   CASE IP_Arr_OP90JB[Input_Page_num] OF
	500: Lamp4:=I90_BOWL1_RDYI500_3 ;
	501: Lamp4:=I90_CONV1_TRK1_CHO_MOD1I501_3 ;
	502: Lamp4:=I90_HPR2_SOL_DOOR_SW_FBI502_3 ;
	503: Lamp4:=I90_VBF1_CONV2_TRK2_OVERFLWI503_3;
	504: Lamp4:=I90_VBF2_CONV_TRK_OVERFLW_2I504_3 ;
	505: Lamp4:=I90_SPARE_I505_3 ;
   ELSE
       Visibility_4:=FALSE;	
   END_CASE
   
   
    Visibility_5:=TRUE;
   
   CASE IP_Arr_OP90JB[Input_Page_num] OF
	500: Lamp5:=I90_BOWL1_LOW_LVLI500_4 ;
	501: Lamp5:=I90_CONV1_TRK1_CHO_MOD2I501_4 ;
	502: Lamp5:=I90_BOWL2_RDYI502_4 ;
	503: Lamp5:=I90_CONV2_TRK1_CHO_MOD1I503_4;
	504: Lamp5:=I90_SPARE_I504_4 ;
	505: Lamp5:=I90_SPARE_I505_4 ;
   ELSE
       Visibility_5:=FALSE;	
   END_CASE
   
   
    Visibility_6:=TRUE;
   
   CASE IP_Arr_OP90JB[Input_Page_num] OF
	500: Lamp6:=I90_BOWL1_OFF_ONI500_5 ;
	501: Lamp6:=I90_CONV1_TRK2_CHO_MOD1I501_5 ;
	502: Lamp6:=I90_BOWL2_LOW_LVLI502_5 ;
	503: Lamp6:=I90_CONV2_TRK1_CHO_MOD2I503_5;
	504: Lamp6:=I90_SPARE_I504_5 ;
	505: Lamp6:=I90_SPARE_I505_5 ;
   ELSE
       Visibility_6:=FALSE;	
   END_CASE
   
   
    Visibility_7:=TRUE;
   
   CASE IP_Arr_OP90JB[Input_Page_num] OF
	500: Lamp7:=I90_HPR1_OFF_ONI500_6 ;
	501: Lamp7:=I90_CONV1_TRK2_CHO_MOD2I501_6 ;
	502: Lamp7:=I90_BOWL2_OFF_ONI502_6 ;
	503: Lamp7:=I90_CONV2_TRK2_CHO_MOD1I503_6;
	504: Lamp7:=I90_SPARE_I504_6 ;
	505: Lamp7:=I90_SPARE_I505_6 ;
   ELSE
       Visibility_7:=FALSE;	
   END_CASE
   
   
    Visibility_8:=TRUE;
   
   CASE IP_Arr_OP90JB[Input_Page_num] OF
	500: Lamp8:=I90_CONV1_REVI500_7 ;
	501: Lamp8:=I90_CONV1_TRK3_CHO_MOD1I501_7 ;
	502: Lamp8:=I90_HPR2_OFF_ONI502_7 ;
	503: Lamp8:=I90_CONV2_TRK2_CHO_MOD2I503_7;
	504: Lamp8:=I90_SPARE_I504_7 ;
	505: Lamp8:=I90_SPARE_I505_7 ;
   ELSE
       Visibility_8:=FALSE;	
   END_CASE
	
    CASE OP_Arr_OP90[Output_Page_num] OF
    500: OLine1:=" O90_HPR1_ENABLE(Q500.0)  ";
    501: OLine1:=" O90_HPR2_ENABLE(Q501.0)  ";
    502: OLine1:=" O90_SPARE_Q502_0(Q502.0) ";
    503: OLine1:=" O90_SPARE_Q503_0(Q503.0) ";
    else
     OLine1:=" ";
    end_case 
    
    CASE OP_Arr_OP90[Output_Page_num] OF
    500: OLine2:="O90_BOWL1_ENABLE(Q500.1)";
    501: OLine2:="O90_BOWL2_ENABLE(Q501.1)";
    502: OLine2:="O90_SPARE_Q502_1(Q502.1)";
    503: OLine2:="O90_SPARE_Q503_1(Q503.1)";
    else
     OLine2:=" ";
    end_case 
    
    CASE OP_Arr_OP90[Output_Page_num] OF
    500: OLine3:="O90_HPR1_TWR_LMP_RED(Q500.2)";
    501: OLine3:="O90_HPR2_TWR_LMP_RED(Q501.2)";
    502: OLine3:="O90_SPARE_Q502_2(Q502.2)    ";
    503: OLine3:="O90_SPARE_Q503_2(Q503.2)    ";
    else
     OLine3:=" ";
    end_case 
    
    CASE OP_Arr_OP90[Output_Page_num] OF
    500: OLine4:="O90_HPR1_TWR_LMP_GREEN(Q500.3)";
    501: OLine4:="O90_HPR2_TWR_LMP_GREEN(Q501.3)";
    502: OLine4:="O90_SPARE_Q502_3(Q502.3)      ";
    503: OLine4:="O90_SPARE_Q503_3(Q503.3)      ";
    else
     OLine4:=" ";
    end_case 
    
    CASE OP_Arr_OP90[Output_Page_num] OF
    500: OLine5:="O90_BOWL1_AIR_PURGE1(Q500.4)";
    501: OLine5:="O90_BOWL2_AIR_PURGE1(Q501.4)";
    502: OLine5:="O90_SPARE_Q502_4(Q502.4)    ";
    503: OLine5:="O90_SPARE_Q503_4(Q503.4)    ";
    else
     OLine5:=" ";
    end_case 
    
    CASE OP_Arr_OP90[Output_Page_num] OF
    500: OLine6:="O90_BOWL1_AIR_PURGE2(Q500.5)";
    501: OLine6:="O90_BOWL2_AIR_PURGE2(Q501.5)";
    502: OLine6:="O90_SPARE_Q502_5(Q502.5)    ";
    503: OLine6:="O90_SPARE_Q503_5(Q503.5)    ";
    else
     OLine6:=" ";
    end_case 
    
    CASE OP_Arr_OP90[Output_Page_num] OF
    500: OLine7:="O90_HPR1_DOOR_OPN(Q500.6)";
    501: OLine7:="O90_HPR2_DOOR_OPN(Q501.6)";
    502: OLine7:="O90_SPARE_Q502_6(Q502.6) ";
    503: OLine7:="O90_SPARE_Q503_6(Q503.6) ";
    else
     OLine7:=" ";
    end_case 
    
    CASE OP_Arr_OP90[Output_Page_num] OF
    500: OLine8:="O90_SPARE_Q500_7(Q500.7)";
    501: OLine8:="O90_SPARE_Q501_7(Q501.7)";
    502: OLine8:="O90_SPARE_Q502_7(Q502.7)";
    503: OLine8:="O90_SPARE_Q503_7(Q503.7)";
    else
     OLine8:=" ";
    END_CASE 
    Out_Visibility_1:=TRUE;
    CASE OP_Arr_OP90[Output_Page_num] OF
	500:  Out_Lamp1:=O90_HPR1_ENABLEQ500_0;
	501:  Out_Lamp1:=O90_HPR2_ENABLEQ501_0;
	502:  Out_Lamp1:=O90_SPARE_Q502_0;
	503:  Out_Lamp1:=O90_SPARE_Q503_0;
    ELSE
       Out_Visibility_1:=FALSE;	
    END_CASE
   
    Out_Visibility_2:=TRUE;
   
    CASE OP_Arr_OP90[Output_Page_num] OF
	500:  Out_Lamp2:=O90_BOWL1_ENABLEQ500_1;
	501:  Out_Lamp2:=O90_BOWL2_ENABLEQ501_1;
	502:  Out_Lamp2:=O90_SPARE_Q502_1;
	503:  Out_Lamp2:=O90_SPARE_Q503_1;
    ELSE
       Out_Visibility_2:=FALSE;	
    END_CASE 
   
    Out_Visibility_3:=TRUE;
	
    CASE OP_Arr_OP90[Output_Page_num] OF
	500:  Out_Lamp3:=O90_HPR1_TWR_LMP_REDQ500_2; 
	501:  Out_Lamp3:=O90_HPR2_TWR_LMP_REDQ501_2; 
	502:  Out_Lamp3:=O90_SPARE_Q502_2; 
	503:  Out_Lamp3:=O90_SPARE_Q503_2; 
    ELSE
       Out_Visibility_3:=FALSE;
    END_CASE 
   
    Out_Visibility_4:=TRUE;
   
    CASE OP_Arr_OP90[Output_Page_num] OF
	500:  Out_Lamp4:=O90_HPR1_TWR_LMP_GREENQ500_3; 
	501:  Out_Lamp4:=O90_HPR2_TWR_LMP_GREENQ501_3; 
	502:  Out_Lamp4:=O90_SPARE_Q502_3; 
	503:  Out_Lamp4:=O90_SPARE_Q503_3;  
    ELSE
       Out_Visibility_4:=FALSE;
    END_CASE 
   
    Out_Visibility_5:=TRUE;
	
    CASE OP_Arr_OP90[Output_Page_num] OF
	500:  Out_Lamp5:=O90_BOWL1_AIR_PURGE1Q500_4; 
	501:  Out_Lamp5:=O90_BOWL2_AIR_PURGE1Q501_4; 
	502:  Out_Lamp5:=O90_SPARE_Q502_4; 
	503:  Out_Lamp5:=O90_SPARE_Q503_4; 
   ELSE
       Out_Visibility_5:=FALSE;
   END_CASE 
   
    Out_Visibility_6:=TRUE;
	
   CASE OP_Arr_OP90[Output_Page_num] OF
	500:  Out_Lamp6:=O90_BOWL1_AIR_PURGE2Q500_5; 
	501:  Out_Lamp6:=O90_BOWL2_AIR_PURGE2Q501_5; 
	502:  Out_Lamp6:=O90_SPARE_Q502_5; 
	503:  Out_Lamp6:=O90_SPARE_Q503_5; 
   ELSE           
       Out_Visibility_6:=FALSE;
   END_CASE 
    
	Out_Visibility_7:=TRUE;
	
   CASE OP_Arr_OP90[Output_Page_num] OF
	500:  Out_Lamp7:=O90_HPR1_DOOR_OPNQ500_6; 
	501:  Out_Lamp7:=O90_HPR2_DOOR_OPNQ501_6; 
	502:  Out_Lamp7:=O90_SPARE_Q502_6; 
	503:  Out_Lamp7:=O90_SPARE_Q503_6;  
   ELSE 
       Out_Visibility_7:=FALSE;
   END_CASE 
   
    Out_Visibility_8:=TRUE;
   
   CASE OP_Arr_OP90[Output_Page_num] OF
	500:  Out_Lamp8:=O90_SPARE_Q500_7;  
	501:  Out_Lamp8:=O90_SPARE_Q501_7;  
	502:  Out_Lamp8:=O90_SPARE_Q502_7;  
	503:  Out_Lamp8:=O90_SPARE_Q503_7;   
   ELSE
       Out_Visibility_8:=FALSE;	
   END_CASE
 7:	CASE IP_Arr_OP120_JB[Input_Page_num] OF
    600: Line1:="I120_SPARE_600_0(I600.0)        ";
    601: Line1:="I120_CONV_FWD(I601.0)           ";
    602: Line1:="I120_CONV_TRK3_CHO_MOD2(I602.0) ";
    603: Line1:="I120_SPARE_I603_0(I603.0)       ";
    else
     Line1:=" ";
    end_case 
     
    CASE IP_Arr_OP120_JB[Input_Page_num] OF
    600: Line2:="I120_HPR_LOW_LVL_FB(I600.1)       ";
    601: Line2:="I120_VBF_CONV_TRK1_OVERFLW(I601.1)";
    602: Line2:="I120_VBF_CONV_TRK_OVERFLW2(I602.1)   ";
    603: Line2:="I120_SPARE_I603_1(I603.1)         ";
    else
     Line2:=" ";
    end_case 
     
    CASE IP_Arr_OP120_JB[Input_Page_num] OF
    600: Line3:="I120_HPR_SOL_DOOR_SW_FB(I600.2)   ";
    601: Line3:="I120_VBF_CONV_TRK2_OVERFLW(I601.2)";
    602: Line3:="I120_SPARE_I602_2(I602.2)         ";
    603: Line3:="I120_SPARE_I603_2(I603.2)         ";
    else
     Line3:=" ";
    end_case 
     
    CASE IP_Arr_OP120_JB[Input_Page_num] OF
    600: Line4:="I120_BOWL_RDY(I600.3)          ";
    601: Line4:="I120_CONV_TRK1_CHO_MOD1(I601.3)";
    602: Line4:="I120_SPARE_I602_3(I602.3)      ";
    603: Line4:="I120_SPARE_I603_3(I603.3)      ";
    else
     Line4:=" ";
    end_case 
     
    CASE IP_Arr_OP120_JB[Input_Page_num] OF
    600: Line5:="I120_BOWL_LOW_LVL(I600.4)      ";
    601: Line5:="I120_CONV_TRK1_CHO_MOD2(I601.4)";
    602: Line5:="I120_SPARE_I602_4(I602.4)      ";
    603: Line5:="I120_SPARE_I603_4(I603.4)      ";
    else
     Line5:=" ";
    end_case 
     
    CASE IP_Arr_OP120_JB[Input_Page_num] OF
    600: Line6:="I120_BOWL_OFF_ON(I600.5)       ";
    601: Line6:="I120_CONV_TRK2_CHO_MOD1(I601.5)";
    602: Line6:="I120_SPARE_I602_5(I602.5)      ";
    603: Line6:="I120_SPARE_I603_5(I603.5)      ";
    else
     Line6:=" ";
    end_case 
     
    CASE IP_Arr_OP120_JB[Input_Page_num] OF
    600: Line7:="I120_HPR_OFF_ON(I600.6)        ";
    601: Line7:="I120_CONV_TRK2_CHO_MOD2(I601.6)";
    602: Line7:="I120_SPARE_I602_6(I602.6)      ";
    603: Line7:="I120_SPARE_I603_6(I603.6)      ";
    else
     Line7:=" ";
    end_case 
     
    CASE IP_Arr_OP120_JB[Input_Page_num] OF
    600: Line8:="I120_CONV_REV(I600.7)           ";
    601: Line8:="I120_CONV_TRK3_CHO_MOD1(I601.7) ";
    602: Line8:="I120_SPARE_I602_7(I602.7)       ";
    603: Line8:="I120_SPARE_I603_7(I603.7)       ";
    else
     Line8:=" ";
    END_CASE 
	Visibility_1:=TRUE;
   
   CASE IP_Arr_OP120_JB[Input_Page_num] OF
	600: Lamp1:=I120_SPARE_600_0I600_0 ;
	601: Lamp1:=I120_CONV_FWDI601_0 ;
	602: Lamp1:=I120_CONV_TRK3_CHO_MOD2I602_0 ;
	603: Lamp1:=I120_SPARE_I603_0;
   ELSE
       Visibility_1:=FALSE;	
   END_CASE
   
   
   Visibility_2:=TRUE;
   
   CASE IP_Arr_OP120_JB[Input_Page_num] OF
	600: Lamp2:=I120_HPR_LOW_LVL_FBI600_1 ;
	601: Lamp2:=I120_VBF_CONV_TRK1_OVERFLW_I601_1 ;
	602: Lamp2:=I120_VBF_CONV_TRK_OVERFLW2_I602_1 ;
	603: Lamp2:=I120_SPARE_I603_1;
   ELSE
       Visibility_2:=FALSE;	
   END_CASE
   
   
    Visibility_3:=TRUE;
   
   CASE IP_Arr_OP120_JB[Input_Page_num] OF
	600: Lamp3:=I120_HPR_SOL_DOOR_SW_FBI600_2 ;
	601: Lamp3:=I120_VBF_CONV_TRK2_OVERFLWI601_2 ;
	602: Lamp3:=I120_SPARE_I602_2 ;
	603: Lamp3:=I120_SPARE_I603_2;
   ELSE
       Visibility_3:=FALSE;	
   END_CASE

    Visibility_4:=TRUE;
   
   CASE IP_Arr_OP120_JB[Input_Page_num] OF
	600: Lamp4:=I120_BOWL_RDYI600_3 ;
	601: Lamp4:=I120_CONV_TRK1_CHO_MOD1I601_3 ;
	602: Lamp4:=I120_SPARE_I602_3 ;
	603: Lamp4:=I120_SPARE_I603_3;
   ELSE
       Visibility_4:=FALSE;	
   END_CASE
   
   
    Visibility_5:=TRUE;
   
   CASE IP_Arr_OP120_JB[Input_Page_num] OF
	600: Lamp5:=I120_BOWL_LOW_LVLI600_4 ;
	601: Lamp5:=I120_CONV_TRK1_CHO_MOD2I601_4 ;
	602: Lamp5:=I120_SPARE_I602_4 ;
	603: Lamp5:=I120_SPARE_I603_4;
   ELSE
       Visibility_5:=FALSE;	
   END_CASE
   
   
    Visibility_6:=TRUE;
   
   CASE IP_Arr_OP120_JB[Input_Page_num] OF
	600: Lamp6:=I120_BOWL_OFF_ONI600_5 ;
	601: Lamp6:=I120_CONV_TRK2_CHO_MOD1I601_5 ;
	602: Lamp6:=I120_SPARE_I602_5 ;
	603: Lamp6:=I120_SPARE_I603_5;
   ELSE
       Visibility_6:=FALSE;	
   END_CASE
   
   
    Visibility_7:=TRUE;
   
   CASE IP_Arr_OP120_JB[Input_Page_num] OF
	600: Lamp7:=I120_HPR_OFF_ONI600_6 ;
	601: Lamp7:=I120_CONV_TRK2_CHO_MOD2I601_6 ;
	602: Lamp7:=I120_SPARE_I602_6 ;
	603: Lamp7:=I120_SPARE_I603_6;
   ELSE
       Visibility_7:=FALSE;	
   END_CASE
   
   
    Visibility_8:=TRUE;
   
   CASE IP_Arr_OP120_JB[Input_Page_num] OF
	600: Lamp8:=I120_CONV_REVI600_7 ;
	601: Lamp8:=I120_CONV_TRK3_CHO_MOD1I601_7 ;
	602: Lamp8:=I120_SPARE_I602_7 ;
	603: Lamp8:=I120_SPARE_I603_7;
   ELSE
       Visibility_8:=FALSE;	
   END_CASE
    
    CASE OP_Arr_OP120[Output_Page_num] OF
    600: OLine1:="O120_HPR_ENABLE(Q600.0)   ";
    601: OLine1:="O120_SPARE_Q601_0(Q601.0) ";
    602: OLine1:="O120_SPARE_Q602_0(Q602.0) ";
    603: OLine1:="O120_SPARE_Q603_0(Q603.0) ";
    else
     OLine1:=" ";
    end_case 
    
    CASE OP_Arr_OP120[Output_Page_num] OF
    600: OLine2:="O120_BOWL_ENABLE(Q600.1) ";
    601: OLine2:="O120_SPARE_Q601_1(Q601.1)";
    602: OLine2:="O120_SPARE_Q602_1(Q602.1)";
    603: OLine2:="O120_SPARE_Q603_1(Q603.1)";
    else
     OLine2:=" ";
    end_case 
    
    CASE OP_Arr_OP120[Output_Page_num] OF
    600: OLine3:="O120_HPR_TWR_LMP_RED(Q600.2)";
    601: OLine3:="O120_SPARE_Q601_2(Q601.2)   ";
    602: OLine3:="O120_SPARE_Q602_2(Q602.2)   ";
    603: OLine3:="O120_SPARE_Q603_2(Q603.2)   ";
    else
     OLine3:=" ";
    end_case 
    
    CASE OP_Arr_OP120[Output_Page_num] OF
    600: OLine4:="O120_HPR_TWR_LMP_GREEN(Q600.3)";
    601: OLine4:="O120_SPARE_Q601.3(Q601.3)     ";
    602: OLine4:="O120_SPARE_Q602.3(Q602.3)     ";
    603: OLine4:="O120_SPARE_Q603.3(Q603.3)     ";
    else
     OLine4:=" ";
    end_case 
    
    CASE OP_Arr_OP120[Output_Page_num] OF
    600: OLine5:="O120_BOWL_AIR_PURGE1(Q600.4)";
    601: OLine5:="O120_SPARE_Q601_4(Q601.4)   ";
    602: OLine5:="O120_SPARE_Q602_4(Q602.4)   ";
    603: OLine5:="O120_SPARE_Q603_4(Q603.4)   ";
    else
     OLine5:=" ";
    end_case 
    
    CASE OP_Arr_OP120[Output_Page_num] OF
    600: OLine6:="O120_BOWL_AIR_PURGE2(Q600.5)";
    601: OLine6:="O120_SPARE_Q601_5(Q601.5)   ";
    602: OLine6:="O120_SPARE_Q602_5(Q602.5)   ";
    603: OLine6:="O120_SPARE_Q603_5(Q603.5)   ";
    else
     OLine6:=" ";
    end_case 
    
    CASE OP_Arr_OP120[Output_Page_num] OF
    600: OLine7:="O120_HPR_DOOR_OPN(Q600.6)";
    601: OLine7:="O120_SPARE_Q601_6(Q601.6)";
    602: OLine7:="O120_SPARE_Q602_6(Q602.6)";
    603: OLine7:="O120_SPARE_Q603_6(Q603.6)";
    else
     OLine7:=" ";
    end_case 
    
    CASE OP_Arr_OP120[Output_Page_num] OF
    600: OLine8:="O120_SPARE_Q600_7(Q600.7)";
    601: OLine8:="O120_SPARE_Q601_7(Q601.7)";
    602: OLine8:="O120_SPARE_Q602_7(Q602.7)";
    603: OLine8:="O120_SPARE_Q603_7(Q603.7)";
    else
     OLine8:=" ";
    END_CASE 
	   Out_Visibility_1:=TRUE;
   
   CASE OP_Arr_OP120[Output_Page_num] OF
	600:  Out_Lamp1:=O120_HPR_ENABLEQ600_0;
	601:  Out_Lamp1:=O120_SPARE_Q601_0;
	602:  Out_Lamp1:=O120_SPARE_Q602_0;
	603:  Out_Lamp1:=O120_SPARE_Q603_0;
   ELSE
       Out_Visibility_1:=FALSE;	
   END_CASE
   
    Out_Visibility_2:=TRUE;
   
   CASE OP_Arr_OP120[Output_Page_num] OF
	600:  Out_Lamp2:=O120_BOWL_ENABLEQ600_1;
	601:  Out_Lamp2:=O120_SPARE_Q601_1;
	602:  Out_Lamp2:=O120_SPARE_Q602_1;
	603:  Out_Lamp2:=O120_SPARE_Q603_1;
   ELSE
       Out_Visibility_2:=FALSE;	
   END_CASE 
   
    Out_Visibility_3:=TRUE;
	
   CASE OP_Arr_OP10A[Output_Page_num] OF
	600:  Out_Lamp3:=O120_HPR_TWR_LMP_REDQ600_2; 
	601:  Out_Lamp3:=O120_SPARE_Q601_2; 
	602:  Out_Lamp3:=O120_SPARE_Q602_2; 
	603:  Out_Lamp3:=O120_SPARE_Q603_2; 
   ELSE
       Out_Visibility_3:=FALSE;
   END_CASE 
   
    Out_Visibility_4:=TRUE;
   
   CASE OP_Arr_OP120[Output_Page_num] OF
	700:  Out_Lamp4:=O120_HPR_TWR_LMP_GREENQ600_3; 
	701:  Out_Lamp4:=O120_SPARE_Q601_3; 
	702:  Out_Lamp4:=O120_SPARE_Q602_3; 
	703:  Out_Lamp4:=O120_SPARE_Q603_3; 
   ELSE
       Out_Visibility_4:=FALSE;
   END_CASE 
   
    Out_Visibility_5:=TRUE;
	
    CASE OP_Arr_OP120[Output_Page_num] OF
	600:  Out_Lamp5:=O120_BOWL_AIR_PURGE1Q600_4; 
	601:  Out_Lamp5:=O120_SPARE_Q601_4; 
	602:  Out_Lamp5:=O120_SPARE_Q602_4; 
	603:  Out_Lamp5:=O120_SPARE_Q603_4; 
   ELSE
       Out_Visibility_5:=FALSE;
   END_CASE 
   
    Out_Visibility_6:=TRUE;
	
   CASE OP_Arr_OP120[Output_Page_num] OF
	600:  Out_Lamp6:=O120_BOWL_AIR_PURGE2Q600_5; 
	601:  Out_Lamp6:=O120_SPARE_Q601_5; 
	602:  Out_Lamp6:=O120_SPARE_Q602_5; 
	603:  Out_Lamp6:=O120_SPARE_Q603_5; 
   ELSE           
       Out_Visibility_6:=FALSE;
   END_CASE 
    
	Out_Visibility_7:=TRUE;
	
   CASE OP_Arr_OP120[Output_Page_num] OF
	600:  Out_Lamp7:=O120_HPR_DOOR_OPNQ600_6; 
	601:  Out_Lamp7:=O120_SPARE_Q601_6; 
	602:  Out_Lamp7:=O120_SPARE_Q602_6; 
	603:  Out_Lamp7:=O120_SPARE_Q603_6; 
   ELSE 
       Out_Visibility_7:=FALSE;
   END_CASE 
   
    Out_Visibility_8:=TRUE;
   
   CASE OP_Arr_OP120[Output_Page_num] OF
	600:  Out_Lamp8:=O120_SPARE_Q600_7;  
	601:  Out_Lamp8:=O120_SPARE_Q601_7;  
	602:  Out_Lamp8:=O120_SPARE_Q602_7;  
	603:  Out_Lamp8:=O120_SPARE_Q603_7;  
   ELSE
       Out_Visibility_8:=FALSE;	
   END_CASE
	
 8: CASE Safety_IP[Input_Page_num] OF
    400: Line1:="IS90_DOORSW_SET1_CH1(IS400.0)";
    401: Line1:="IS90_DOORSW_SET5_CH1(IS401.0)";
    402: Line1:="IS90_ESTOP_CONT_EDM(IS402.0) ";
    700: Line1:="IS160_ESTOP_CONT_EDM(IS700.0)";
    else
     Line1:=" ";
    END_CASE 
    
    CASE Safety_IP[Input_Page_num] OF
    400: Line2:="IS90_DOORSW_SET2_CH1(IS400.1)";
    401: Line2:="IS90_DOORSW_SET6_CH1(IS401.1)";
    402: Line2:="IS90_DOOR_CONT_EDM(IS402.1)  ";
    700: Line2:="IS160_DOOR_CONT_EDM(IS700.1) ";
    else
     Line2:=" ";
    end_case 
    
    
    CASE Safety_IP[Input_Page_num] OF
    400: Line3:="IS90_DOORSW_SET3_CH1(IS400.2)";
    401: Line3:="IS90_LHS_ESTOP_CH1(IS401.2)  ";
    402: Line3:="IS90_RESET_IS402_2(IS402.2)  ";
    700: Line3:="IS160_SPARE_IS700_2(IS700.2) ";
    else
     Line3:=" ";
    end_case 
    
    
    CASE Safety_IP[Input_Page_num] OF
    400: Line4:="IS90_DOORSW_SET4_CH1(IS400.3)";
    401: Line4:="IS90_RHS_ESTOP_CH1(IS401.3)  ";
    402: Line4:="IS90_SPARE_IS402_3(IS402.3)  ";
    700: Line4:="IS160_SPARE_IS700_3(IS700.3) ";
    else
     Line4:=" ";
    end_case 
    
    CASE Safety_IP[Input_Page_num] OF
    400: Line5:="IS90_DOORSW_SET1_CH2(IS400.4)";
    401: Line5:="IS90_DOORSW_SET5_CH2(IS401.4)";
    402: Line5:="IS90_SPARE_IS402_4(IS402.4)  ";
    700: Line5:="IS160_SPARE_IS700_4(IS700.4) ";
    else
     Line5:=" ";
    end_case 
    
    CASE Safety_IP[Input_Page_num] OF
    400: Line6:="IS90_DOORSW_SET2_CH2(IS400.5)";
    401: Line6:="IS90_DOORSW_SET6_CH2(IS401.5)";
    402: Line6:="IS90_SPARE_IS402_5(IS402.5)  ";
    700: Line6:="IS160_SPARE_IS700_5(IS700.5) ";
    else
     Line6:=" ";
    end_case 
    
    CASE Safety_IP[Input_Page_num] OF
    400: Line7:="IS90_DOORSW_SET3_CH2(IS400.6)";
    401: Line7:="IS90_LHS_ESTOP_CH2(IS401.6)  ";
    402: Line7:="IS90_SPARE_IS402_6(IS402.6)  ";
    700: Line7:="IS160_SPARE_IS700_6(IS700.6) ";
    else
     Line7:=" ";
    end_case 
    
    CASE Safety_IP[Input_Page_num] OF
    400: Line8:="IS90_DOORSW_SET4_CH2(IS400.7)";
    401: Line8:="IS90_RHS_ESTOP_CH2(IS401.7)  ";
    402: Line8:="IS90_SPARE_IS402_7(IS402.7)  ";
    700: Line8:="IS160_SPARE_IS700_7(IS700.7) ";
    else
     Line8:=" ";
    END_CASE 
	   Visibility_1:=TRUE;
   
   CASE Safety_IP[Input_Page_num] OF
	400: Lamp1:=IS90_DOORSW_SET1_CH1_IS400_0 ;
	401: Lamp1:=IS90_DOORSW_SET5_CH1_IS401_0 ;
	402: Lamp1:=IS90_ESTOP_CONT_EDM_IS402_0 ;
	700: Lamp1:=IS160_ESTOP_CONT_EDM_IS700_0;
   ELSE
       Visibility_1:=FALSE;	
   END_CASE
   
   
   Visibility_2:=TRUE;
   
   CASE Safety_IP[Input_Page_num]OF
	400: Lamp2:=IS90_DOORSW_SET2_CH1_IS400_1 ;
	401: Lamp2:=IS90_DOORSW_SET6_CH1_IS401_1 ;
	402: Lamp2:=IS90_DOOR_CONT_EDM_IS402_1 ;
	700: Lamp2:=IS160_DOOR_CONT_EDM_IS700_1;
   ELSE
       Visibility_2:=FALSE;	
   END_CASE
   
   
    Visibility_3:=TRUE;
   
   CASE Safety_IP[Input_Page_num] OF
	400: Lamp3:=IS90_DOORSW_SET3_CH1_IS400_2 ;
	401: Lamp3:=IS90_LHS_ESTOP_CH1_IS401_2 ;
	402: Lamp3:=IS90_RESET_IS402_2 ;
	700: Lamp3:=IS160_SPARE_IS700_2;
   ELSE
       Visibility_3:=FALSE;	
   END_CASE
   
   
    Visibility_4:=TRUE;
   
   CASE Safety_IP[Input_Page_num] OF
	400: Lamp4:=IS90_DOORSW_SET4_CH1_IS400_3 ;
	401: Lamp4:=IS90_RHS_ESTOP_CH1_IS401_3 ;
	402: Lamp4:=IS90_SPARE_IS402_3 ;
	700: Lamp4:=IS160_SPARE_IS700_3;
   ELSE
       Visibility_4:=FALSE;	
   END_CASE
   
   
    Visibility_5:=TRUE;
   
   CASE Safety_IP[Input_Page_num] OF
	400: Lamp5:=IS90_DOORSW_SET1_CH2_IS400_4 ;
	401: Lamp5:=IS90_DOORSW_SET5_CH2_IS401_4 ;
	402: Lamp5:=IS90_SPARE_IS402_4 ;
	700: Lamp5:=IS160_SPARE_IS700_4;
   ELSE
       Visibility_5:=FALSE;	
   END_CASE
   
   
    Visibility_6:=TRUE;
   
   CASE Safety_IP[Input_Page_num] OF
	400: Lamp6:=IS90_DOORSW_SET2_CH2_IS400_5 ;
	401: Lamp6:=IS90_DOORSW_SET6_CH2_IS401_5 ;
	402: Lamp6:=IS90_SPARE_IS402_5 ;
	700: Lamp6:=IS160_SPARE_IS700_5;
   ELSE
       Visibility_6:=FALSE;	
   END_CASE
   
   
    Visibility_7:=TRUE;
   
   CASE Safety_IP[Input_Page_num] OF
	400: Lamp7:=IS90_DOORSW_SET3_CH2_IS400_6 ;
	401: Lamp7:=IS90_LHS_ESTOP_CH2_IS401_6 ;
	402: Lamp7:=IS90_SPARE_IS402_6 ;
	700: Lamp7:=IS160_SPARE_IS700_6;
   ELSE
       Visibility_7:=FALSE;	
   END_CASE
   
   
    Visibility_8:=TRUE;
   
   CASE Safety_IP[Input_Page_num] OF
	400: Lamp8:=IS90_DOORSW_SET4_CH2_IS400_7 ;
	401: Lamp8:=IS90_RHS_ESTOP_CH2_IS401_7 ;
	402: Lamp8:=IS90_SPARE_IS402_7 ;
	700: Lamp8:=IS160_SPARE_IS700_7;
   ELSE
       Visibility_8:=FALSE;	
   END_CASE

	CASE Safety_OP[Output_Page_num] OF
    400: OLine1:="OS90_ESTOP_CH1(QS400.0) ";
    700: OLine1:="OS160_ESTOP_CH1(QS700.0)";
    else
     OLine1:=" ";
    end_case 
    
    CASE Safety_OP[Output_Page_num] OF
    400: OLine2:="OS90_ESTOP_CH2(QS400.1) ";
    700: OLine2:="OS160_ESTOP_CH2(QS700.1)";
    else
     OLine2:=" ";
    end_case 
    
    CASE Safety_OP[Output_Page_num] OF
    400: OLine3:="OS90_DOORCH1(QS400.2)  ";
    700: OLine3:="OS160_DOORCH1(QS700.2) ";
    else
     OLine3:=" ";
    end_case 
    
    CASE Safety_OP[Output_Page_num] OF
    400: OLine4:="OS90_DOORCH2(QS400.3) ";
    700: OLine4:="OS160_DOORCH2(QS700.3)";
    else
     OLine4:=" ";
    END_CASE
	
	   Out_Visibility_1:=TRUE;
   
   CASE Safety_OP[Output_Page_num] OF
	400:  Out_Lamp1:=OS90_ESTOP_CH1_QS400_0;
	700:  Out_Lamp1:=OS160_ESTOP_CH1_QS700_0;
   ELSE
       Out_Visibility_1:=FALSE;	
   END_CASE
   
    Out_Visibility_2:=TRUE;
   
   CASE Safety_OP[Output_Page_num] OF
	400:  Out_Lamp2:=OS90_ESTOP_CH2_QS400_1;
	700:  Out_Lamp2:=OS160_ESTOP_CH2_QS700_1;
   ELSE
       Out_Visibility_2:=FALSE;	
   END_CASE 
   
    Out_Visibility_3:=TRUE;
	
   CASE Safety_OP[Output_Page_num] OF
	400:  Out_Lamp3:=OS90_DOORCH1_QS400_2; 
	700:  Out_Lamp3:=OS160_DOORCH1_QS700_2; 
   ELSE
       Out_Visibility_3:=FALSE;
   END_CASE 
   
    Out_Visibility_4:=TRUE;
   
    CASE Safety_OP[Output_Page_num] OF
	400:  Out_Lamp4:=OS90_DOORCH2_QS400_3; 
	700:  Out_Lamp4:=OS160_DOORCH2_QS700_3; 
    ELSE
	   Out_Visibility_4:=FALSE;
    END_CASE 
	   
    
    Out_Visibility_5:=FALSE; 
    Out_Visibility_6:=FALSE;
    Out_Visibility_7:=FALSE;
    Out_Visibility_8:=FALSE;
   
END_CASE	 

IF panel_num = 1 THEN
i:= IP_Arr_OP10P[Input_Page_num];
j:= OP_Arr_OP10P[Output_Page_num];	
 IF Input_Page_num >= 24 THEN
	Input_Page_num:=0;
 END_IF
 IF Output_Page_num >= 22 THEN
	Output_Page_num:=0;
 END_IF	
END_IF

IF panel_num = 2 THEN
i:= IP_Arr_OP90P[Input_Page_num];
j:= OP_Arr_OP90P[Output_Page_num];	
 IF Input_Page_num >= 12 THEN
	Input_Page_num:=0;
 END_IF
 IF Output_Page_num >= 12 THEN
	Output_Page_num:=0;
 END_IF	
END_IF

IF panel_num = 3 THEN
i:= IP_Arr_OP160P[Input_Page_num];
j:= OP_Arr_OP160P[Output_Page_num];	
 IF Input_Page_num >= 24 THEN
	Input_Page_num:=0;
 END_IF
 IF Output_Page_num >= 18 THEN
	Output_Page_num:=0;
 END_IF	
END_IF

IF panel_num = 4 THEN
i:= IP_Arr_OP10A[Input_Page_num];
j:= OP_Arr_OP10A[Output_Page_num];	
 IF Input_Page_num >= 4 THEN
	Input_Page_num:=0;
 END_IF
 IF Output_Page_num >= 4 THEN
	Output_Page_num:=0;
 END_IF	
END_IF

IF panel_num = 5 THEN
i:= IP_Arr_OP10B[Input_Page_num];
j:= OP_Arr_OP10B_JB[Output_Page_num];	
 IF Input_Page_num >= 4 THEN
	Input_Page_num:=0;
 END_IF
 IF Output_Page_num >= 4 THEN
	Output_Page_num:=0;
 END_IF	
END_IF

IF panel_num = 6 THEN
i:= IP_Arr_OP90JB[Input_Page_num];
j:= OP_Arr_OP90[Output_Page_num];	
 IF Input_Page_num >= 6 THEN
	Input_Page_num:=0;
 END_IF
 IF Output_Page_num >= 4 THEN
	Output_Page_num:=0;
 END_IF	
END_IF

IF panel_num = 7 THEN
i:= IP_Arr_OP120_JB[Input_Page_num];
j:= OP_Arr_OP120[Output_Page_num];	
 IF Input_Page_num >= 4 THEN
	Input_Page_num:=0;
 END_IF
 IF Output_Page_num >= 4 THEN
	Output_Page_num:=0;
 END_IF	
END_IF

IF panel_num = 8 THEN
 OLine5:=" ";
 OLine6:=" ";
 OLine7:=" ";
 OLine8:=" ";	
 i:= Safety_IP[Input_Page_num];
 j:= Safety_OP[Output_Page_num];	
  IF Input_Page_num >= 4 THEN
 	Input_Page_num:=0;
  END_IF
  IF Output_Page_num >= 2 THEN
 	Output_Page_num:=0;
  END_IF	
END_IF

END_PROGRAM

// ---- POUs/IO_mapping_OP10MP/IO_OP10_PANEL.TcPOU
PROGRAM IO_OP10_PANEL
VAR
	OP10_MP_16DI_MODULE_1 AT %I* : WORD;
	OP10_MP_16DI_MODULE_2 AT %I* : WORD;
	OP10_MP_16DI_MODULE_3 AT %I* : WORD;
	OP10_MP_16DI_MODULE_4 AT %I* : WORD;
	OP10_MP_16DI_MODULE_5 AT %I* : WORD;
	OP10_MP_16DI_MODULE_6 AT %I* : WORD;
	
	OP10_MP_16DO_MODULE_1 AT %Q* : WORD;
	OP10_MP_16DO_MODULE_2 AT %Q* : WORD;
	OP10_MP_16DO_MODULE_3 AT %Q* : WORD;
	OP10_MP_16DO_MODULE_4 AT %Q* : WORD;
	OP10_MP_16DO_MODULE_5 AT %Q* : WORD;
	
	WORD_AS_BIT_0: WORD_AS_BIT;
	WORD_AS_BIT_1: WORD_AS_BIT;
	WORD_AS_BIT_2: WORD_AS_BIT;
	WORD_AS_BIT_3: WORD_AS_BIT;
	WORD_AS_BIT_4: WORD_AS_BIT;
	WORD_AS_BIT_5: WORD_AS_BIT;

	BIT_AS_WORD_0: BIT_AS_WORD;
	BIT_AS_WORD_1: BIT_AS_WORD;
	BIT_AS_WORD_2: BIT_AS_WORD;
	BIT_AS_WORD_3: BIT_AS_WORD;
	BIT_AS_WORD_4: BIT_AS_WORD;
	OP10_MP_Spare_byte: WORD;
END_VAR

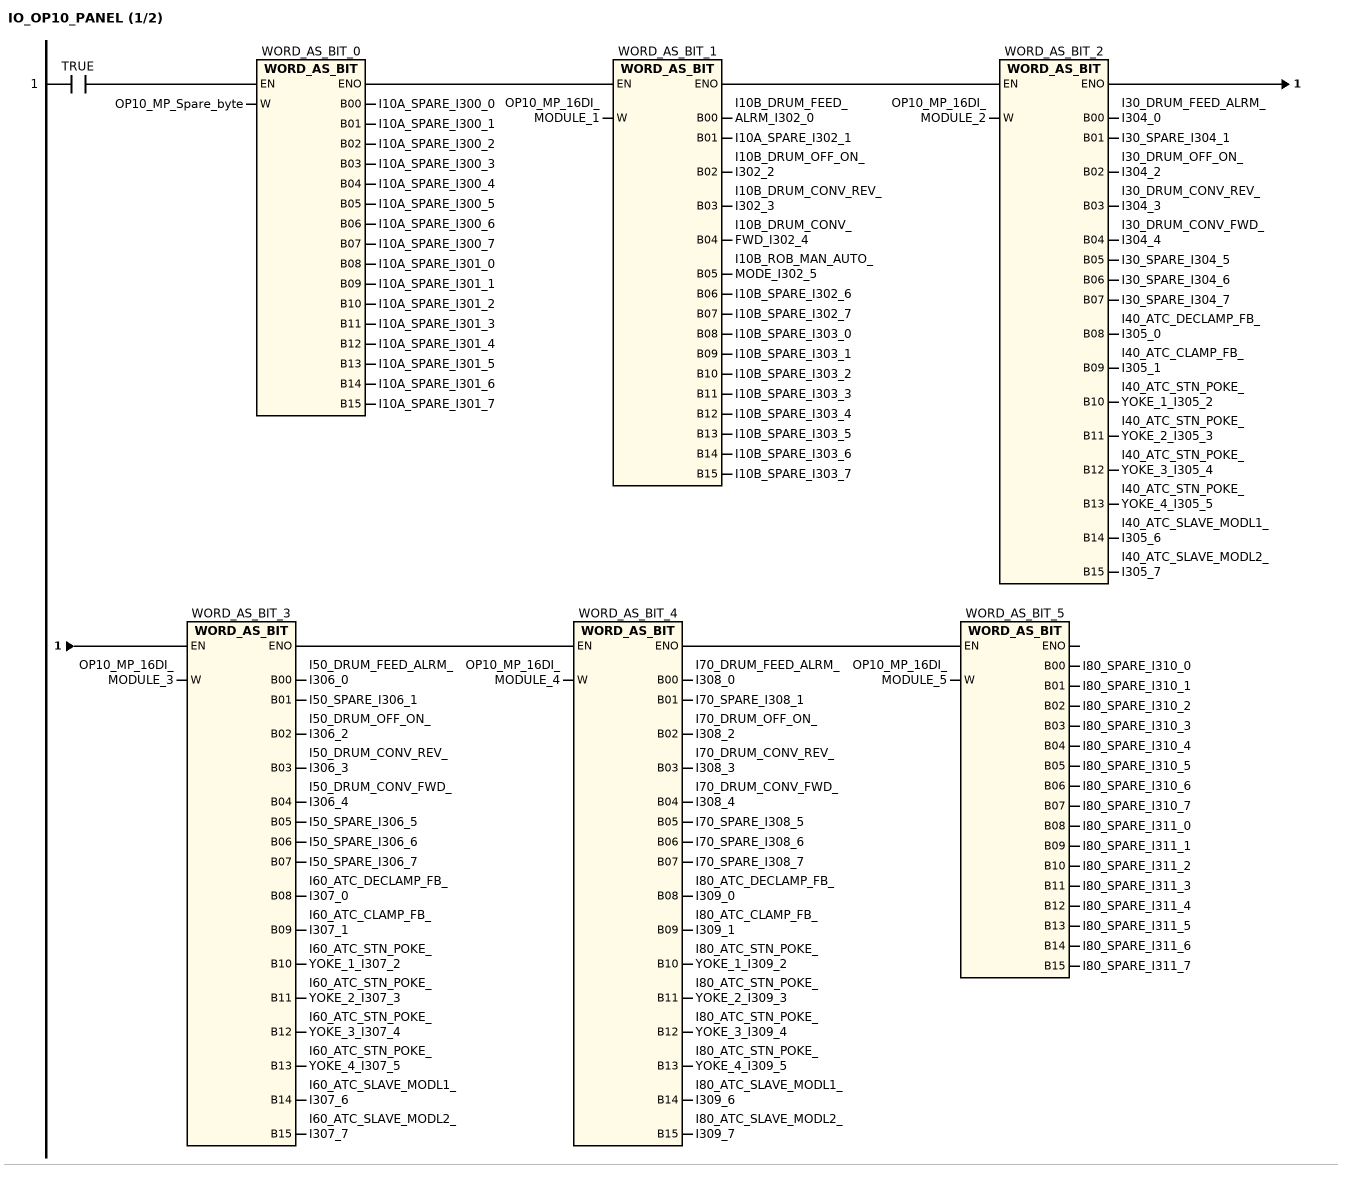
// NETWORK 1
WORD_AS_BIT_0(
    W := OP10_MP_Spare_byte,
    B00 => I10A_SPARE_I300_0,
    B01 => I10A_SPARE_I300_1,
    B02 => I10A_SPARE_I300_2,
    B03 => I10A_SPARE_I300_3,
    B04 => I10A_SPARE_I300_4,
    B05 => I10A_SPARE_I300_5,
    B06 => I10A_SPARE_I300_6,
    B07 => I10A_SPARE_I300_7,
    B08 => I10A_SPARE_I301_0,
    B09 => I10A_SPARE_I301_1,
    B10 => I10A_SPARE_I301_2,
    B11 => I10A_SPARE_I301_3,
    B12 => I10A_SPARE_I301_4,
    B13 => I10A_SPARE_I301_5,
    B14 => I10A_SPARE_I301_6,
    B15 => I10A_SPARE_I301_7); // WORD_AS_BIT
WORD_AS_BIT_1(
    W := OP10_MP_16DI_MODULE_1,
    B00 => I10B_DRUM_FEED_ALRM_I302_0,
    B01 => I10A_SPARE_I302_1,
    B02 => I10B_DRUM_OFF_ON_I302_2,
    B03 => I10B_DRUM_CONV_REV_I302_3,
    B04 => I10B_DRUM_CONV_FWD_I302_4,
    B05 => I10B_ROB_MAN_AUTO_MODE_I302_5,
    B06 => I10B_SPARE_I302_6,
    B07 => I10B_SPARE_I302_7,
    B08 => I10B_SPARE_I303_0,
    B09 => I10B_SPARE_I303_1,
    B10 => I10B_SPARE_I303_2,
    B11 => I10B_SPARE_I303_3,
    B12 => I10B_SPARE_I303_4,
    B13 => I10B_SPARE_I303_5,
    B14 => I10B_SPARE_I303_6,
    B15 => I10B_SPARE_I303_7); // WORD_AS_BIT
WORD_AS_BIT_2(
    W := OP10_MP_16DI_MODULE_2,
    B00 => I30_DRUM_FEED_ALRM_I304_0,
    B01 => I30_SPARE_I304_1,
    B02 => I30_DRUM_OFF_ON_I304_2,
    B03 => I30_DRUM_CONV_REV_I304_3,
    B04 => I30_DRUM_CONV_FWD_I304_4,
    B05 => I30_SPARE_I304_5,
    B06 => I30_SPARE_I304_6,
    B07 => I30_SPARE_I304_7,
    B08 => I40_ATC_DECLAMP_FB_I305_0,
    B09 => I40_ATC_CLAMP_FB_I305_1,
    B10 => I40_ATC_STN_POKE_YOKE_1_I305_2,
    B11 => I40_ATC_STN_POKE_YOKE_2_I305_3,
    B12 => I40_ATC_STN_POKE_YOKE_3_I305_4,
    B13 => I40_ATC_STN_POKE_YOKE_4_I305_5,
    B14 => I40_ATC_SLAVE_MODL1_I305_6,
    B15 => I40_ATC_SLAVE_MODL2_I305_7); // WORD_AS_BIT
WORD_AS_BIT_3(
    W := OP10_MP_16DI_MODULE_3,
    B00 => I50_DRUM_FEED_ALRM_I306_0,
    B01 => I50_SPARE_I306_1,
    B02 => I50_DRUM_OFF_ON_I306_2,
    B03 => I50_DRUM_CONV_REV_I306_3,
    B04 => I50_DRUM_CONV_FWD_I306_4,
    B05 => I50_SPARE_I306_5,
    B06 => I50_SPARE_I306_6,
    B07 => I50_SPARE_I306_7,
    B08 => I60_ATC_DECLAMP_FB_I307_0,
    B09 => I60_ATC_CLAMP_FB_I307_1,
    B10 => I60_ATC_STN_POKE_YOKE_1_I307_2,
    B11 => I60_ATC_STN_POKE_YOKE_2_I307_3,
    B12 => I60_ATC_STN_POKE_YOKE_3_I307_4,
    B13 => I60_ATC_STN_POKE_YOKE_4_I307_5,
    B14 => I60_ATC_SLAVE_MODL1_I307_6,
    B15 => I60_ATC_SLAVE_MODL2_I307_7); // WORD_AS_BIT
WORD_AS_BIT_4(
    W := OP10_MP_16DI_MODULE_4,
    B00 => I70_DRUM_FEED_ALRM_I308_0,
    B01 => I70_SPARE_I308_1,
    B02 => I70_DRUM_OFF_ON_I308_2,
    B03 => I70_DRUM_CONV_REV_I308_3,
    B04 => I70_DRUM_CONV_FWD_I308_4,
    B05 => I70_SPARE_I308_5,
    B06 => I70_SPARE_I308_6,
    B07 => I70_SPARE_I308_7,
    B08 => I80_ATC_DECLAMP_FB_I309_0,
    B09 => I80_ATC_CLAMP_FB_I309_1,
    B10 => I80_ATC_STN_POKE_YOKE_1_I309_2,
    B11 => I80_ATC_STN_POKE_YOKE_2_I309_3,
    B12 => I80_ATC_STN_POKE_YOKE_3_I309_4,
    B13 => I80_ATC_STN_POKE_YOKE_4_I309_5,
    B14 => I80_ATC_SLAVE_MODL1_I309_6,
    B15 => I80_ATC_SLAVE_MODL2_I309_7); // WORD_AS_BIT
WORD_AS_BIT_5(
    W := OP10_MP_16DI_MODULE_5,
    B00 => I80_SPARE_I310_0,
    B01 => I80_SPARE_I310_1,
    B02 => I80_SPARE_I310_2,
    B03 => I80_SPARE_I310_3,
    B04 => I80_SPARE_I310_4,
    B05 => I80_SPARE_I310_5,
    B06 => I80_SPARE_I310_6,
    B07 => I80_SPARE_I310_7,
    B08 => I80_SPARE_I311_0,
    B09 => I80_SPARE_I311_1,
    B10 => I80_SPARE_I311_2,
    B11 => I80_SPARE_I311_3,
    B12 => I80_SPARE_I311_4,
    B13 => I80_SPARE_I311_5,
    B14 => I80_SPARE_I311_6,
    B15 => I80_SPARE_I311_7); // WORD_AS_BIT

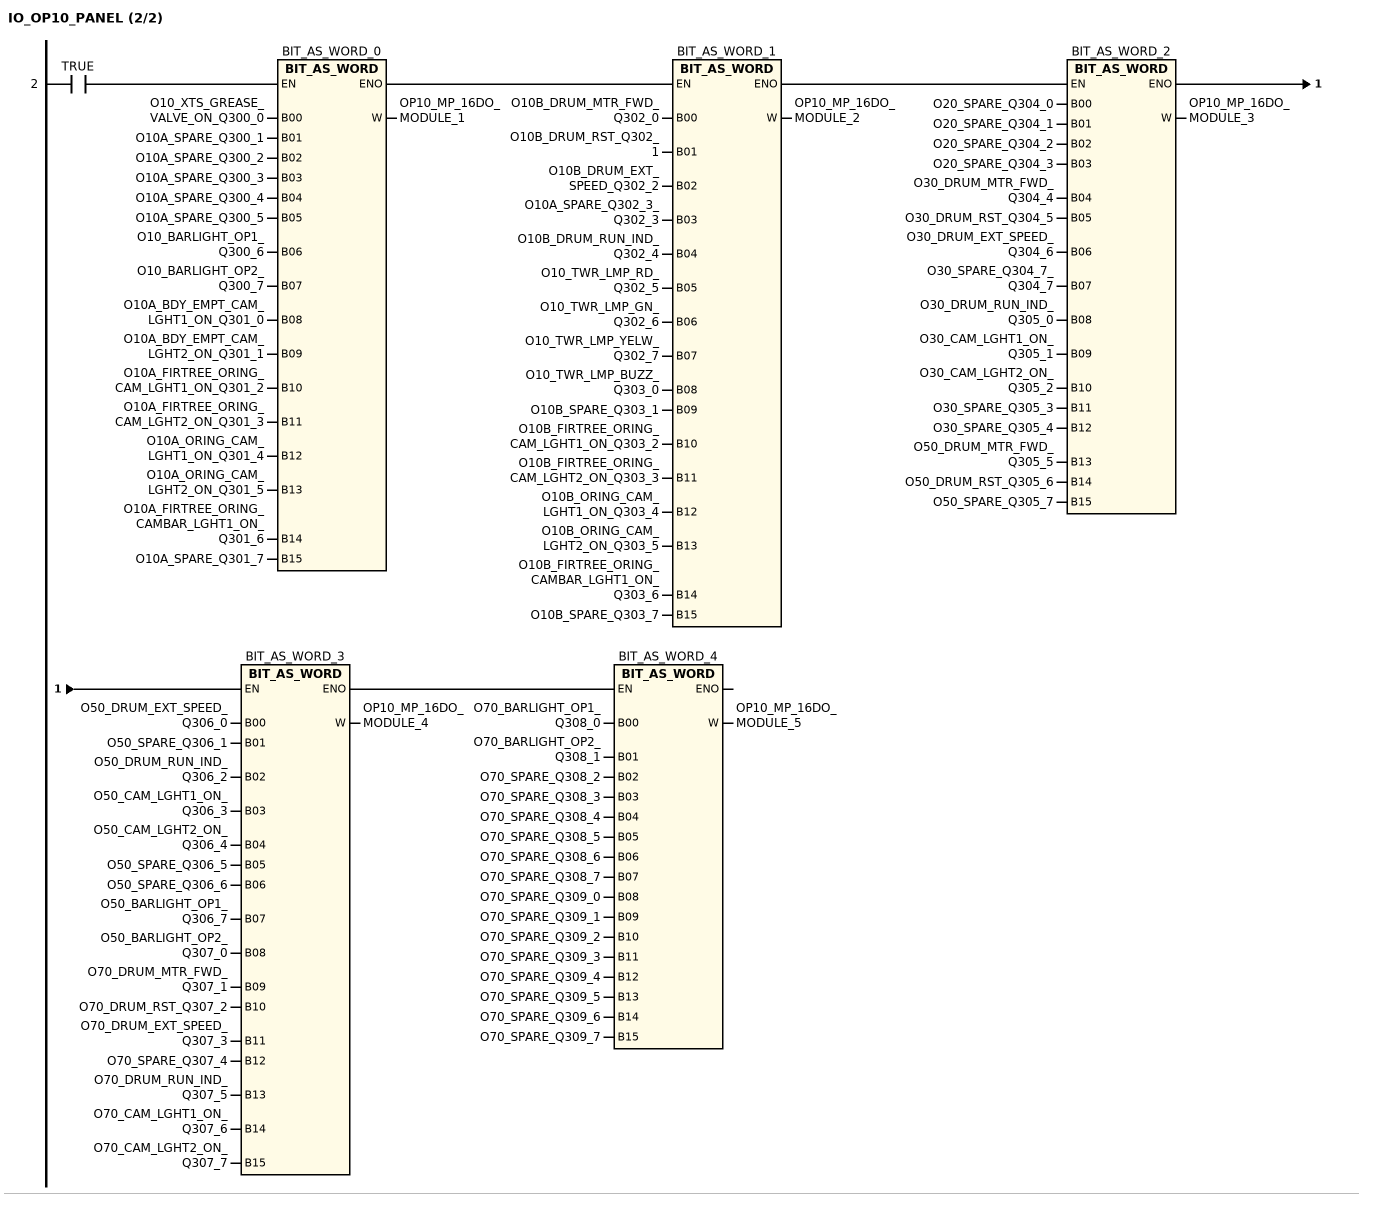
// NETWORK 2
BIT_AS_WORD_0(
    B00 := O10_XTS_GREASE_VALVE_ON_Q300_0,
    B01 := O10A_SPARE_Q300_1,
    B02 := O10A_SPARE_Q300_2,
    B03 := O10A_SPARE_Q300_3,
    B04 := O10A_SPARE_Q300_4,
    B05 := O10A_SPARE_Q300_5,
    B06 := O10_BARLIGHT_OP1_Q300_6,
    B07 := O10_BARLIGHT_OP2_Q300_7,
    B08 := O10A_BDY_EMPT_CAM_LGHT1_ON_Q301_0,
    B09 := O10A_BDY_EMPT_CAM_LGHT2_ON_Q301_1,
    B10 := O10A_FIRTREE_ORING_CAM_LGHT1_ON_Q301_2,
    B11 := O10A_FIRTREE_ORING_CAM_LGHT2_ON_Q301_3,
    B12 := O10A_ORING_CAM_LGHT1_ON_Q301_4,
    B13 := O10A_ORING_CAM_LGHT2_ON_Q301_5,
    B14 := O10A_FIRTREE_ORING_CAMBAR_LGHT1_ON_Q301_6,
    B15 := O10A_SPARE_Q301_7,
    W => OP10_MP_16DO_MODULE_1); // BIT_AS_WORD
BIT_AS_WORD_1(
    B00 := O10B_DRUM_MTR_FWD_Q302_0,
    B01 := O10B_DRUM_RST_Q302_1,
    B02 := O10B_DRUM_EXT_SPEED_Q302_2,
    B03 := O10A_SPARE_Q302_3_Q302_3,
    B04 := O10B_DRUM_RUN_IND_Q302_4,
    B05 := O10_TWR_LMP_RD_Q302_5,
    B06 := O10_TWR_LMP_GN_Q302_6,
    B07 := O10_TWR_LMP_YELW_Q302_7,
    B08 := O10_TWR_LMP_BUZZ_Q303_0,
    B09 := O10B_SPARE_Q303_1,
    B10 := O10B_FIRTREE_ORING_CAM_LGHT1_ON_Q303_2,
    B11 := O10B_FIRTREE_ORING_CAM_LGHT2_ON_Q303_3,
    B12 := O10B_ORING_CAM_LGHT1_ON_Q303_4,
    B13 := O10B_ORING_CAM_LGHT2_ON_Q303_5,
    B14 := O10B_FIRTREE_ORING_CAMBAR_LGHT1_ON_Q303_6,
    B15 := O10B_SPARE_Q303_7,
    W => OP10_MP_16DO_MODULE_2); // BIT_AS_WORD
BIT_AS_WORD_2(
    B00 := O20_SPARE_Q304_0,
    B01 := O20_SPARE_Q304_1,
    B02 := O20_SPARE_Q304_2,
    B03 := O20_SPARE_Q304_3,
    B04 := O30_DRUM_MTR_FWD_Q304_4,
    B05 := O30_DRUM_RST_Q304_5,
    B06 := O30_DRUM_EXT_SPEED_Q304_6,
    B07 := O30_SPARE_Q304_7_Q304_7,
    B08 := O30_DRUM_RUN_IND_Q305_0,
    B09 := O30_CAM_LGHT1_ON_Q305_1,
    B10 := O30_CAM_LGHT2_ON_Q305_2,
    B11 := O30_SPARE_Q305_3,
    B12 := O30_SPARE_Q305_4,
    B13 := O50_DRUM_MTR_FWD_Q305_5,
    B14 := O50_DRUM_RST_Q305_6,
    B15 := O50_SPARE_Q305_7,
    W => OP10_MP_16DO_MODULE_3); // BIT_AS_WORD
BIT_AS_WORD_3(
    B00 := O50_DRUM_EXT_SPEED_Q306_0,
    B01 := O50_SPARE_Q306_1,
    B02 := O50_DRUM_RUN_IND_Q306_2,
    B03 := O50_CAM_LGHT1_ON_Q306_3,
    B04 := O50_CAM_LGHT2_ON_Q306_4,
    B05 := O50_SPARE_Q306_5,
    B06 := O50_SPARE_Q306_6,
    B07 := O50_BARLIGHT_OP1_Q306_7,
    B08 := O50_BARLIGHT_OP2_Q307_0,
    B09 := O70_DRUM_MTR_FWD_Q307_1,
    B10 := O70_DRUM_RST_Q307_2,
    B11 := O70_DRUM_EXT_SPEED_Q307_3,
    B12 := O70_SPARE_Q307_4,
    B13 := O70_DRUM_RUN_IND_Q307_5,
    B14 := O70_CAM_LGHT1_ON_Q307_6,
    B15 := O70_CAM_LGHT2_ON_Q307_7,
    W => OP10_MP_16DO_MODULE_4); // BIT_AS_WORD
BIT_AS_WORD_4(
    B00 := O70_BARLIGHT_OP1_Q308_0,
    B01 := O70_BARLIGHT_OP2_Q308_1,
    B02 := O70_SPARE_Q308_2,
    B03 := O70_SPARE_Q308_3,
    B04 := O70_SPARE_Q308_4,
    B05 := O70_SPARE_Q308_5,
    B06 := O70_SPARE_Q308_6,
    B07 := O70_SPARE_Q308_7,
    B08 := O70_SPARE_Q309_0,
    B09 := O70_SPARE_Q309_1,
    B10 := O70_SPARE_Q309_2,
    B11 := O70_SPARE_Q309_3,
    B12 := O70_SPARE_Q309_4,
    B13 := O70_SPARE_Q309_5,
    B14 := O70_SPARE_Q309_6,
    B15 := O70_SPARE_Q309_7,
    W => OP10_MP_16DO_MODULE_5); // BIT_AS_WORD

END_PROGRAM

// ---- POUs/IO_Mapping_OP10JB/IO_OP10A_10B_JB.TcPOU
PROGRAM IO_OP10A_10B_JB
VAR
	//INPUT
	WORD_AS_BIT_0: WORD_AS_BIT;
	WORD_AS_BIT_1: WORD_AS_BIT;
	WORD_AS_BIT_2: WORD_AS_BIT;
	WORD_AS_BIT_3: WORD_AS_BIT;	
	//OUTPUT
	BIT_AS_WORD_0: BIT_AS_WORD;
	BIT_AS_WORD_1: BIT_AS_WORD;
	BIT_AS_WORD_2: BIT_AS_WORD;
	BIT_AS_WORD_3: BIT_AS_WORD;	
	//OP10A JB DI/DO 
	OP10A_BOWL_FEEDER_JB_16DI_MODULE_1 AT %I* : WORD;
	OP10A_BOWL_FEEDER_JB_16DI_MODULE_2 AT %I* : WORD;
	OP10A_BOWL_FEEDER_JB_16DO_MODULE_1 AT %Q* : WORD;
	OP10A_BOWL_FEEDER_JB_16DO_MODULE_2 AT %Q* : WORD;
	//OP10B JB DI/DO 
	OP10B_BOWL_FEEDER_JB_16DI_MODULE_1 AT %I* : WORD;
	OP10B_BOWL_FEEDER_JB_16DI_MODULE_2 AT %I* : WORD;
	OP10B_BOWL_FEEDER_JB_16DO_MODULE_1 AT %Q* : WORD;
	OP10B_BOWL_FEEDER_JB_16DO_MODULE_2 AT %Q* : WORD;
END_VAR

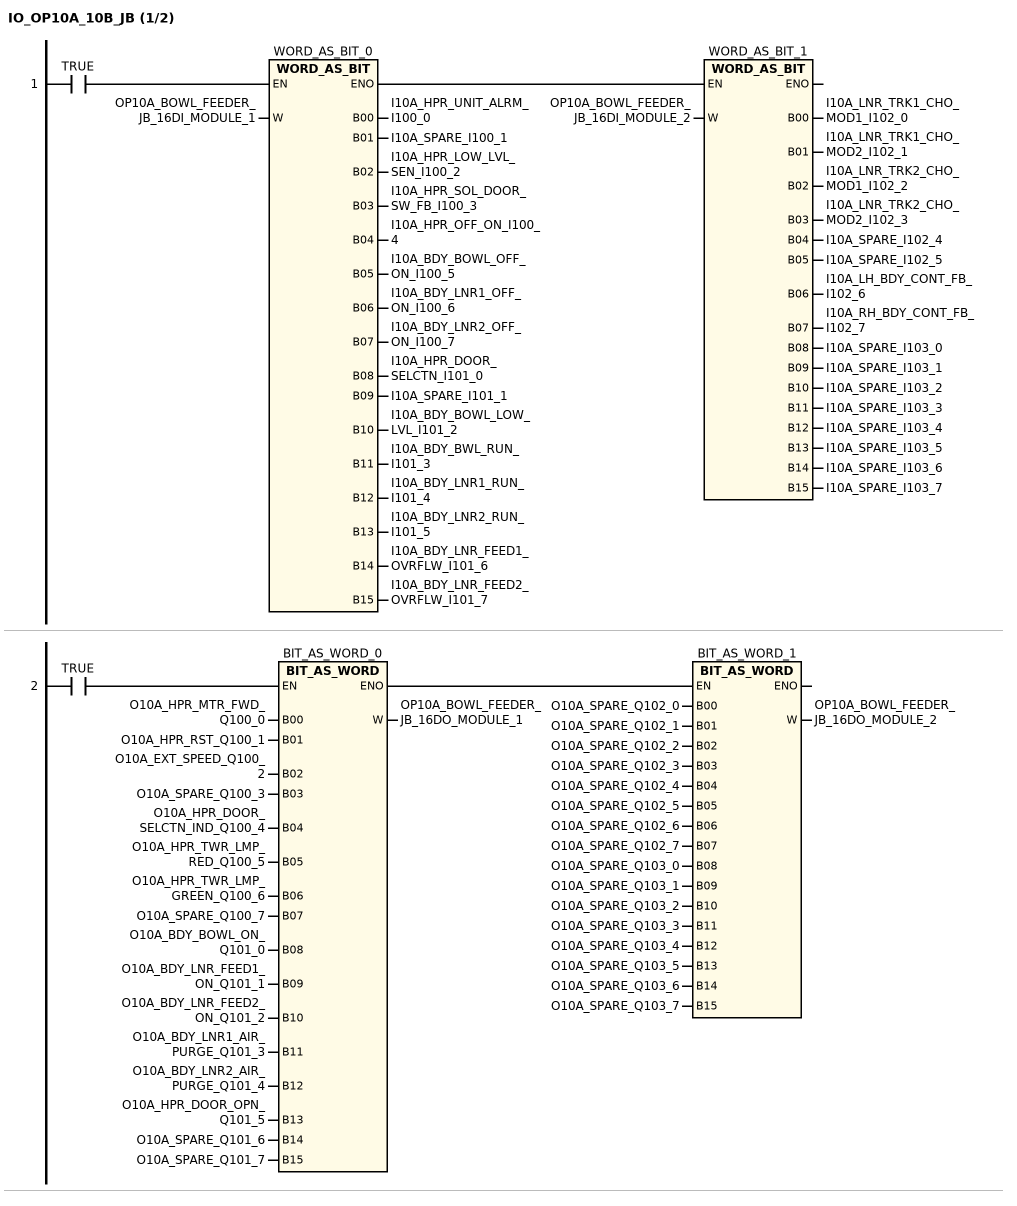
// NETWORK 1
WORD_AS_BIT_0(
    W := OP10A_BOWL_FEEDER_JB_16DI_MODULE_1,
    B00 => I10A_HPR_UNIT_ALRM_I100_0,
    B01 => I10A_SPARE_I100_1,
    B02 => I10A_HPR_LOW_LVL_SEN_I100_2,
    B03 => I10A_HPR_SOL_DOOR_SW_FB_I100_3,
    B04 => I10A_HPR_OFF_ON_I100_4,
    B05 => I10A_BDY_BOWL_OFF_ON_I100_5,
    B06 => I10A_BDY_LNR1_OFF_ON_I100_6,
    B07 => I10A_BDY_LNR2_OFF_ON_I100_7,
    B08 => I10A_HPR_DOOR_SELCTN_I101_0,
    B09 => I10A_SPARE_I101_1,
    B10 => I10A_BDY_BOWL_LOW_LVL_I101_2,
    B11 => I10A_BDY_BWL_RUN_I101_3,
    B12 => I10A_BDY_LNR1_RUN_I101_4,
    B13 => I10A_BDY_LNR2_RUN_I101_5,
    B14 => I10A_BDY_LNR_FEED1_OVRFLW_I101_6,
    B15 => I10A_BDY_LNR_FEED2_OVRFLW_I101_7); // WORD_AS_BIT
WORD_AS_BIT_1(
    W := OP10A_BOWL_FEEDER_JB_16DI_MODULE_2,
    B00 => I10A_LNR_TRK1_CHO_MOD1_I102_0,
    B01 => I10A_LNR_TRK1_CHO_MOD2_I102_1,
    B02 => I10A_LNR_TRK2_CHO_MOD1_I102_2,
    B03 => I10A_LNR_TRK2_CHO_MOD2_I102_3,
    B04 => I10A_SPARE_I102_4,
    B05 => I10A_SPARE_I102_5,
    B06 => I10A_LH_BDY_CONT_FB_I102_6,
    B07 => I10A_RH_BDY_CONT_FB_I102_7,
    B08 => I10A_SPARE_I103_0,
    B09 => I10A_SPARE_I103_1,
    B10 => I10A_SPARE_I103_2,
    B11 => I10A_SPARE_I103_3,
    B12 => I10A_SPARE_I103_4,
    B13 => I10A_SPARE_I103_5,
    B14 => I10A_SPARE_I103_6,
    B15 => I10A_SPARE_I103_7); // WORD_AS_BIT

// NETWORK 2
BIT_AS_WORD_0(
    B00 := O10A_HPR_MTR_FWD_Q100_0,
    B01 := O10A_HPR_RST_Q100_1,
    B02 := O10A_EXT_SPEED_Q100_2,
    B03 := O10A_SPARE_Q100_3,
    B04 := O10A_HPR_DOOR_SELCTN_IND_Q100_4,
    B05 := O10A_HPR_TWR_LMP_RED_Q100_5,
    B06 := O10A_HPR_TWR_LMP_GREEN_Q100_6,
    B07 := O10A_SPARE_Q100_7,
    B08 := O10A_BDY_BOWL_ON_Q101_0,
    B09 := O10A_BDY_LNR_FEED1_ON_Q101_1,
    B10 := O10A_BDY_LNR_FEED2_ON_Q101_2,
    B11 := O10A_BDY_LNR1_AIR_PURGE_Q101_3,
    B12 := O10A_BDY_LNR2_AIR_PURGE_Q101_4,
    B13 := O10A_HPR_DOOR_OPN_Q101_5,
    B14 := O10A_SPARE_Q101_6,
    B15 := O10A_SPARE_Q101_7,
    W => OP10A_BOWL_FEEDER_JB_16DO_MODULE_1); // BIT_AS_WORD
BIT_AS_WORD_1(
    B00 := O10A_SPARE_Q102_0,
    B01 := O10A_SPARE_Q102_1,
    B02 := O10A_SPARE_Q102_2,
    B03 := O10A_SPARE_Q102_3,
    B04 := O10A_SPARE_Q102_4,
    B05 := O10A_SPARE_Q102_5,
    B06 := O10A_SPARE_Q102_6,
    B07 := O10A_SPARE_Q102_7,
    B08 := O10A_SPARE_Q103_0,
    B09 := O10A_SPARE_Q103_1,
    B10 := O10A_SPARE_Q103_2,
    B11 := O10A_SPARE_Q103_3,
    B12 := O10A_SPARE_Q103_4,
    B13 := O10A_SPARE_Q103_5,
    B14 := O10A_SPARE_Q103_6,
    B15 := O10A_SPARE_Q103_7,
    W => OP10A_BOWL_FEEDER_JB_16DO_MODULE_2); // BIT_AS_WORD

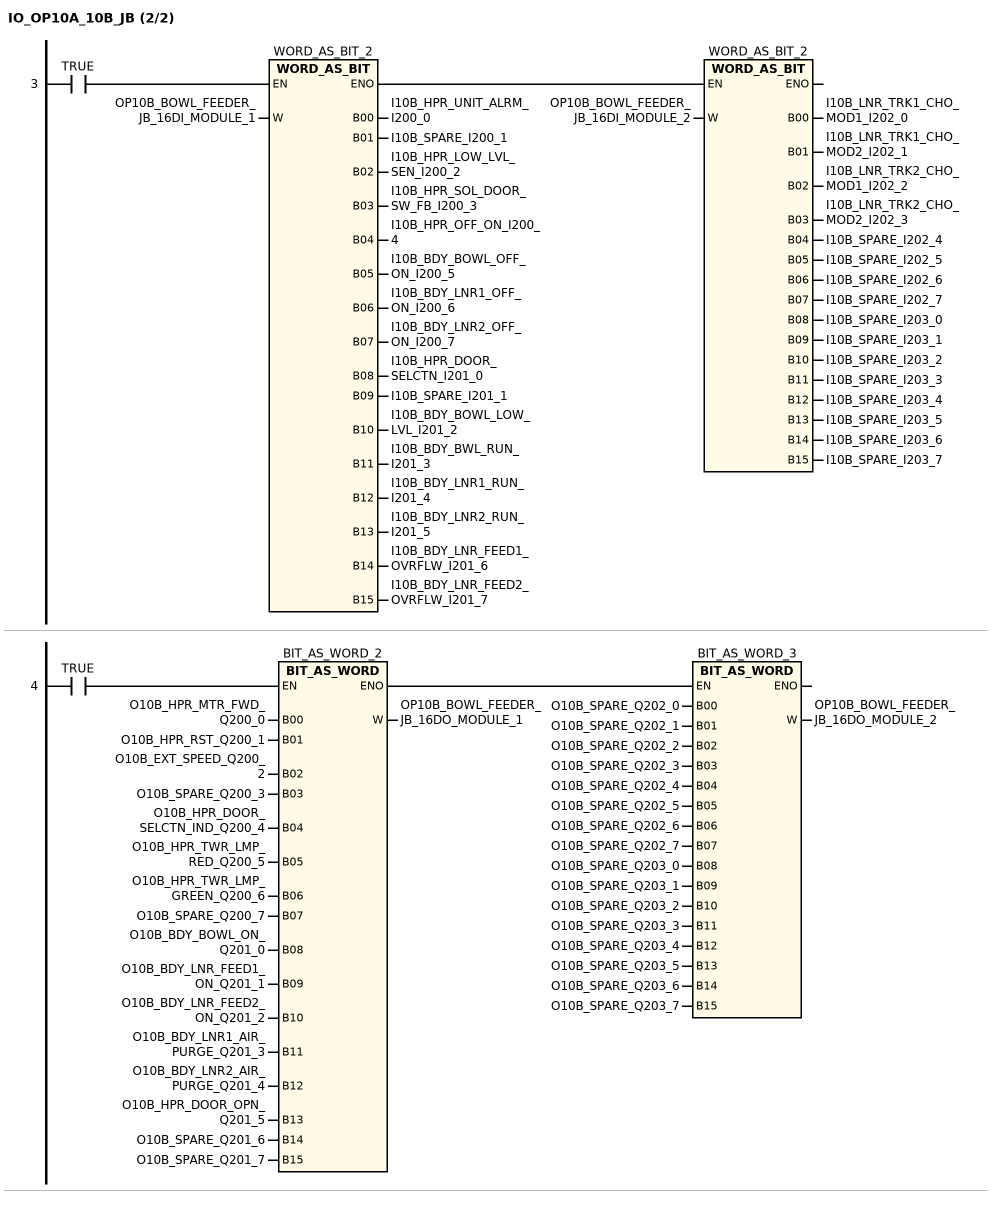
// NETWORK 3
WORD_AS_BIT_2(
    W := OP10B_BOWL_FEEDER_JB_16DI_MODULE_1,
    B00 => I10B_HPR_UNIT_ALRM_I200_0,
    B01 => I10B_SPARE_I200_1,
    B02 => I10B_HPR_LOW_LVL_SEN_I200_2,
    B03 => I10B_HPR_SOL_DOOR_SW_FB_I200_3,
    B04 => I10B_HPR_OFF_ON_I200_4,
    B05 => I10B_BDY_BOWL_OFF_ON_I200_5,
    B06 => I10B_BDY_LNR1_OFF_ON_I200_6,
    B07 => I10B_BDY_LNR2_OFF_ON_I200_7,
    B08 => I10B_HPR_DOOR_SELCTN_I201_0,
    B09 => I10B_SPARE_I201_1,
    B10 => I10B_BDY_BOWL_LOW_LVL_I201_2,
    B11 => I10B_BDY_BWL_RUN_I201_3,
    B12 => I10B_BDY_LNR1_RUN_I201_4,
    B13 => I10B_BDY_LNR2_RUN_I201_5,
    B14 => I10B_BDY_LNR_FEED1_OVRFLW_I201_6,
    B15 => I10B_BDY_LNR_FEED2_OVRFLW_I201_7); // WORD_AS_BIT
WORD_AS_BIT_2(
    W := OP10B_BOWL_FEEDER_JB_16DI_MODULE_2,
    B00 => I10B_LNR_TRK1_CHO_MOD1_I202_0,
    B01 => I10B_LNR_TRK1_CHO_MOD2_I202_1,
    B02 => I10B_LNR_TRK2_CHO_MOD1_I202_2,
    B03 => I10B_LNR_TRK2_CHO_MOD2_I202_3,
    B04 => I10B_SPARE_I202_4,
    B05 => I10B_SPARE_I202_5,
    B06 => I10B_SPARE_I202_6,
    B07 => I10B_SPARE_I202_7,
    B08 => I10B_SPARE_I203_0,
    B09 => I10B_SPARE_I203_1,
    B10 => I10B_SPARE_I203_2,
    B11 => I10B_SPARE_I203_3,
    B12 => I10B_SPARE_I203_4,
    B13 => I10B_SPARE_I203_5,
    B14 => I10B_SPARE_I203_6,
    B15 => I10B_SPARE_I203_7); // WORD_AS_BIT

// NETWORK 4
BIT_AS_WORD_2(
    B00 := O10B_HPR_MTR_FWD_Q200_0,
    B01 := O10B_HPR_RST_Q200_1,
    B02 := O10B_EXT_SPEED_Q200_2,
    B03 := O10B_SPARE_Q200_3,
    B04 := O10B_HPR_DOOR_SELCTN_IND_Q200_4,
    B05 := O10B_HPR_TWR_LMP_RED_Q200_5,
    B06 := O10B_HPR_TWR_LMP_GREEN_Q200_6,
    B07 := O10B_SPARE_Q200_7,
    B08 := O10B_BDY_BOWL_ON_Q201_0,
    B09 := O10B_BDY_LNR_FEED1_ON_Q201_1,
    B10 := O10B_BDY_LNR_FEED2_ON_Q201_2,
    B11 := O10B_BDY_LNR1_AIR_PURGE_Q201_3,
    B12 := O10B_BDY_LNR2_AIR_PURGE_Q201_4,
    B13 := O10B_HPR_DOOR_OPN_Q201_5,
    B14 := O10B_SPARE_Q201_6,
    B15 := O10B_SPARE_Q201_7,
    W => OP10B_BOWL_FEEDER_JB_16DO_MODULE_1); // BIT_AS_WORD
BIT_AS_WORD_3(
    B00 := O10B_SPARE_Q202_0,
    B01 := O10B_SPARE_Q202_1,
    B02 := O10B_SPARE_Q202_2,
    B03 := O10B_SPARE_Q202_3,
    B04 := O10B_SPARE_Q202_4,
    B05 := O10B_SPARE_Q202_5,
    B06 := O10B_SPARE_Q202_6,
    B07 := O10B_SPARE_Q202_7,
    B08 := O10B_SPARE_Q203_0,
    B09 := O10B_SPARE_Q203_1,
    B10 := O10B_SPARE_Q203_2,
    B11 := O10B_SPARE_Q203_3,
    B12 := O10B_SPARE_Q203_4,
    B13 := O10B_SPARE_Q203_5,
    B14 := O10B_SPARE_Q203_6,
    B15 := O10B_SPARE_Q203_7,
    W => OP10B_BOWL_FEEDER_JB_16DO_MODULE_2); // BIT_AS_WORD

END_PROGRAM

// ---- POUs/OP10_Profinet_IO/Master1_IO_Map.TcPOU
PROGRAM Master1_IO_Map
VAR
	BYTE_AS_BIT_0: BYTE_AS_BIT;
	BYTE_AS_BIT_1: BYTE_AS_BIT;
	BYTE_AS_BIT_2: BYTE_AS_BIT;
	BYTE_AS_BIT_3: BYTE_AS_BIT;
	BYTE_AS_BIT_4: BYTE_AS_BIT;
	BYTE_AS_BIT_5: BYTE_AS_BIT;
	BYTE_AS_BIT_6: BYTE_AS_BIT;
	BYTE_AS_BIT_7: BYTE_AS_BIT;
	BYTE_AS_BIT_8: BYTE_AS_BIT;
	BYTE_AS_BIT_9: BYTE_AS_BIT;
	
	BIT_AS_BYTE_0: BIT_AS_BYTE;
	BIT_AS_BYTE_1: BIT_AS_BYTE;
	BIT_AS_BYTE_2: BIT_AS_BYTE;
	BIT_AS_BYTE_3: BIT_AS_BYTE;
	BIT_AS_BYTE_4: BIT_AS_BYTE;
	BIT_AS_BYTE_5: BIT_AS_BYTE;
	BIT_AS_BYTE_6: BIT_AS_BYTE;
	BIT_AS_BYTE_7: BIT_AS_BYTE;
	BIT_AS_BYTE_8: BIT_AS_BYTE;
	BIT_AS_BYTE_9: BIT_AS_BYTE;
	BIT_AS_BYTE_10: BIT_AS_BYTE;
	BIT_AS_BYTE_11: BIT_AS_BYTE;	
	
	OP10_MAS1_PORT1_BYTE1_DI_MODULE_1 AT %I* : BYTE;
	OP10_MAS1_PORT1_BYTE2_DI_MODULE_1 AT %I* : BYTE;
	OP10_MAS1_PORT2_BYTE1_DI_MODULE_2 AT %I* : BYTE;
	OP10_MAS1_PORT2_BYTE2_DI_MODULE_2 AT %I* : BYTE;
	OP10_MAS1_PORT3_BYTE1_DI_MODULE_3 AT %I* : BYTE;
	OP10_MAS1_PORT3_BYTE2_DI_MODULE_3 AT %I* : BYTE;
	OP10_MAS1_PORT4_BYTE1_DI_MODULE_4 AT %I* : BYTE;
	OP10_MAS1_PORT4_BYTE2_DI_MODULE_4 AT %I* : BYTE;
	OP10_MAS1_PORT5_BYTE1_DI_MODULE_5 AT %I* : BYTE;
	OP10_MAS1_PORT5_BYTE2_DI_MODULE_5 AT %I* : BYTE;
	
	OP10_MAS1_PORT6_BYTE1_DO_MODULE_1 AT %Q* : BYTE;
	OP10_MAS1_PORT6_BYTE2_DO_MODULE_1 AT %Q* : BYTE;
    OP10_MAS1_PORT6_BYTE3_DO_MODULE_1 AT %Q* : BYTE;
	OP10_MAS1_PORT6_BYTE4_DO_MODULE_1 AT %Q* : BYTE;
	
	OP10_MAS1_PORT7_BYTE1_DO_MODULE_2 AT %Q* : BYTE;
	OP10_MAS1_PORT7_BYTE2_DO_MODULE_2 AT %Q* : BYTE;
	OP10_MAS1_PORT7_BYTE3_DO_MODULE_2 AT %Q* : BYTE;
	OP10_MAS1_PORT7_BYTE4_DO_MODULE_2 AT %Q* : BYTE;
	
	OP10_MAS1_PORT8_BYTE1_DO_MODULE_3 AT %Q* : BYTE;
	OP10_MAS1_PORT8_BYTE2_DO_MODULE_3 AT %Q* : BYTE;
    OP10_MAS1_PORT8_BYTE3_DO_MODULE_3 AT %Q* : BYTE;
	OP10_MAS1_PORT8_BYTE4_DO_MODULE_3 AT %Q* : BYTE;

END_VAR

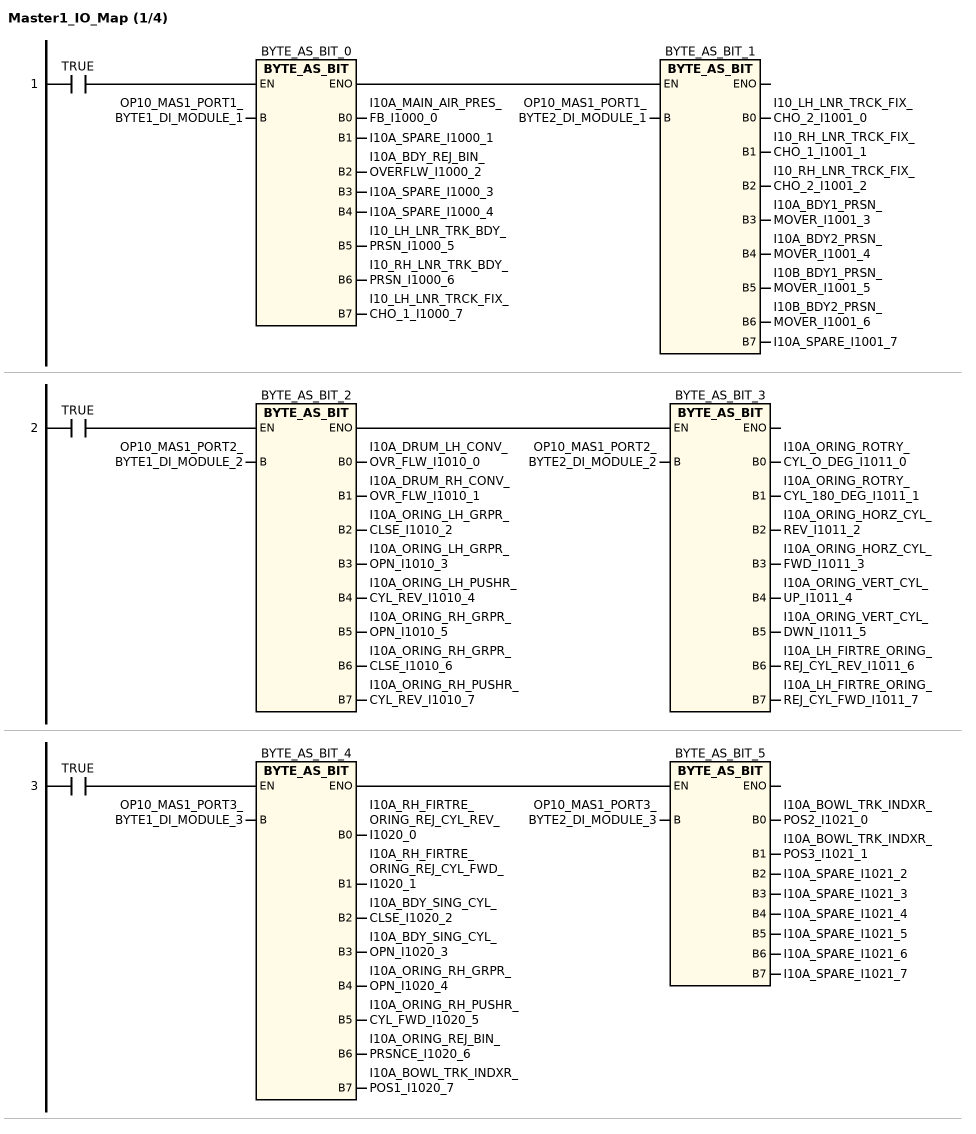
// NETWORK 1
BYTE_AS_BIT_0(
    B := OP10_MAS1_PORT1_BYTE1_DI_MODULE_1,
    B0 => I10A_MAIN_AIR_PRES_FB_I1000_0,
    B1 => I10A_SPARE_I1000_1,
    B2 => I10A_BDY_REJ_BIN_OVERFLW_I1000_2,
    B3 => I10A_SPARE_I1000_3,
    B4 => I10A_SPARE_I1000_4,
    B5 => I10_LH_LNR_TRK_BDY_PRSN_I1000_5,
    B6 => I10_RH_LNR_TRK_BDY_PRSN_I1000_6,
    B7 => I10_LH_LNR_TRCK_FIX_CHO_1_I1000_7); // BYTE_AS_BIT
BYTE_AS_BIT_1(
    B := OP10_MAS1_PORT1_BYTE2_DI_MODULE_1,
    B0 => I10_LH_LNR_TRCK_FIX_CHO_2_I1001_0,
    B1 => I10_RH_LNR_TRCK_FIX_CHO_1_I1001_1,
    B2 => I10_RH_LNR_TRCK_FIX_CHO_2_I1001_2,
    B3 => I10A_BDY1_PRSN_MOVER_I1001_3,
    B4 => I10A_BDY2_PRSN_MOVER_I1001_4,
    B5 => I10B_BDY1_PRSN_MOVER_I1001_5,
    B6 => I10B_BDY2_PRSN_MOVER_I1001_6,
    B7 => I10A_SPARE_I1001_7); // BYTE_AS_BIT

// NETWORK 2
BYTE_AS_BIT_2(
    B := OP10_MAS1_PORT2_BYTE1_DI_MODULE_2,
    B0 => I10A_DRUM_LH_CONV_OVR_FLW_I1010_0,
    B1 => I10A_DRUM_RH_CONV_OVR_FLW_I1010_1,
    B2 => I10A_ORING_LH_GRPR_CLSE_I1010_2,
    B3 => I10A_ORING_LH_GRPR_OPN_I1010_3,
    B4 => I10A_ORING_LH_PUSHR_CYL_REV_I1010_4,
    B5 => I10A_ORING_RH_GRPR_OPN_I1010_5,
    B6 => I10A_ORING_RH_GRPR_CLSE_I1010_6,
    B7 => I10A_ORING_RH_PUSHR_CYL_REV_I1010_7); // BYTE_AS_BIT
BYTE_AS_BIT_3(
    B := OP10_MAS1_PORT2_BYTE2_DI_MODULE_2,
    B0 => I10A_ORING_ROTRY_CYL_O_DEG_I1011_0,
    B1 => I10A_ORING_ROTRY_CYL_180_DEG_I1011_1,
    B2 => I10A_ORING_HORZ_CYL_REV_I1011_2,
    B3 => I10A_ORING_HORZ_CYL_FWD_I1011_3,
    B4 => I10A_ORING_VERT_CYL_UP_I1011_4,
    B5 => I10A_ORING_VERT_CYL_DWN_I1011_5,
    B6 => I10A_LH_FIRTRE_ORING_REJ_CYL_REV_I1011_6,
    B7 => I10A_LH_FIRTRE_ORING_REJ_CYL_FWD_I1011_7); // BYTE_AS_BIT

// NETWORK 3
BYTE_AS_BIT_4(
    B := OP10_MAS1_PORT3_BYTE1_DI_MODULE_3,
    B0 => I10A_RH_FIRTRE_ORING_REJ_CYL_REV_I1020_0,
    B1 => I10A_RH_FIRTRE_ORING_REJ_CYL_FWD_I1020_1,
    B2 => I10A_BDY_SING_CYL_CLSE_I1020_2,
    B3 => I10A_BDY_SING_CYL_OPN_I1020_3,
    B4 => I10A_ORING_RH_GRPR_OPN_I1020_4,
    B5 => I10A_ORING_RH_PUSHR_CYL_FWD_I1020_5,
    B6 => I10A_ORING_REJ_BIN_PRSNCE_I1020_6,
    B7 => I10A_BOWL_TRK_INDXR_POS1_I1020_7); // BYTE_AS_BIT
BYTE_AS_BIT_5(
    B := OP10_MAS1_PORT3_BYTE2_DI_MODULE_3,
    B0 => I10A_BOWL_TRK_INDXR_POS2_I1021_0,
    B1 => I10A_BOWL_TRK_INDXR_POS3_I1021_1,
    B2 => I10A_SPARE_I1021_2,
    B3 => I10A_SPARE_I1021_3,
    B4 => I10A_SPARE_I1021_4,
    B5 => I10A_SPARE_I1021_5,
    B6 => I10A_SPARE_I1021_6,
    B7 => I10A_SPARE_I1021_7); // BYTE_AS_BIT

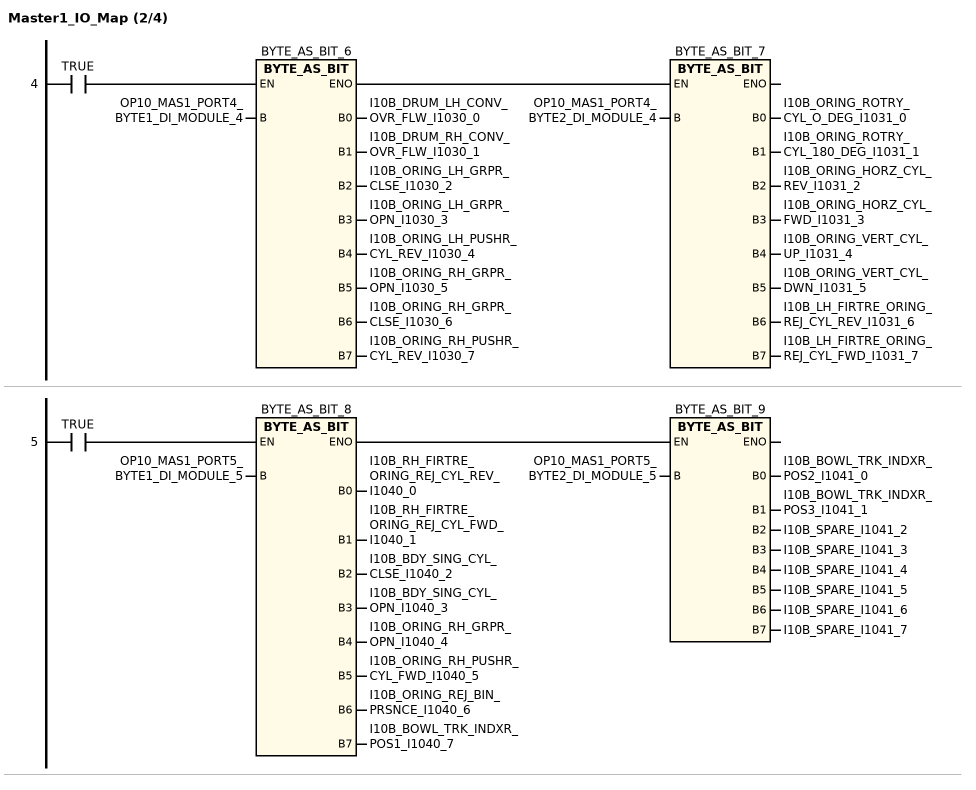
// NETWORK 4
BYTE_AS_BIT_6(
    B := OP10_MAS1_PORT4_BYTE1_DI_MODULE_4,
    B0 => I10B_DRUM_LH_CONV_OVR_FLW_I1030_0,
    B1 => I10B_DRUM_RH_CONV_OVR_FLW_I1030_1,
    B2 => I10B_ORING_LH_GRPR_CLSE_I1030_2,
    B3 => I10B_ORING_LH_GRPR_OPN_I1030_3,
    B4 => I10B_ORING_LH_PUSHR_CYL_REV_I1030_4,
    B5 => I10B_ORING_RH_GRPR_OPN_I1030_5,
    B6 => I10B_ORING_RH_GRPR_CLSE_I1030_6,
    B7 => I10B_ORING_RH_PUSHR_CYL_REV_I1030_7); // BYTE_AS_BIT
BYTE_AS_BIT_7(
    B := OP10_MAS1_PORT4_BYTE2_DI_MODULE_4,
    B0 => I10B_ORING_ROTRY_CYL_O_DEG_I1031_0,
    B1 => I10B_ORING_ROTRY_CYL_180_DEG_I1031_1,
    B2 => I10B_ORING_HORZ_CYL_REV_I1031_2,
    B3 => I10B_ORING_HORZ_CYL_FWD_I1031_3,
    B4 => I10B_ORING_VERT_CYL_UP_I1031_4,
    B5 => I10B_ORING_VERT_CYL_DWN_I1031_5,
    B6 => I10B_LH_FIRTRE_ORING_REJ_CYL_REV_I1031_6,
    B7 => I10B_LH_FIRTRE_ORING_REJ_CYL_FWD_I1031_7); // BYTE_AS_BIT

// NETWORK 5
BYTE_AS_BIT_8(
    B := OP10_MAS1_PORT5_BYTE1_DI_MODULE_5,
    B0 => I10B_RH_FIRTRE_ORING_REJ_CYL_REV_I1040_0,
    B1 => I10B_RH_FIRTRE_ORING_REJ_CYL_FWD_I1040_1,
    B2 => I10B_BDY_SING_CYL_CLSE_I1040_2,
    B3 => I10B_BDY_SING_CYL_OPN_I1040_3,
    B4 => I10B_ORING_RH_GRPR_OPN_I1040_4,
    B5 => I10B_ORING_RH_PUSHR_CYL_FWD_I1040_5,
    B6 => I10B_ORING_REJ_BIN_PRSNCE_I1040_6,
    B7 => I10B_BOWL_TRK_INDXR_POS1_I1040_7); // BYTE_AS_BIT
BYTE_AS_BIT_9(
    B := OP10_MAS1_PORT5_BYTE2_DI_MODULE_5,
    B0 => I10B_BOWL_TRK_INDXR_POS2_I1041_0,
    B1 => I10B_BOWL_TRK_INDXR_POS3_I1041_1,
    B2 => I10B_SPARE_I1041_2,
    B3 => I10B_SPARE_I1041_3,
    B4 => I10B_SPARE_I1041_4,
    B5 => I10B_SPARE_I1041_5,
    B6 => I10B_SPARE_I1041_6,
    B7 => I10B_SPARE_I1041_7); // BYTE_AS_BIT

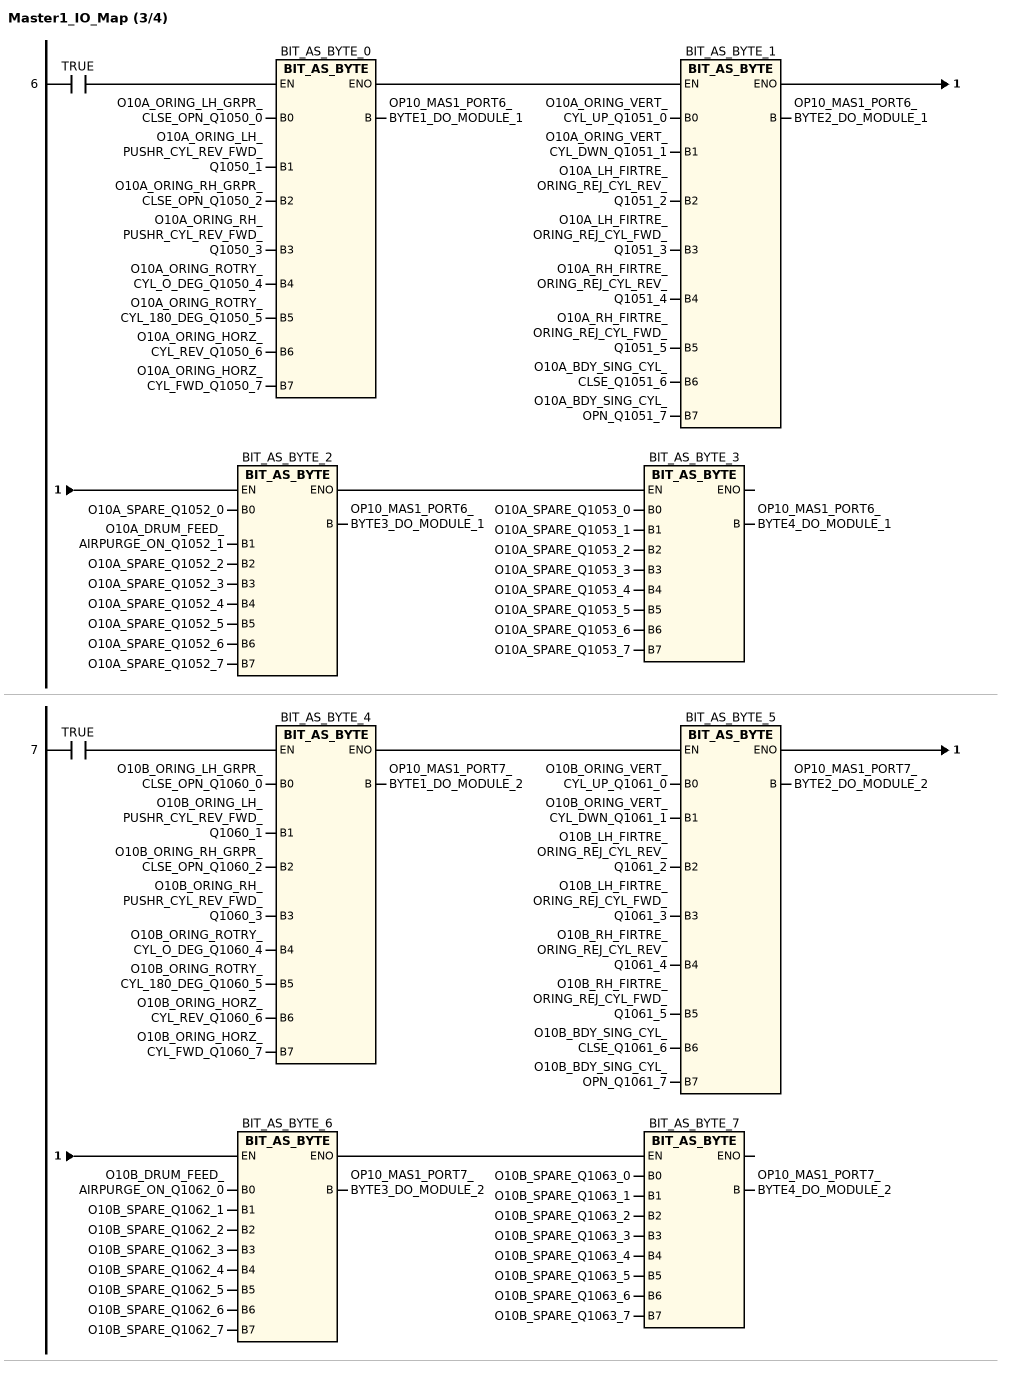
// NETWORK 6
BIT_AS_BYTE_0(
    B0 := O10A_ORING_LH_GRPR_CLSE_OPN_Q1050_0,
    B1 := O10A_ORING_LH_PUSHR_CYL_REV_FWD_Q1050_1,
    B2 := O10A_ORING_RH_GRPR_CLSE_OPN_Q1050_2,
    B3 := O10A_ORING_RH_PUSHR_CYL_REV_FWD_Q1050_3,
    B4 := O10A_ORING_ROTRY_CYL_O_DEG_Q1050_4,
    B5 := O10A_ORING_ROTRY_CYL_180_DEG_Q1050_5,
    B6 := O10A_ORING_HORZ_CYL_REV_Q1050_6,
    B7 := O10A_ORING_HORZ_CYL_FWD_Q1050_7,
    B => OP10_MAS1_PORT6_BYTE1_DO_MODULE_1); // BIT_AS_BYTE
BIT_AS_BYTE_1(
    B0 := O10A_ORING_VERT_CYL_UP_Q1051_0,
    B1 := O10A_ORING_VERT_CYL_DWN_Q1051_1,
    B2 := O10A_LH_FIRTRE_ORING_REJ_CYL_REV_Q1051_2,
    B3 := O10A_LH_FIRTRE_ORING_REJ_CYL_FWD_Q1051_3,
    B4 := O10A_RH_FIRTRE_ORING_REJ_CYL_REV_Q1051_4,
    B5 := O10A_RH_FIRTRE_ORING_REJ_CYL_FWD_Q1051_5,
    B6 := O10A_BDY_SING_CYL_CLSE_Q1051_6,
    B7 := O10A_BDY_SING_CYL_OPN_Q1051_7,
    B => OP10_MAS1_PORT6_BYTE2_DO_MODULE_1); // BIT_AS_BYTE
BIT_AS_BYTE_2(
    B0 := O10A_SPARE_Q1052_0,
    B1 := O10A_DRUM_FEED_AIRPURGE_ON_Q1052_1,
    B2 := O10A_SPARE_Q1052_2,
    B3 := O10A_SPARE_Q1052_3,
    B4 := O10A_SPARE_Q1052_4,
    B5 := O10A_SPARE_Q1052_5,
    B6 := O10A_SPARE_Q1052_6,
    B7 := O10A_SPARE_Q1052_7,
    B => OP10_MAS1_PORT6_BYTE3_DO_MODULE_1); // BIT_AS_BYTE
BIT_AS_BYTE_3(
    B0 := O10A_SPARE_Q1053_0,
    B1 := O10A_SPARE_Q1053_1,
    B2 := O10A_SPARE_Q1053_2,
    B3 := O10A_SPARE_Q1053_3,
    B4 := O10A_SPARE_Q1053_4,
    B5 := O10A_SPARE_Q1053_5,
    B6 := O10A_SPARE_Q1053_6,
    B7 := O10A_SPARE_Q1053_7,
    B => OP10_MAS1_PORT6_BYTE4_DO_MODULE_1); // BIT_AS_BYTE

// NETWORK 7
BIT_AS_BYTE_4(
    B0 := O10B_ORING_LH_GRPR_CLSE_OPN_Q1060_0,
    B1 := O10B_ORING_LH_PUSHR_CYL_REV_FWD_Q1060_1,
    B2 := O10B_ORING_RH_GRPR_CLSE_OPN_Q1060_2,
    B3 := O10B_ORING_RH_PUSHR_CYL_REV_FWD_Q1060_3,
    B4 := O10B_ORING_ROTRY_CYL_O_DEG_Q1060_4,
    B5 := O10B_ORING_ROTRY_CYL_180_DEG_Q1060_5,
    B6 := O10B_ORING_HORZ_CYL_REV_Q1060_6,
    B7 := O10B_ORING_HORZ_CYL_FWD_Q1060_7,
    B => OP10_MAS1_PORT7_BYTE1_DO_MODULE_2); // BIT_AS_BYTE
BIT_AS_BYTE_5(
    B0 := O10B_ORING_VERT_CYL_UP_Q1061_0,
    B1 := O10B_ORING_VERT_CYL_DWN_Q1061_1,
    B2 := O10B_LH_FIRTRE_ORING_REJ_CYL_REV_Q1061_2,
    B3 := O10B_LH_FIRTRE_ORING_REJ_CYL_FWD_Q1061_3,
    B4 := O10B_RH_FIRTRE_ORING_REJ_CYL_REV_Q1061_4,
    B5 := O10B_RH_FIRTRE_ORING_REJ_CYL_FWD_Q1061_5,
    B6 := O10B_BDY_SING_CYL_CLSE_Q1061_6,
    B7 := O10B_BDY_SING_CYL_OPN_Q1061_7,
    B => OP10_MAS1_PORT7_BYTE2_DO_MODULE_2); // BIT_AS_BYTE
BIT_AS_BYTE_6(
    B0 := O10B_DRUM_FEED_AIRPURGE_ON_Q1062_0,
    B1 := O10B_SPARE_Q1062_1,
    B2 := O10B_SPARE_Q1062_2,
    B3 := O10B_SPARE_Q1062_3,
    B4 := O10B_SPARE_Q1062_4,
    B5 := O10B_SPARE_Q1062_5,
    B6 := O10B_SPARE_Q1062_6,
    B7 := O10B_SPARE_Q1062_7,
    B => OP10_MAS1_PORT7_BYTE3_DO_MODULE_2); // BIT_AS_BYTE
BIT_AS_BYTE_7(
    B0 := O10B_SPARE_Q1063_0,
    B1 := O10B_SPARE_Q1063_1,
    B2 := O10B_SPARE_Q1063_2,
    B3 := O10B_SPARE_Q1063_3,
    B4 := O10B_SPARE_Q1063_4,
    B5 := O10B_SPARE_Q1063_5,
    B6 := O10B_SPARE_Q1063_6,
    B7 := O10B_SPARE_Q1063_7,
    B => OP10_MAS1_PORT7_BYTE4_DO_MODULE_2); // BIT_AS_BYTE

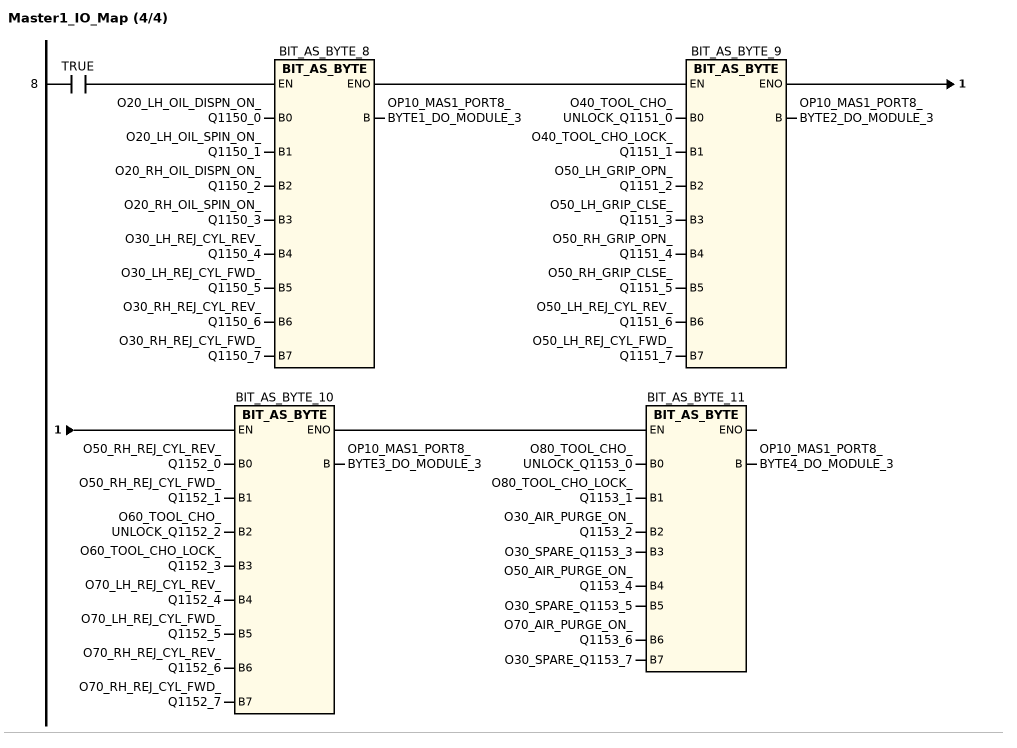
// NETWORK 8
BIT_AS_BYTE_8(
    B0 := O20_LH_OIL_DISPN_ON_Q1150_0,
    B1 := O20_LH_OIL_SPIN_ON_Q1150_1,
    B2 := O20_RH_OIL_DISPN_ON_Q1150_2,
    B3 := O20_RH_OIL_SPIN_ON_Q1150_3,
    B4 := O30_LH_REJ_CYL_REV_Q1150_4,
    B5 := O30_LH_REJ_CYL_FWD_Q1150_5,
    B6 := O30_RH_REJ_CYL_REV_Q1150_6,
    B7 := O30_RH_REJ_CYL_FWD_Q1150_7,
    B => OP10_MAS1_PORT8_BYTE1_DO_MODULE_3); // BIT_AS_BYTE
BIT_AS_BYTE_9(
    B0 := O40_TOOL_CHO_UNLOCK_Q1151_0,
    B1 := O40_TOOL_CHO_LOCK_Q1151_1,
    B2 := O50_LH_GRIP_OPN_Q1151_2,
    B3 := O50_LH_GRIP_CLSE_Q1151_3,
    B4 := O50_RH_GRIP_OPN_Q1151_4,
    B5 := O50_RH_GRIP_CLSE_Q1151_5,
    B6 := O50_LH_REJ_CYL_REV_Q1151_6,
    B7 := O50_LH_REJ_CYL_FWD_Q1151_7,
    B => OP10_MAS1_PORT8_BYTE2_DO_MODULE_3); // BIT_AS_BYTE
BIT_AS_BYTE_10(
    B0 := O50_RH_REJ_CYL_REV_Q1152_0,
    B1 := O50_RH_REJ_CYL_FWD_Q1152_1,
    B2 := O60_TOOL_CHO_UNLOCK_Q1152_2,
    B3 := O60_TOOL_CHO_LOCK_Q1152_3,
    B4 := O70_LH_REJ_CYL_REV_Q1152_4,
    B5 := O70_LH_REJ_CYL_FWD_Q1152_5,
    B6 := O70_RH_REJ_CYL_REV_Q1152_6,
    B7 := O70_RH_REJ_CYL_FWD_Q1152_7,
    B => OP10_MAS1_PORT8_BYTE3_DO_MODULE_3); // BIT_AS_BYTE
BIT_AS_BYTE_11(
    B0 := O80_TOOL_CHO_UNLOCK_Q1153_0,
    B1 := O80_TOOL_CHO_LOCK_Q1153_1,
    B2 := O30_AIR_PURGE_ON_Q1153_2,
    B3 := O30_SPARE_Q1153_3,
    B4 := O50_AIR_PURGE_ON_Q1153_4,
    B5 := O30_SPARE_Q1153_5,
    B6 := O70_AIR_PURGE_ON_Q1153_6,
    B7 := O30_SPARE_Q1153_7,
    B => OP10_MAS1_PORT8_BYTE4_DO_MODULE_3); // BIT_AS_BYTE

END_PROGRAM

// ---- POUs/OP10_Profinet_IO/MASTER2_IO_Map.TcPOU
PROGRAM MASTER2_IO_Map
VAR
	BYTE_AS_BIT_0: BYTE_AS_BIT;
	BYTE_AS_BIT_1: BYTE_AS_BIT;
	BYTE_AS_BIT_2: BYTE_AS_BIT;
	BYTE_AS_BIT_3: BYTE_AS_BIT;

	BIT_AS_BYTE_0: BIT_AS_BYTE;
	BIT_AS_BYTE_1: BIT_AS_BYTE;
	BIT_AS_BYTE_2: BIT_AS_BYTE;
	BIT_AS_BYTE_3: BIT_AS_BYTE;
	
	OP10_MAS2_PORT1_BYTE1_DI_MODULE_1 AT %I* : BYTE;
	OP10_MAS2_PORT1_BYTE2_DI_MODULE_1 AT %I* : BYTE;
	OP10_MAS2_PORT2_BYTE1_DI_MODULE_2 AT %I* : BYTE;
	OP10_MAS2_PORT2_BYTE2_DI_MODULE_2 AT %I* : BYTE;	

	
END_VAR

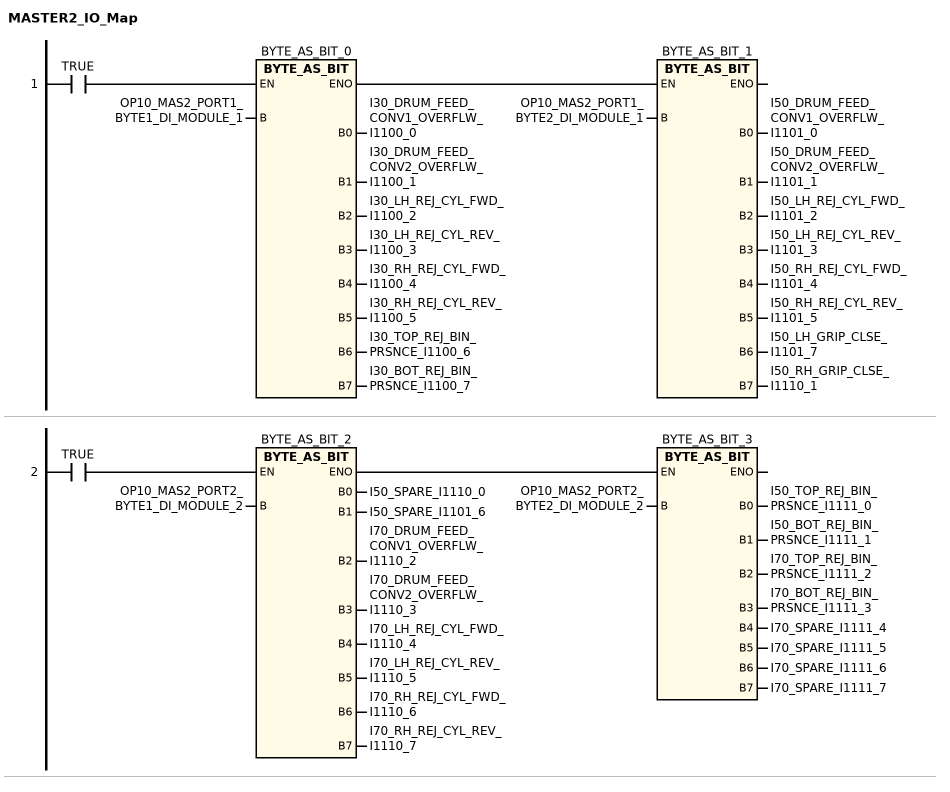
// NETWORK 1
BYTE_AS_BIT_0(
    B := OP10_MAS2_PORT1_BYTE1_DI_MODULE_1,
    B0 => I30_DRUM_FEED_CONV1_OVERFLW_I1100_0,
    B1 => I30_DRUM_FEED_CONV2_OVERFLW_I1100_1,
    B2 => I30_LH_REJ_CYL_FWD_I1100_2,
    B3 => I30_LH_REJ_CYL_REV_I1100_3,
    B4 => I30_RH_REJ_CYL_FWD_I1100_4,
    B5 => I30_RH_REJ_CYL_REV_I1100_5,
    B6 => I30_TOP_REJ_BIN_PRSNCE_I1100_6,
    B7 => I30_BOT_REJ_BIN_PRSNCE_I1100_7); // BYTE_AS_BIT
BYTE_AS_BIT_1(
    B := OP10_MAS2_PORT1_BYTE2_DI_MODULE_1,
    B0 => I50_DRUM_FEED_CONV1_OVERFLW_I1101_0,
    B1 => I50_DRUM_FEED_CONV2_OVERFLW_I1101_1,
    B2 => I50_LH_REJ_CYL_FWD_I1101_2,
    B3 => I50_LH_REJ_CYL_REV_I1101_3,
    B4 => I50_RH_REJ_CYL_FWD_I1101_4,
    B5 => I50_RH_REJ_CYL_REV_I1101_5,
    B6 => I50_LH_GRIP_CLSE_I1101_7,
    B7 => I50_RH_GRIP_CLSE_I1110_1); // BYTE_AS_BIT

// NETWORK 2
BYTE_AS_BIT_2(
    B := OP10_MAS2_PORT2_BYTE1_DI_MODULE_2,
    B0 => I50_SPARE_I1110_0,
    B1 => I50_SPARE_I1101_6,
    B2 => I70_DRUM_FEED_CONV1_OVERFLW_I1110_2,
    B3 => I70_DRUM_FEED_CONV2_OVERFLW_I1110_3,
    B4 => I70_LH_REJ_CYL_FWD_I1110_4,
    B5 => I70_LH_REJ_CYL_REV_I1110_5,
    B6 => I70_RH_REJ_CYL_FWD_I1110_6,
    B7 => I70_RH_REJ_CYL_REV_I1110_7); // BYTE_AS_BIT
BYTE_AS_BIT_3(
    B := OP10_MAS2_PORT2_BYTE2_DI_MODULE_2,
    B0 => I50_TOP_REJ_BIN_PRSNCE_I1111_0,
    B1 => I50_BOT_REJ_BIN_PRSNCE_I1111_1,
    B2 => I70_TOP_REJ_BIN_PRSNCE_I1111_2,
    B3 => I70_BOT_REJ_BIN_PRSNCE_I1111_3,
    B4 => I70_SPARE_I1111_4,
    B5 => I70_SPARE_I1111_5,
    B6 => I70_SPARE_I1111_6,
    B7 => I70_SPARE_I1111_7); // BYTE_AS_BIT

END_PROGRAM

// ---- POUs/IO/OP90_MP_IO.TcPOU
PROGRAM OP90_MP_IO
VAR
	OP90_MP_DI_MODULE_1 AT %I* : WORD;
	OP90_MP_DI_MODULE_2 AT %I* : WORD;
	OP90_MP_DI_MODULE_3 AT %I* : WORD;
	
	OP90_MP_DO_MODULE_1 AT %Q* : WORD;
	OP90_MP_DO_MODULE_2 AT %Q* : WORD;
	
	WORD_AS_BIT_0: WORD_AS_BIT;
	WORD_AS_BIT_1: WORD_AS_BIT;
	WORD_AS_BIT_2: WORD_AS_BIT;
	
	BIT_AS_WORD_0: BIT_AS_WORD;
	BIT_AS_WORD_1: BIT_AS_WORD;
END_VAR

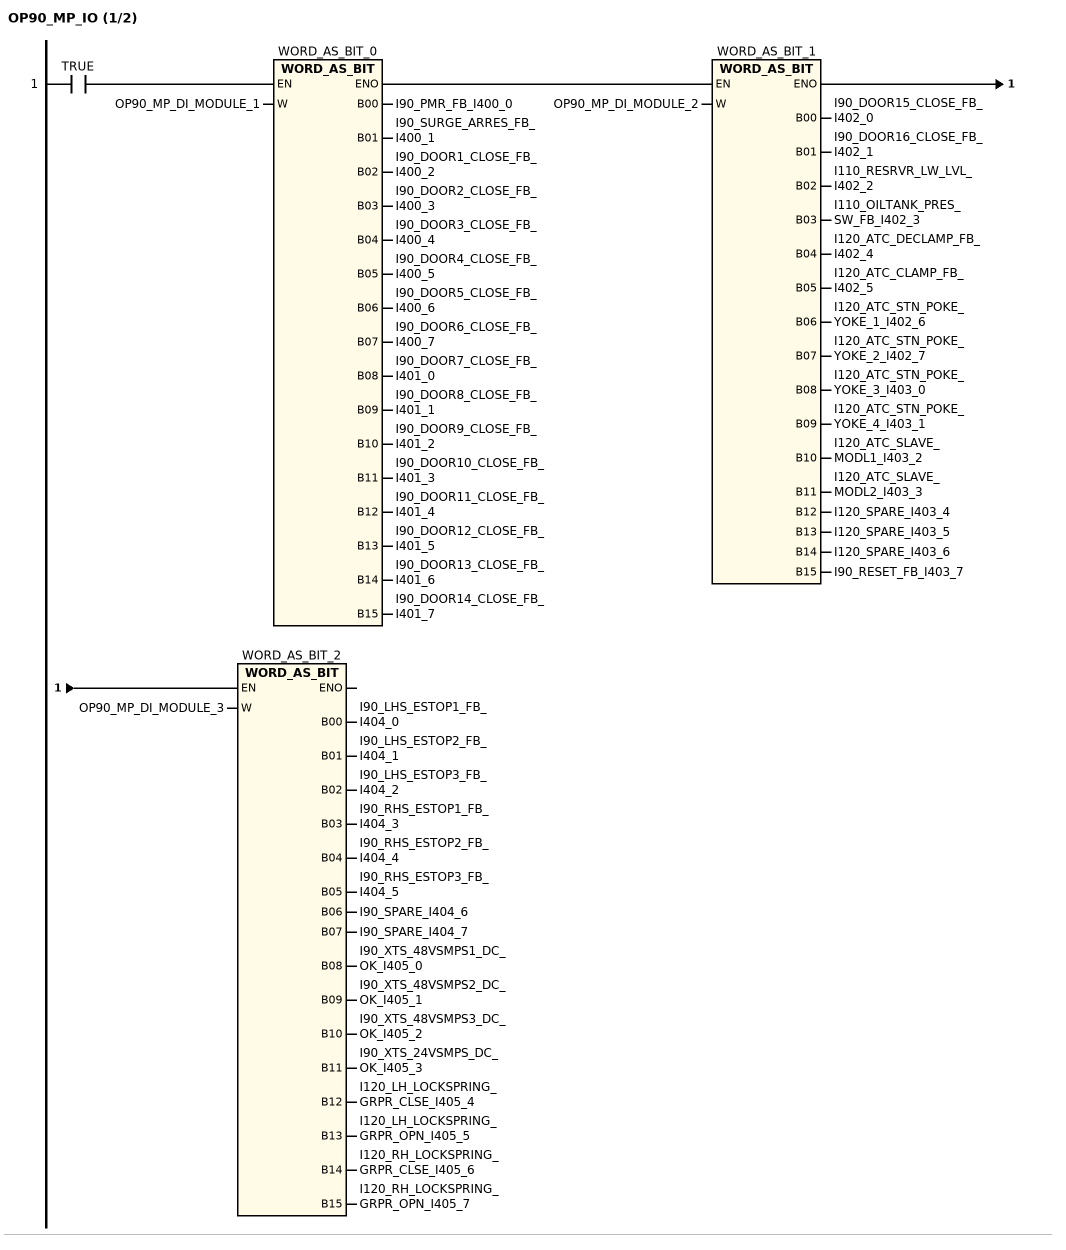
// NETWORK 1
WORD_AS_BIT_0(
    W := OP90_MP_DI_MODULE_1,
    B00 => I90_PMR_FB_I400_0,
    B01 => I90_SURGE_ARRES_FB_I400_1,
    B02 => I90_DOOR1_CLOSE_FB_I400_2,
    B03 => I90_DOOR2_CLOSE_FB_I400_3,
    B04 => I90_DOOR3_CLOSE_FB_I400_4,
    B05 => I90_DOOR4_CLOSE_FB_I400_5,
    B06 => I90_DOOR5_CLOSE_FB_I400_6,
    B07 => I90_DOOR6_CLOSE_FB_I400_7,
    B08 => I90_DOOR7_CLOSE_FB_I401_0,
    B09 => I90_DOOR8_CLOSE_FB_I401_1,
    B10 => I90_DOOR9_CLOSE_FB_I401_2,
    B11 => I90_DOOR10_CLOSE_FB_I401_3,
    B12 => I90_DOOR11_CLOSE_FB_I401_4,
    B13 => I90_DOOR12_CLOSE_FB_I401_5,
    B14 => I90_DOOR13_CLOSE_FB_I401_6,
    B15 => I90_DOOR14_CLOSE_FB_I401_7); // WORD_AS_BIT
WORD_AS_BIT_1(
    W := OP90_MP_DI_MODULE_2,
    B00 => I90_DOOR15_CLOSE_FB_I402_0,
    B01 => I90_DOOR16_CLOSE_FB_I402_1,
    B02 => I110_RESRVR_LW_LVL_I402_2,
    B03 => I110_OILTANK_PRES_SW_FB_I402_3,
    B04 => I120_ATC_DECLAMP_FB_I402_4,
    B05 => I120_ATC_CLAMP_FB_I402_5,
    B06 => I120_ATC_STN_POKE_YOKE_1_I402_6,
    B07 => I120_ATC_STN_POKE_YOKE_2_I402_7,
    B08 => I120_ATC_STN_POKE_YOKE_3_I403_0,
    B09 => I120_ATC_STN_POKE_YOKE_4_I403_1,
    B10 => I120_ATC_SLAVE_MODL1_I403_2,
    B11 => I120_ATC_SLAVE_MODL2_I403_3,
    B12 => I120_SPARE_I403_4,
    B13 => I120_SPARE_I403_5,
    B14 => I120_SPARE_I403_6,
    B15 => I90_RESET_FB_I403_7); // WORD_AS_BIT
WORD_AS_BIT_2(
    W := OP90_MP_DI_MODULE_3,
    B00 => I90_LHS_ESTOP1_FB_I404_0,
    B01 => I90_LHS_ESTOP2_FB_I404_1,
    B02 => I90_LHS_ESTOP3_FB_I404_2,
    B03 => I90_RHS_ESTOP1_FB_I404_3,
    B04 => I90_RHS_ESTOP2_FB_I404_4,
    B05 => I90_RHS_ESTOP3_FB_I404_5,
    B06 => I90_SPARE_I404_6,
    B07 => I90_SPARE_I404_7,
    B08 => I90_XTS_48VSMPS1_DC_OK_I405_0,
    B09 => I90_XTS_48VSMPS2_DC_OK_I405_1,
    B10 => I90_XTS_48VSMPS3_DC_OK_I405_2,
    B11 => I90_XTS_24VSMPS_DC_OK_I405_3,
    B12 => I120_LH_LOCKSPRING_GRPR_CLSE_I405_4,
    B13 => I120_LH_LOCKSPRING_GRPR_OPN_I405_5,
    B14 => I120_RH_LOCKSPRING_GRPR_CLSE_I405_6,
    B15 => I120_RH_LOCKSPRING_GRPR_OPN_I405_7); // WORD_AS_BIT

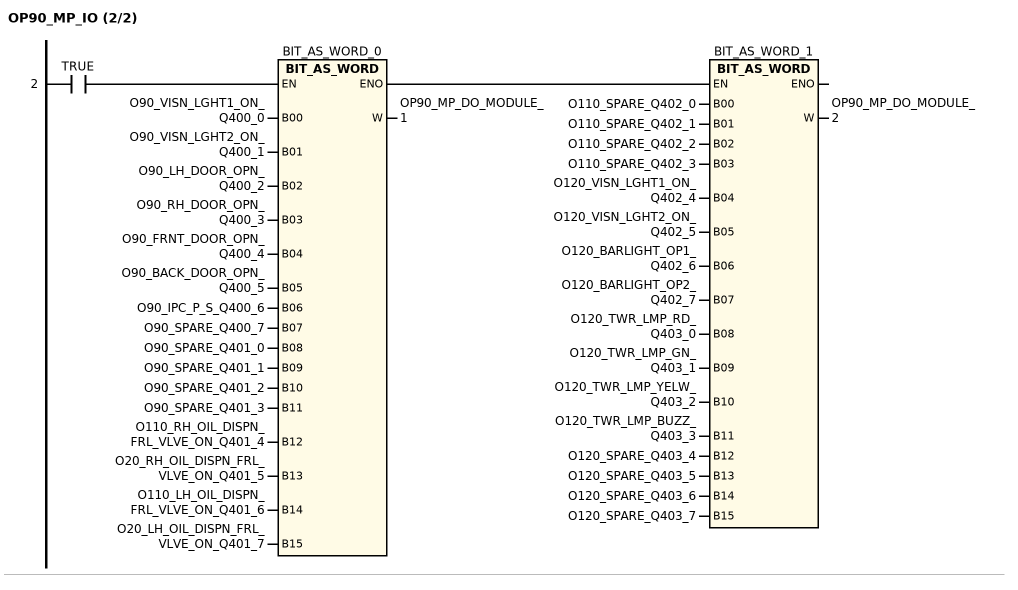
// NETWORK 2
BIT_AS_WORD_0(
    B00 := O90_VISN_LGHT1_ON_Q400_0,
    B01 := O90_VISN_LGHT2_ON_Q400_1,
    B02 := O90_LH_DOOR_OPN_Q400_2,
    B03 := O90_RH_DOOR_OPN_Q400_3,
    B04 := O90_FRNT_DOOR_OPN_Q400_4,
    B05 := O90_BACK_DOOR_OPN_Q400_5,
    B06 := O90_IPC_P_S_Q400_6,
    B07 := O90_SPARE_Q400_7,
    B08 := O90_SPARE_Q401_0,
    B09 := O90_SPARE_Q401_1,
    B10 := O90_SPARE_Q401_2,
    B11 := O90_SPARE_Q401_3,
    B12 := O110_RH_OIL_DISPN_FRL_VLVE_ON_Q401_4,
    B13 := O20_RH_OIL_DISPN_FRL_VLVE_ON_Q401_5,
    B14 := O110_LH_OIL_DISPN_FRL_VLVE_ON_Q401_6,
    B15 := O20_LH_OIL_DISPN_FRL_VLVE_ON_Q401_7,
    W => OP90_MP_DO_MODULE_1); // BIT_AS_WORD
BIT_AS_WORD_1(
    B00 := O110_SPARE_Q402_0,
    B01 := O110_SPARE_Q402_1,
    B02 := O110_SPARE_Q402_2,
    B03 := O110_SPARE_Q402_3,
    B04 := O120_VISN_LGHT1_ON_Q402_4,
    B05 := O120_VISN_LGHT2_ON_Q402_5,
    B06 := O120_BARLIGHT_OP1_Q402_6,
    B07 := O120_BARLIGHT_OP2_Q402_7,
    B08 := O120_TWR_LMP_RD_Q403_0,
    B09 := O120_TWR_LMP_GN_Q403_1,
    B10 := O120_TWR_LMP_YELW_Q403_2,
    B11 := O120_TWR_LMP_BUZZ_Q403_3,
    B12 := O120_SPARE_Q403_4,
    B13 := O120_SPARE_Q403_5,
    B14 := O120_SPARE_Q403_6,
    B15 := O120_SPARE_Q403_7,
    W => OP90_MP_DO_MODULE_2); // BIT_AS_WORD

END_PROGRAM

// ---- POUs/IO/OP90_MASTER3_IO.TcPOU
PROGRAM OP90_MASTER3_IO
VAR
    OP90_MAS3_PORT1_BYTE1_DI_MODULE_1 AT %I* : BYTE;
	OP90_MAS3_PORT1_BYTE2_DI_MODULE_1 AT %I* : BYTE;
	OP90_MAS3_PORT2_BYTE1_DI_MODULE_2 AT %I* : BYTE;
	OP90_MAS3_PORT2_BYTE2_DI_MODULE_2 AT %I* : BYTE;
	OP90_MAS3_PORT3_BYTE1_DI_MODULE_3 AT %I* : BYTE;
	OP90_MAS3_PORT3_BYTE2_DI_MODULE_3 AT %I* : BYTE;
	
	OP90_MAS3_PORT5_BYTE1_DO_MODULE_1 AT %Q* : BYTE;
	OP90_MAS3_PORT5_BYTE2_DO_MODULE_1 AT %Q* : BYTE;
	OP90_MAS3_PORT5_BYTE3_DO_MODULE_1 AT %Q* : BYTE;
	OP90_MAS3_PORT6_BYTE1_DO_MODULE_2 AT %Q* : BYTE;
	OP90_MAS3_PORT6_BYTE2_DO_MODULE_2 AT %Q* : BYTE;
	OP90_MAS3_PORT7_BYTE1_DO_MODULE_3 AT %Q* : BYTE; 
	OP90_MAS3_PORT7_BYTE2_DO_MODULE_3 AT %Q* : BYTE;
	OP90_MAS3_PORT7_BYTE3_DO_MODULE_3 AT %Q* : BYTE;
	
	

	BYTE_AS_BIT_0: BYTE_AS_BIT;
	BYTE_AS_BIT_1: BYTE_AS_BIT;
	BYTE_AS_BIT_2: BYTE_AS_BIT;
	BYTE_AS_BIT_3: BYTE_AS_BIT;
	BYTE_AS_BIT_4: BYTE_AS_BIT;
	BYTE_AS_BIT_5: BYTE_AS_BIT;
	
	
	
	BIT_AS_BYTE_0: BIT_AS_BYTE;
	BIT_AS_BYTE_1: BIT_AS_BYTE;
	BIT_AS_BYTE_2: BIT_AS_BYTE;
	BIT_AS_BYTE_3: BIT_AS_BYTE;
	BIT_AS_BYTE_4: BIT_AS_BYTE;
	BIT_AS_BYTE_5: BIT_AS_BYTE;
	BIT_AS_BYTE_6: BIT_AS_BYTE;
	BIT_AS_BYTE_7: BIT_AS_BYTE;
		
END_VAR

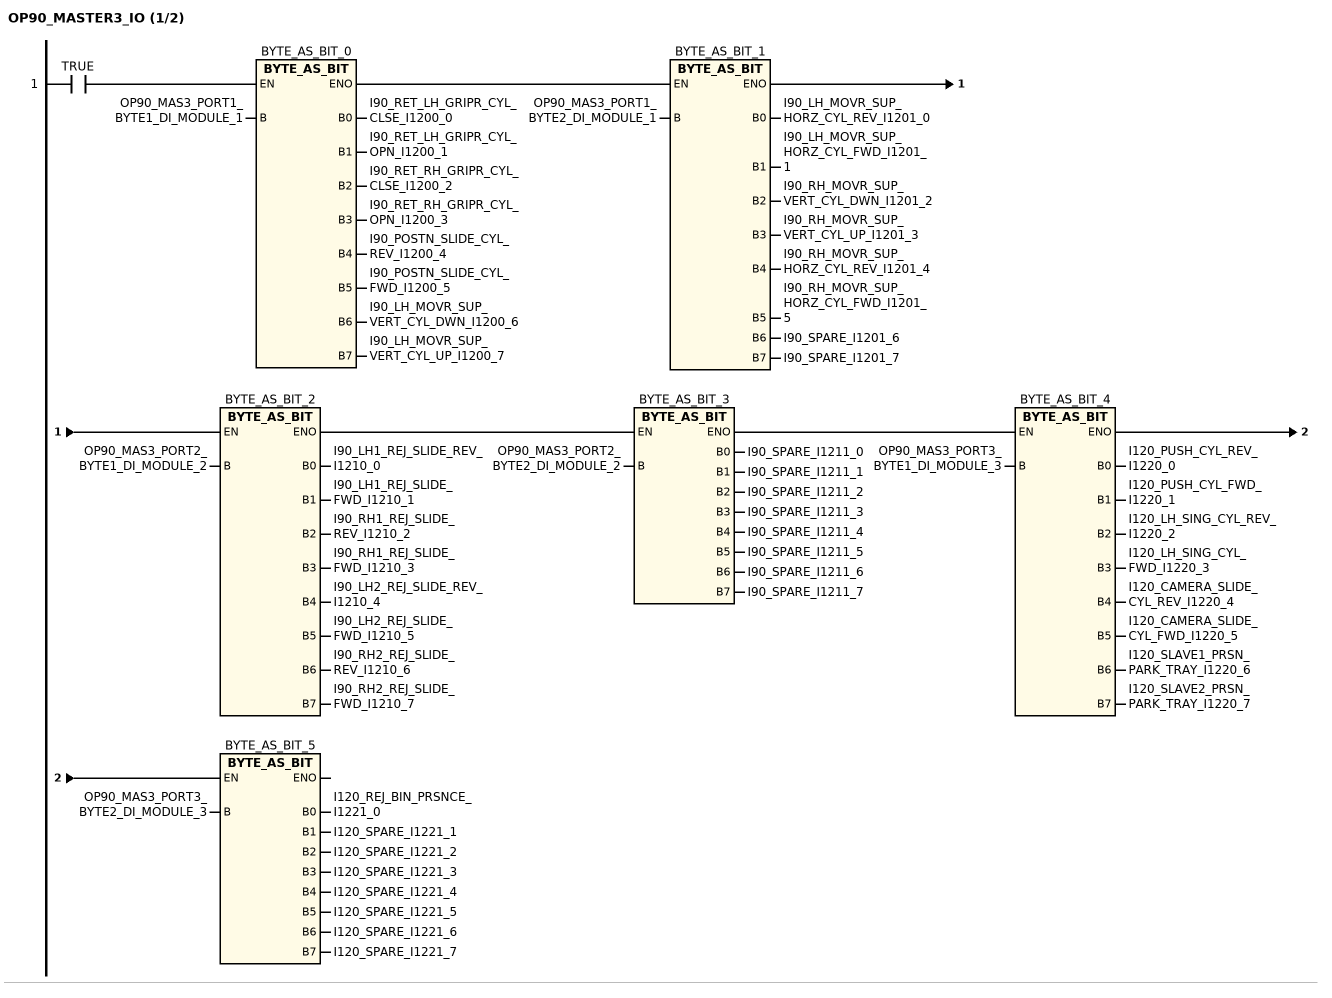
// NETWORK 1
BYTE_AS_BIT_0(
    B := OP90_MAS3_PORT1_BYTE1_DI_MODULE_1,
    B0 => I90_RET_LH_GRIPR_CYL_CLSE_I1200_0,
    B1 => I90_RET_LH_GRIPR_CYL_OPN_I1200_1,
    B2 => I90_RET_RH_GRIPR_CYL_CLSE_I1200_2,
    B3 => I90_RET_RH_GRIPR_CYL_OPN_I1200_3,
    B4 => I90_POSTN_SLIDE_CYL_REV_I1200_4,
    B5 => I90_POSTN_SLIDE_CYL_FWD_I1200_5,
    B6 => I90_LH_MOVR_SUP_VERT_CYL_DWN_I1200_6,
    B7 => I90_LH_MOVR_SUP_VERT_CYL_UP_I1200_7); // BYTE_AS_BIT
BYTE_AS_BIT_1(
    B := OP90_MAS3_PORT1_BYTE2_DI_MODULE_1,
    B0 => I90_LH_MOVR_SUP_HORZ_CYL_REV_I1201_0,
    B1 => I90_LH_MOVR_SUP_HORZ_CYL_FWD_I1201_1,
    B2 => I90_RH_MOVR_SUP_VERT_CYL_DWN_I1201_2,
    B3 => I90_RH_MOVR_SUP_VERT_CYL_UP_I1201_3,
    B4 => I90_RH_MOVR_SUP_HORZ_CYL_REV_I1201_4,
    B5 => I90_RH_MOVR_SUP_HORZ_CYL_FWD_I1201_5,
    B6 => I90_SPARE_I1201_6,
    B7 => I90_SPARE_I1201_7); // BYTE_AS_BIT
BYTE_AS_BIT_2(
    B := OP90_MAS3_PORT2_BYTE1_DI_MODULE_2,
    B0 => I90_LH1_REJ_SLIDE_REV_I1210_0,
    B1 => I90_LH1_REJ_SLIDE_FWD_I1210_1,
    B2 => I90_RH1_REJ_SLIDE_REV_I1210_2,
    B3 => I90_RH1_REJ_SLIDE_FWD_I1210_3,
    B4 => I90_LH2_REJ_SLIDE_REV_I1210_4,
    B5 => I90_LH2_REJ_SLIDE_FWD_I1210_5,
    B6 => I90_RH2_REJ_SLIDE_REV_I1210_6,
    B7 => I90_RH2_REJ_SLIDE_FWD_I1210_7); // BYTE_AS_BIT
BYTE_AS_BIT_3(
    B := OP90_MAS3_PORT2_BYTE2_DI_MODULE_2,
    B0 => I90_SPARE_I1211_0,
    B1 => I90_SPARE_I1211_1,
    B2 => I90_SPARE_I1211_2,
    B3 => I90_SPARE_I1211_3,
    B4 => I90_SPARE_I1211_4,
    B5 => I90_SPARE_I1211_5,
    B6 => I90_SPARE_I1211_6,
    B7 => I90_SPARE_I1211_7); // BYTE_AS_BIT
BYTE_AS_BIT_4(
    B := OP90_MAS3_PORT3_BYTE1_DI_MODULE_3,
    B0 => I120_PUSH_CYL_REV_I1220_0,
    B1 => I120_PUSH_CYL_FWD_I1220_1,
    B2 => I120_LH_SING_CYL_REV_I1220_2,
    B3 => I120_LH_SING_CYL_FWD_I1220_3,
    B4 => I120_CAMERA_SLIDE_CYL_REV_I1220_4,
    B5 => I120_CAMERA_SLIDE_CYL_FWD_I1220_5,
    B6 => I120_SLAVE1_PRSN_PARK_TRAY_I1220_6,
    B7 => I120_SLAVE2_PRSN_PARK_TRAY_I1220_7); // BYTE_AS_BIT
BYTE_AS_BIT_5(
    B := OP90_MAS3_PORT3_BYTE2_DI_MODULE_3,
    B0 => I120_REJ_BIN_PRSNCE_I1221_0,
    B1 => I120_SPARE_I1221_1,
    B2 => I120_SPARE_I1221_2,
    B3 => I120_SPARE_I1221_3,
    B4 => I120_SPARE_I1221_4,
    B5 => I120_SPARE_I1221_5,
    B6 => I120_SPARE_I1221_6,
    B7 => I120_SPARE_I1221_7); // BYTE_AS_BIT

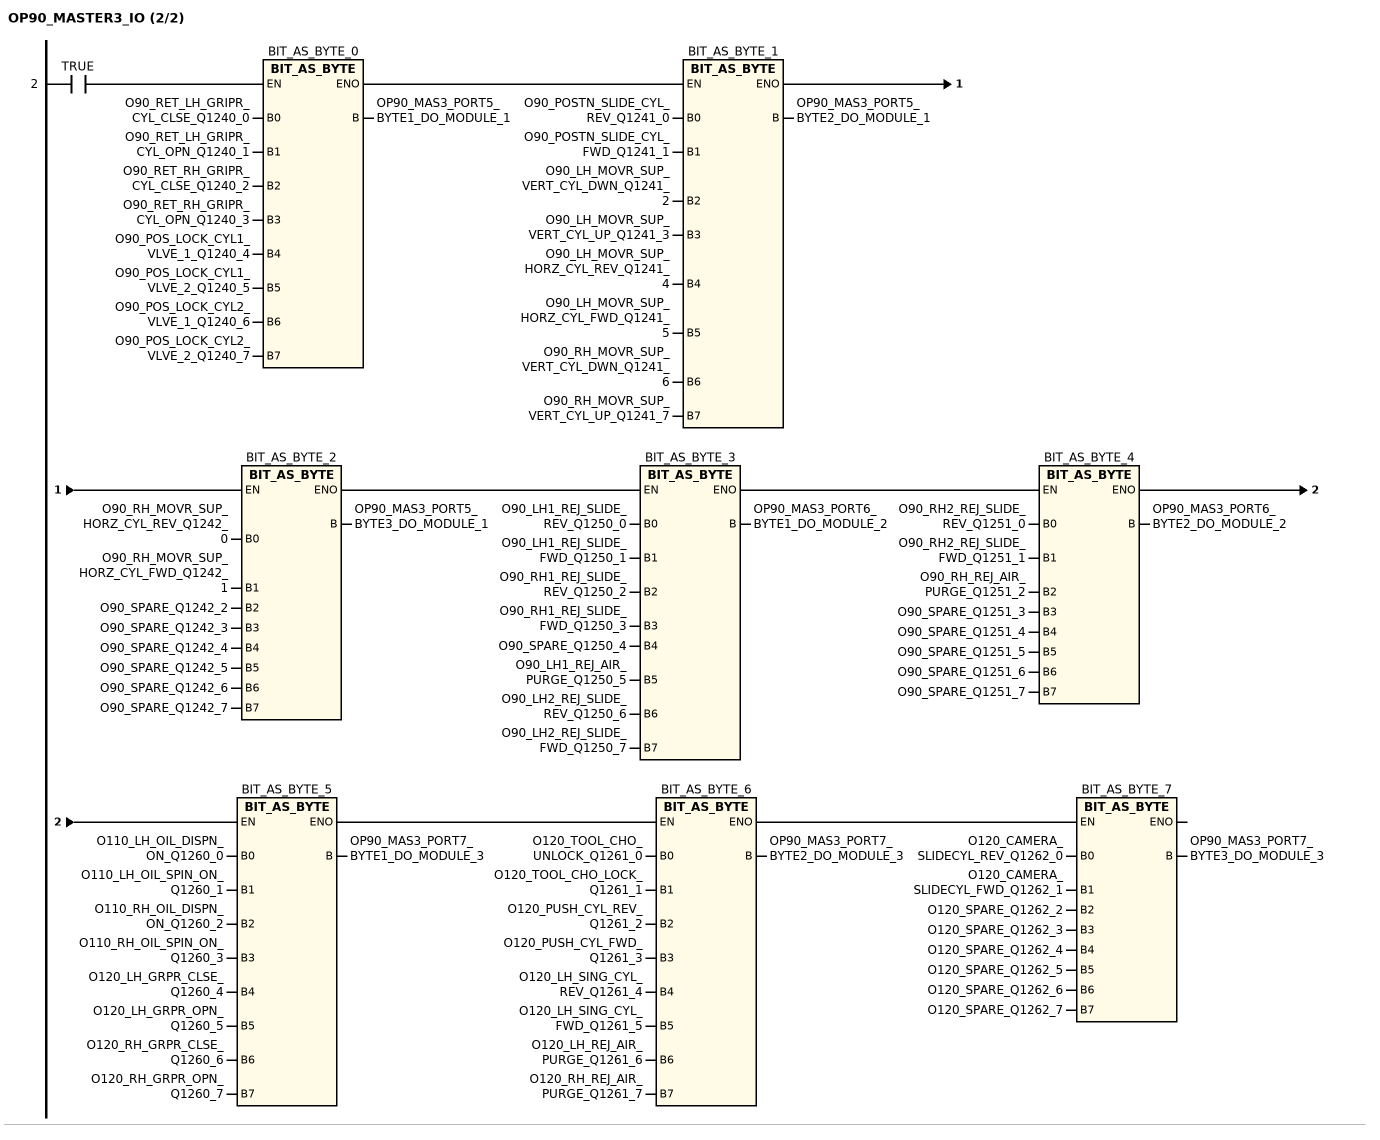
// NETWORK 2
BIT_AS_BYTE_0(
    B0 := O90_RET_LH_GRIPR_CYL_CLSE_Q1240_0,
    B1 := O90_RET_LH_GRIPR_CYL_OPN_Q1240_1,
    B2 := O90_RET_RH_GRIPR_CYL_CLSE_Q1240_2,
    B3 := O90_RET_RH_GRIPR_CYL_OPN_Q1240_3,
    B4 := O90_POS_LOCK_CYL1_VLVE_1_Q1240_4,
    B5 := O90_POS_LOCK_CYL1_VLVE_2_Q1240_5,
    B6 := O90_POS_LOCK_CYL2_VLVE_1_Q1240_6,
    B7 := O90_POS_LOCK_CYL2_VLVE_2_Q1240_7,
    B => OP90_MAS3_PORT5_BYTE1_DO_MODULE_1); // BIT_AS_BYTE
BIT_AS_BYTE_1(
    B0 := O90_POSTN_SLIDE_CYL_REV_Q1241_0,
    B1 := O90_POSTN_SLIDE_CYL_FWD_Q1241_1,
    B2 := O90_LH_MOVR_SUP_VERT_CYL_DWN_Q1241_2,
    B3 := O90_LH_MOVR_SUP_VERT_CYL_UP_Q1241_3,
    B4 := O90_LH_MOVR_SUP_HORZ_CYL_REV_Q1241_4,
    B5 := O90_LH_MOVR_SUP_HORZ_CYL_FWD_Q1241_5,
    B6 := O90_RH_MOVR_SUP_VERT_CYL_DWN_Q1241_6,
    B7 := O90_RH_MOVR_SUP_VERT_CYL_UP_Q1241_7,
    B => OP90_MAS3_PORT5_BYTE2_DO_MODULE_1); // BIT_AS_BYTE
BIT_AS_BYTE_2(
    B0 := O90_RH_MOVR_SUP_HORZ_CYL_REV_Q1242_0,
    B1 := O90_RH_MOVR_SUP_HORZ_CYL_FWD_Q1242_1,
    B2 := O90_SPARE_Q1242_2,
    B3 := O90_SPARE_Q1242_3,
    B4 := O90_SPARE_Q1242_4,
    B5 := O90_SPARE_Q1242_5,
    B6 := O90_SPARE_Q1242_6,
    B7 := O90_SPARE_Q1242_7,
    B => OP90_MAS3_PORT5_BYTE3_DO_MODULE_1); // BIT_AS_BYTE
BIT_AS_BYTE_3(
    B0 := O90_LH1_REJ_SLIDE_REV_Q1250_0,
    B1 := O90_LH1_REJ_SLIDE_FWD_Q1250_1,
    B2 := O90_RH1_REJ_SLIDE_REV_Q1250_2,
    B3 := O90_RH1_REJ_SLIDE_FWD_Q1250_3,
    B4 := O90_SPARE_Q1250_4,
    B5 := O90_LH1_REJ_AIR_PURGE_Q1250_5,
    B6 := O90_LH2_REJ_SLIDE_REV_Q1250_6,
    B7 := O90_LH2_REJ_SLIDE_FWD_Q1250_7,
    B => OP90_MAS3_PORT6_BYTE1_DO_MODULE_2); // BIT_AS_BYTE
BIT_AS_BYTE_4(
    B0 := O90_RH2_REJ_SLIDE_REV_Q1251_0,
    B1 := O90_RH2_REJ_SLIDE_FWD_Q1251_1,
    B2 := O90_RH_REJ_AIR_PURGE_Q1251_2,
    B3 := O90_SPARE_Q1251_3,
    B4 := O90_SPARE_Q1251_4,
    B5 := O90_SPARE_Q1251_5,
    B6 := O90_SPARE_Q1251_6,
    B7 := O90_SPARE_Q1251_7,
    B => OP90_MAS3_PORT6_BYTE2_DO_MODULE_2); // BIT_AS_BYTE
BIT_AS_BYTE_5(
    B0 := O110_LH_OIL_DISPN_ON_Q1260_0,
    B1 := O110_LH_OIL_SPIN_ON_Q1260_1,
    B2 := O110_RH_OIL_DISPN_ON_Q1260_2,
    B3 := O110_RH_OIL_SPIN_ON_Q1260_3,
    B4 := O120_LH_GRPR_CLSE_Q1260_4,
    B5 := O120_LH_GRPR_OPN_Q1260_5,
    B6 := O120_RH_GRPR_CLSE_Q1260_6,
    B7 := O120_RH_GRPR_OPN_Q1260_7,
    B => OP90_MAS3_PORT7_BYTE1_DO_MODULE_3); // BIT_AS_BYTE
BIT_AS_BYTE_6(
    B0 := O120_TOOL_CHO_UNLOCK_Q1261_0,
    B1 := O120_TOOL_CHO_LOCK_Q1261_1,
    B2 := O120_PUSH_CYL_REV_Q1261_2,
    B3 := O120_PUSH_CYL_FWD_Q1261_3,
    B4 := O120_LH_SING_CYL_REV_Q1261_4,
    B5 := O120_LH_SING_CYL_FWD_Q1261_5,
    B6 := O120_LH_REJ_AIR_PURGE_Q1261_6,
    B7 := O120_RH_REJ_AIR_PURGE_Q1261_7,
    B => OP90_MAS3_PORT7_BYTE2_DO_MODULE_3); // BIT_AS_BYTE
BIT_AS_BYTE_7(
    B0 := O120_CAMERA_SLIDECYL_REV_Q1262_0,
    B1 := O120_CAMERA_SLIDECYL_FWD_Q1262_1,
    B2 := O120_SPARE_Q1262_2,
    B3 := O120_SPARE_Q1262_3,
    B4 := O120_SPARE_Q1262_4,
    B5 := O120_SPARE_Q1262_5,
    B6 := O120_SPARE_Q1262_6,
    B7 := O120_SPARE_Q1262_7,
    B => OP90_MAS3_PORT7_BYTE3_DO_MODULE_3); // BIT_AS_BYTE

END_PROGRAM

// ---- POUs/IO/OP90_JB_IO.TcPOU
PROGRAM OP90_JB_IO

VAR
	OP90_JB_DI_MODULE_1 AT %I* : WORD;
	OP90_JB_DI_MODULE_2 AT %I* : WORD;
	OP90_JB_DI_MODULE_3 AT %I* : WORD;
	
	OP90_JB_DO_MODULE_1  AT %Q* : WORD;
	OP90_JB_DO_MODULE_2 AT %Q* : WORD;
	
	WORD_AS_BIT_0: WORD_AS_BIT;
	WORD_AS_BIT_1: WORD_AS_BIT;
	WORD_AS_BIT_2: WORD_AS_BIT;
	
	BIT_AS_WORD_0: BIT_AS_WORD;
	BIT_AS_WORD_1: BIT_AS_WORD;
END_VAR

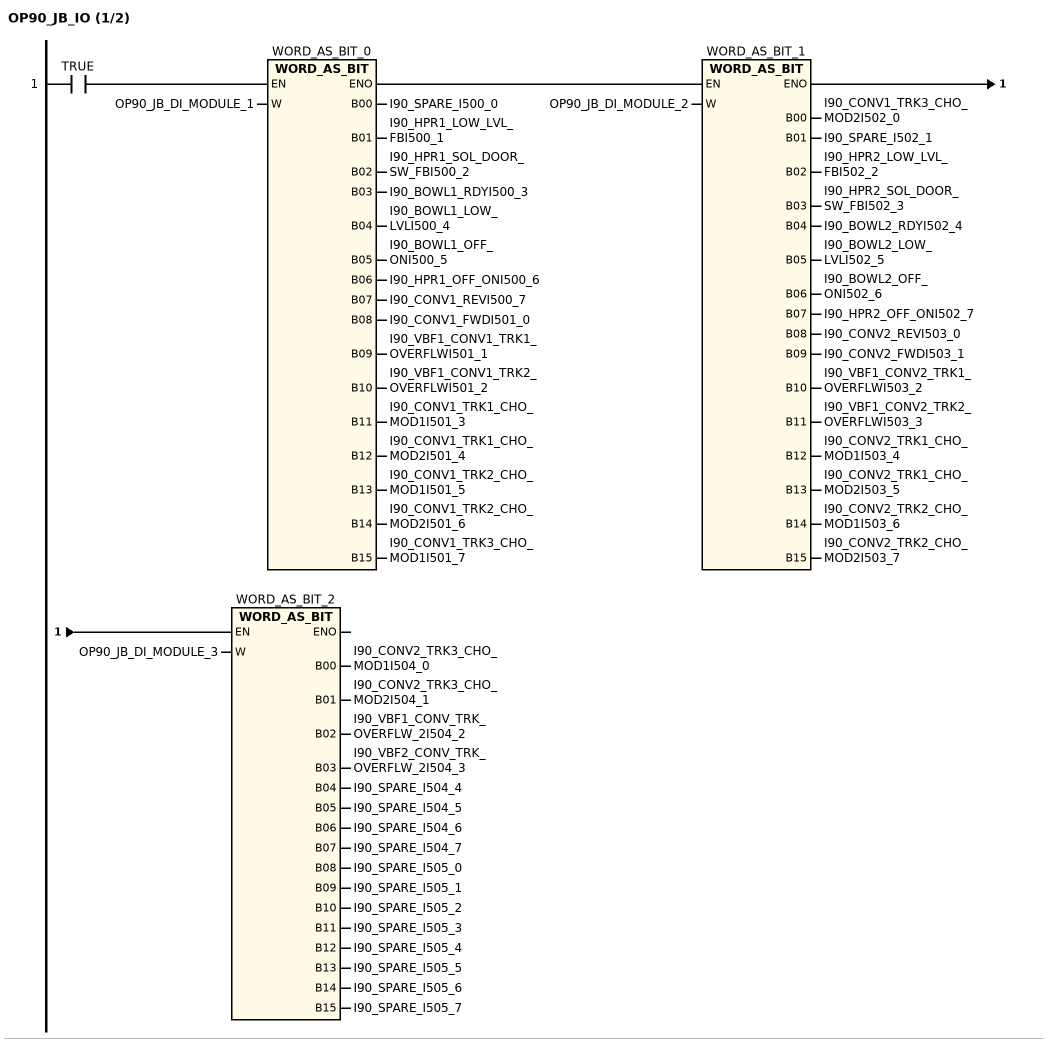
// NETWORK 1
WORD_AS_BIT_0(
    W := OP90_JB_DI_MODULE_1,
    B00 => I90_SPARE_I500_0,
    B01 => I90_HPR1_LOW_LVL_FBI500_1,
    B02 => I90_HPR1_SOL_DOOR_SW_FBI500_2,
    B03 => I90_BOWL1_RDYI500_3,
    B04 => I90_BOWL1_LOW_LVLI500_4,
    B05 => I90_BOWL1_OFF_ONI500_5,
    B06 => I90_HPR1_OFF_ONI500_6,
    B07 => I90_CONV1_REVI500_7,
    B08 => I90_CONV1_FWDI501_0,
    B09 => I90_VBF1_CONV1_TRK1_OVERFLWI501_1,
    B10 => I90_VBF1_CONV1_TRK2_OVERFLWI501_2,
    B11 => I90_CONV1_TRK1_CHO_MOD1I501_3,
    B12 => I90_CONV1_TRK1_CHO_MOD2I501_4,
    B13 => I90_CONV1_TRK2_CHO_MOD1I501_5,
    B14 => I90_CONV1_TRK2_CHO_MOD2I501_6,
    B15 => I90_CONV1_TRK3_CHO_MOD1I501_7); // WORD_AS_BIT
WORD_AS_BIT_1(
    W := OP90_JB_DI_MODULE_2,
    B00 => I90_CONV1_TRK3_CHO_MOD2I502_0,
    B01 => I90_SPARE_I502_1,
    B02 => I90_HPR2_LOW_LVL_FBI502_2,
    B03 => I90_HPR2_SOL_DOOR_SW_FBI502_3,
    B04 => I90_BOWL2_RDYI502_4,
    B05 => I90_BOWL2_LOW_LVLI502_5,
    B06 => I90_BOWL2_OFF_ONI502_6,
    B07 => I90_HPR2_OFF_ONI502_7,
    B08 => I90_CONV2_REVI503_0,
    B09 => I90_CONV2_FWDI503_1,
    B10 => I90_VBF1_CONV2_TRK1_OVERFLWI503_2,
    B11 => I90_VBF1_CONV2_TRK2_OVERFLWI503_3,
    B12 => I90_CONV2_TRK1_CHO_MOD1I503_4,
    B13 => I90_CONV2_TRK1_CHO_MOD2I503_5,
    B14 => I90_CONV2_TRK2_CHO_MOD1I503_6,
    B15 => I90_CONV2_TRK2_CHO_MOD2I503_7); // WORD_AS_BIT
WORD_AS_BIT_2(
    W := OP90_JB_DI_MODULE_3,
    B00 => I90_CONV2_TRK3_CHO_MOD1I504_0,
    B01 => I90_CONV2_TRK3_CHO_MOD2I504_1,
    B02 => I90_VBF1_CONV_TRK_OVERFLW_2I504_2,
    B03 => I90_VBF2_CONV_TRK_OVERFLW_2I504_3,
    B04 => I90_SPARE_I504_4,
    B05 => I90_SPARE_I504_5,
    B06 => I90_SPARE_I504_6,
    B07 => I90_SPARE_I504_7,
    B08 => I90_SPARE_I505_0,
    B09 => I90_SPARE_I505_1,
    B10 => I90_SPARE_I505_2,
    B11 => I90_SPARE_I505_3,
    B12 => I90_SPARE_I505_4,
    B13 => I90_SPARE_I505_5,
    B14 => I90_SPARE_I505_6,
    B15 => I90_SPARE_I505_7); // WORD_AS_BIT

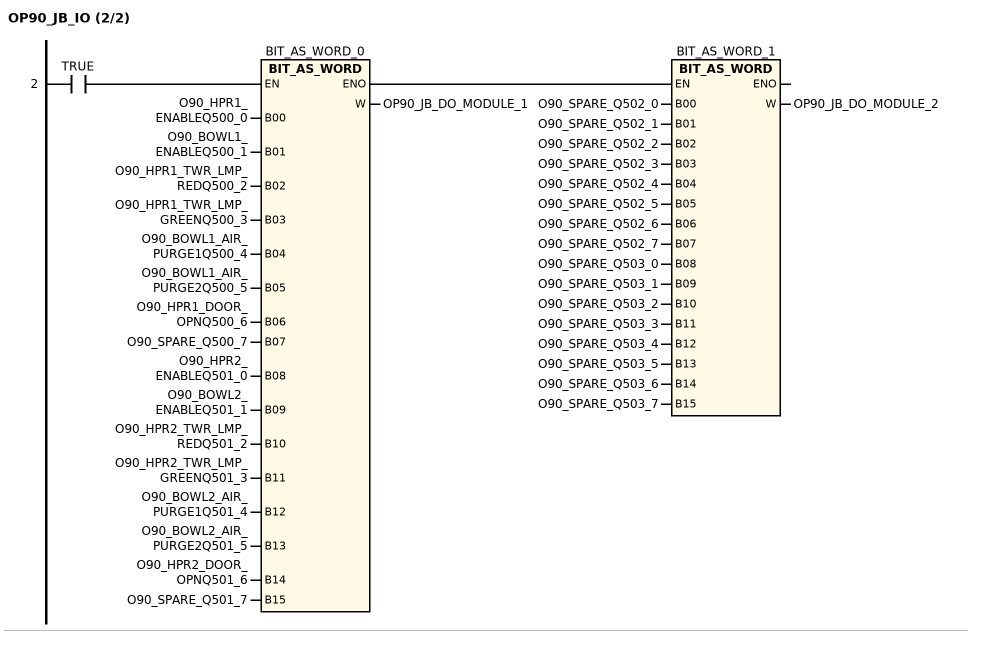
// NETWORK 2
BIT_AS_WORD_0(
    B00 := O90_HPR1_ENABLEQ500_0,
    B01 := O90_BOWL1_ENABLEQ500_1,
    B02 := O90_HPR1_TWR_LMP_REDQ500_2,
    B03 := O90_HPR1_TWR_LMP_GREENQ500_3,
    B04 := O90_BOWL1_AIR_PURGE1Q500_4,
    B05 := O90_BOWL1_AIR_PURGE2Q500_5,
    B06 := O90_HPR1_DOOR_OPNQ500_6,
    B07 := O90_SPARE_Q500_7,
    B08 := O90_HPR2_ENABLEQ501_0,
    B09 := O90_BOWL2_ENABLEQ501_1,
    B10 := O90_HPR2_TWR_LMP_REDQ501_2,
    B11 := O90_HPR2_TWR_LMP_GREENQ501_3,
    B12 := O90_BOWL2_AIR_PURGE1Q501_4,
    B13 := O90_BOWL2_AIR_PURGE2Q501_5,
    B14 := O90_HPR2_DOOR_OPNQ501_6,
    B15 := O90_SPARE_Q501_7,
    W => OP90_JB_DO_MODULE_1); // BIT_AS_WORD
BIT_AS_WORD_1(
    B00 := O90_SPARE_Q502_0,
    B01 := O90_SPARE_Q502_1,
    B02 := O90_SPARE_Q502_2,
    B03 := O90_SPARE_Q502_3,
    B04 := O90_SPARE_Q502_4,
    B05 := O90_SPARE_Q502_5,
    B06 := O90_SPARE_Q502_6,
    B07 := O90_SPARE_Q502_7,
    B08 := O90_SPARE_Q503_0,
    B09 := O90_SPARE_Q503_1,
    B10 := O90_SPARE_Q503_2,
    B11 := O90_SPARE_Q503_3,
    B12 := O90_SPARE_Q503_4,
    B13 := O90_SPARE_Q503_5,
    B14 := O90_SPARE_Q503_6,
    B15 := O90_SPARE_Q503_7,
    W => OP90_JB_DO_MODULE_2); // BIT_AS_WORD

END_PROGRAM

// ---- POUs/IO/OP160_MP_IO.TcPOU
PROGRAM OP160_MP_IO
VAR
	OP160_MP_DI_MODULE_1 AT %I* : WORD;
	OP160_MP_DI_MODULE_2 AT %I* : WORD;
	OP160_MP_DI_MODULE_3 AT %I* : WORD;
	OP160_MP_DI_MODULE_4 AT %I* : WORD;
	OP160_MP_DI_MODULE_5 AT %I* : WORD;
	OP160_MP_DI_MODULE_6 AT %I* : WORD;
	OP160_MP_DI_MODULE_7 AT %I* : WORD;
	OP160_MP_DI_MODULE_8 AT %I* : WORD;
	
	OP160_MP_DO_MODULE_1 AT %Q* : WORD;
	OP160_MP_DO_MODULE_2 AT %Q* : WORD;
	OP160_MP_DO_MODULE_3 AT %Q* : WORD;
	OP160_MP_DO_MODULE_4 AT %Q* : WORD;
	OP160_MP_DO_MODULE_5 AT %Q* : WORD;
	
	
	WORD_AS_BIT_0: WORD_AS_BIT;
	WORD_AS_BIT_1: WORD_AS_BIT;
	WORD_AS_BIT_2: WORD_AS_BIT;
	WORD_AS_BIT_3: WORD_AS_BIT;
	WORD_AS_BIT_4: WORD_AS_BIT;
	WORD_AS_BIT_5: WORD_AS_BIT;
	WORD_AS_BIT_6: WORD_AS_BIT;
	WORD_AS_BIT_7: WORD_AS_BIT;
	
	BIT_AS_WORD_0: BIT_AS_WORD;
	BIT_AS_WORD_1: BIT_AS_WORD;
	BIT_AS_WORD_2: BIT_AS_WORD;
	BIT_AS_WORD_3: BIT_AS_WORD;
	BIT_AS_WORD_4: BIT_AS_WORD;
END_VAR

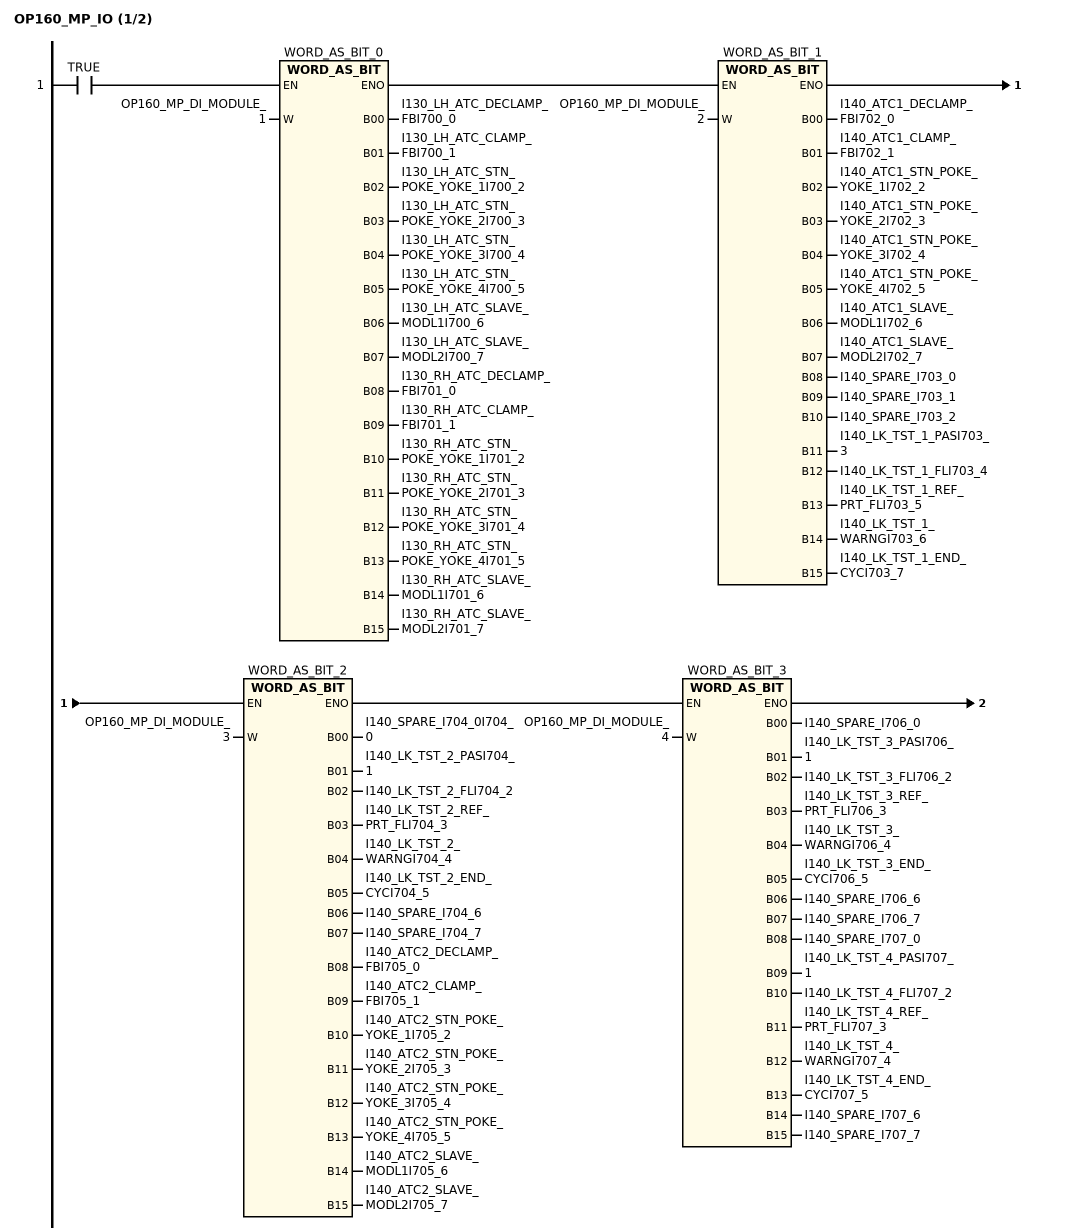
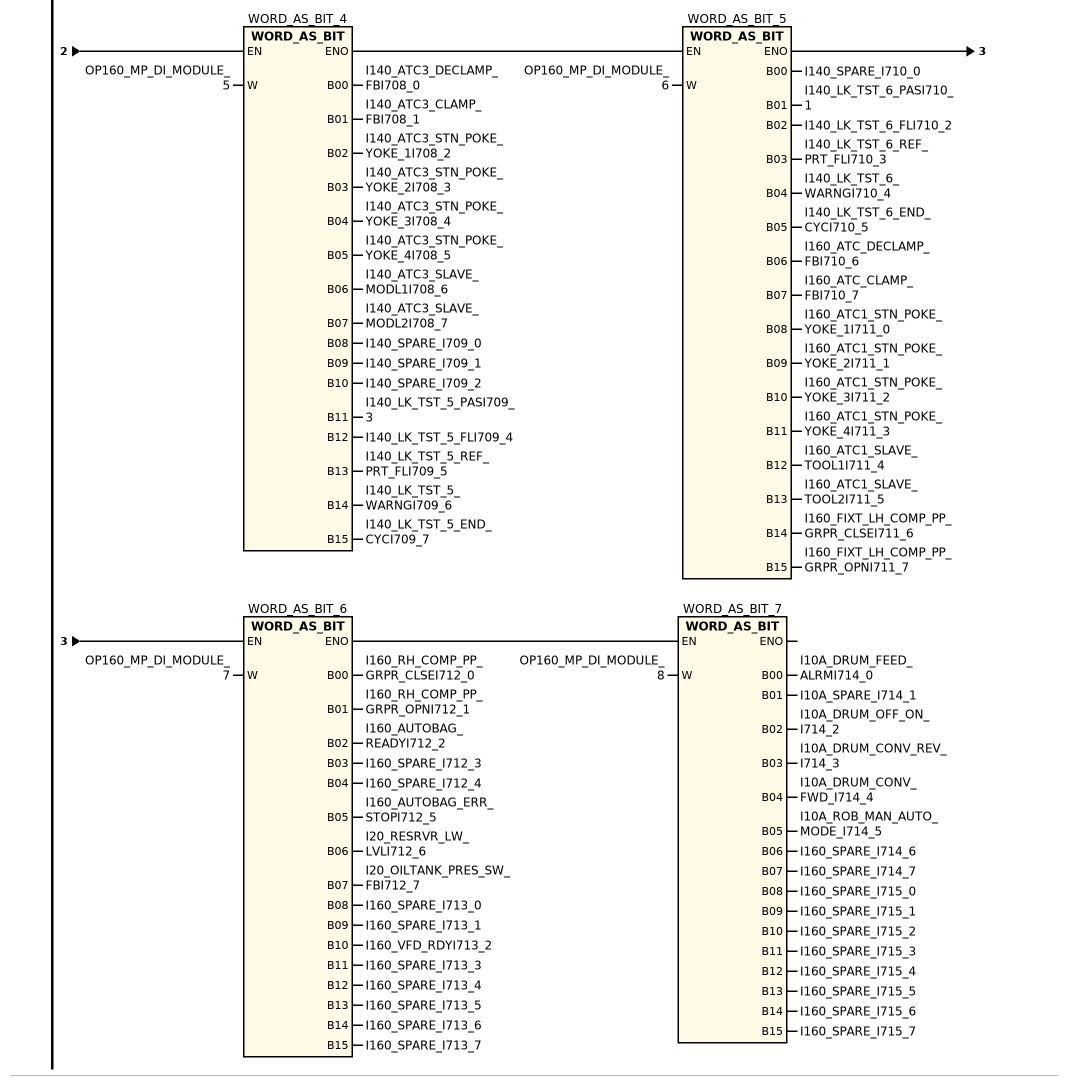
// NETWORK 1
WORD_AS_BIT_0(
    W := OP160_MP_DI_MODULE_1,
    B00 => I130_LH_ATC_DECLAMP_FBI700_0,
    B01 => I130_LH_ATC_CLAMP_FBI700_1,
    B02 => I130_LH_ATC_STN_POKE_YOKE_1I700_2,
    B03 => I130_LH_ATC_STN_POKE_YOKE_2I700_3,
    B04 => I130_LH_ATC_STN_POKE_YOKE_3I700_4,
    B05 => I130_LH_ATC_STN_POKE_YOKE_4I700_5,
    B06 => I130_LH_ATC_SLAVE_MODL1I700_6,
    B07 => I130_LH_ATC_SLAVE_MODL2I700_7,
    B08 => I130_RH_ATC_DECLAMP_FBI701_0,
    B09 => I130_RH_ATC_CLAMP_FBI701_1,
    B10 => I130_RH_ATC_STN_POKE_YOKE_1I701_2,
    B11 => I130_RH_ATC_STN_POKE_YOKE_2I701_3,
    B12 => I130_RH_ATC_STN_POKE_YOKE_3I701_4,
    B13 => I130_RH_ATC_STN_POKE_YOKE_4I701_5,
    B14 => I130_RH_ATC_SLAVE_MODL1I701_6,
    B15 => I130_RH_ATC_SLAVE_MODL2I701_7); // WORD_AS_BIT
WORD_AS_BIT_1(
    W := OP160_MP_DI_MODULE_2,
    B00 => I140_ATC1_DECLAMP_FBI702_0,
    B01 => I140_ATC1_CLAMP_FBI702_1,
    B02 => I140_ATC1_STN_POKE_YOKE_1I702_2,
    B03 => I140_ATC1_STN_POKE_YOKE_2I702_3,
    B04 => I140_ATC1_STN_POKE_YOKE_3I702_4,
    B05 => I140_ATC1_STN_POKE_YOKE_4I702_5,
    B06 => I140_ATC1_SLAVE_MODL1I702_6,
    B07 => I140_ATC1_SLAVE_MODL2I702_7,
    B08 => I140_SPARE_I703_0,
    B09 => I140_SPARE_I703_1,
    B10 => I140_SPARE_I703_2,
    B11 => I140_LK_TST_1_PASI703_3,
    B12 => I140_LK_TST_1_FLI703_4,
    B13 => I140_LK_TST_1_REF_PRT_FLI703_5,
    B14 => I140_LK_TST_1_WARNGI703_6,
    B15 => I140_LK_TST_1_END_CYCI703_7); // WORD_AS_BIT
WORD_AS_BIT_2(
    W := OP160_MP_DI_MODULE_3,
    B00 => I140_SPARE_I704_0I704_0,
    B01 => I140_LK_TST_2_PASI704_1,
    B02 => I140_LK_TST_2_FLI704_2,
    B03 => I140_LK_TST_2_REF_PRT_FLI704_3,
    B04 => I140_LK_TST_2_WARNGI704_4,
    B05 => I140_LK_TST_2_END_CYCI704_5,
    B06 => I140_SPARE_I704_6,
    B07 => I140_SPARE_I704_7,
    B08 => I140_ATC2_DECLAMP_FBI705_0,
    B09 => I140_ATC2_CLAMP_FBI705_1,
    B10 => I140_ATC2_STN_POKE_YOKE_1I705_2,
    B11 => I140_ATC2_STN_POKE_YOKE_2I705_3,
    B12 => I140_ATC2_STN_POKE_YOKE_3I705_4,
    B13 => I140_ATC2_STN_POKE_YOKE_4I705_5,
    B14 => I140_ATC2_SLAVE_MODL1I705_6,
    B15 => I140_ATC2_SLAVE_MODL2I705_7); // WORD_AS_BIT
WORD_AS_BIT_3(
    W := OP160_MP_DI_MODULE_4,
    B00 => I140_SPARE_I706_0,
    B01 => I140_LK_TST_3_PASI706_1,
    B02 => I140_LK_TST_3_FLI706_2,
    B03 => I140_LK_TST_3_REF_PRT_FLI706_3,
    B04 => I140_LK_TST_3_WARNGI706_4,
    B05 => I140_LK_TST_3_END_CYCI706_5,
    B06 => I140_SPARE_I706_6,
    B07 => I140_SPARE_I706_7,
    B08 => I140_SPARE_I707_0,
    B09 => I140_LK_TST_4_PASI707_1,
    B10 => I140_LK_TST_4_FLI707_2,
    B11 => I140_LK_TST_4_REF_PRT_FLI707_3,
    B12 => I140_LK_TST_4_WARNGI707_4,
    B13 => I140_LK_TST_4_END_CYCI707_5,
    B14 => I140_SPARE_I707_6,
    B15 => I140_SPARE_I707_7); // WORD_AS_BIT
WORD_AS_BIT_4(
    W := OP160_MP_DI_MODULE_5,
    B00 => I140_ATC3_DECLAMP_FBI708_0,
    B01 => I140_ATC3_CLAMP_FBI708_1,
    B02 => I140_ATC3_STN_POKE_YOKE_1I708_2,
    B03 => I140_ATC3_STN_POKE_YOKE_2I708_3,
    B04 => I140_ATC3_STN_POKE_YOKE_3I708_4,
    B05 => I140_ATC3_STN_POKE_YOKE_4I708_5,
    B06 => I140_ATC3_SLAVE_MODL1I708_6,
    B07 => I140_ATC3_SLAVE_MODL2I708_7,
    B08 => I140_SPARE_I709_0,
    B09 => I140_SPARE_I709_1,
    B10 => I140_SPARE_I709_2,
    B11 => I140_LK_TST_5_PASI709_3,
    B12 => I140_LK_TST_5_FLI709_4,
    B13 => I140_LK_TST_5_REF_PRT_FLI709_5,
    B14 => I140_LK_TST_5_WARNGI709_6,
    B15 => I140_LK_TST_5_END_CYCI709_7); // WORD_AS_BIT
WORD_AS_BIT_5(
    W := OP160_MP_DI_MODULE_6,
    B00 => I140_SPARE_I710_0,
    B01 => I140_LK_TST_6_PASI710_1,
    B02 => I140_LK_TST_6_FLI710_2,
    B03 => I140_LK_TST_6_REF_PRT_FLI710_3,
    B04 => I140_LK_TST_6_WARNGI710_4,
    B05 => I140_LK_TST_6_END_CYCI710_5,
    B06 => I160_ATC_DECLAMP_FBI710_6,
    B07 => I160_ATC_CLAMP_FBI710_7,
    B08 => I160_ATC1_STN_POKE_YOKE_1I711_0,
    B09 => I160_ATC1_STN_POKE_YOKE_2I711_1,
    B10 => I160_ATC1_STN_POKE_YOKE_3I711_2,
    B11 => I160_ATC1_STN_POKE_YOKE_4I711_3,
    B12 => I160_ATC1_SLAVE_TOOL1I711_4,
    B13 => I160_ATC1_SLAVE_TOOL2I711_5,
    B14 => I160_FIXT_LH_COMP_PP_GRPR_CLSEI711_6,
    B15 => I160_FIXT_LH_COMP_PP_GRPR_OPNI711_7); // WORD_AS_BIT
WORD_AS_BIT_6(
    W := OP160_MP_DI_MODULE_7,
    B00 => I160_RH_COMP_PP_GRPR_CLSEI712_0,
    B01 => I160_RH_COMP_PP_GRPR_OPNI712_1,
    B02 => I160_AUTOBAG_READYI712_2,
    B03 => I160_SPARE_I712_3,
    B04 => I160_SPARE_I712_4,
    B05 => I160_AUTOBAG_ERR_STOPI712_5,
    B06 => I20_RESRVR_LW_LVLI712_6,
    B07 => I20_OILTANK_PRES_SW_FBI712_7,
    B08 => I160_SPARE_I713_0,
    B09 => I160_SPARE_I713_1,
    B10 => I160_VFD_RDYI713_2,
    B11 => I160_SPARE_I713_3,
    B12 => I160_SPARE_I713_4,
    B13 => I160_SPARE_I713_5,
    B14 => I160_SPARE_I713_6,
    B15 => I160_SPARE_I713_7); // WORD_AS_BIT
WORD_AS_BIT_7(
    W := OP160_MP_DI_MODULE_8,
    B00 => I10A_DRUM_FEED_ALRMI714_0,
    B01 => I10A_SPARE_I714_1,
    B02 => I10A_DRUM_OFF_ON_I714_2,
    B03 => I10A_DRUM_CONV_REV_I714_3,
    B04 => I10A_DRUM_CONV_FWD_I714_4,
    B05 => I10A_ROB_MAN_AUTO_MODE_I714_5,
    B06 => I160_SPARE_I714_6,
    B07 => I160_SPARE_I714_7,
    B08 => I160_SPARE_I715_0,
    B09 => I160_SPARE_I715_1,
    B10 => I160_SPARE_I715_2,
    B11 => I160_SPARE_I715_3,
    B12 => I160_SPARE_I715_4,
    B13 => I160_SPARE_I715_5,
    B14 => I160_SPARE_I715_6,
    B15 => I160_SPARE_I715_7); // WORD_AS_BIT

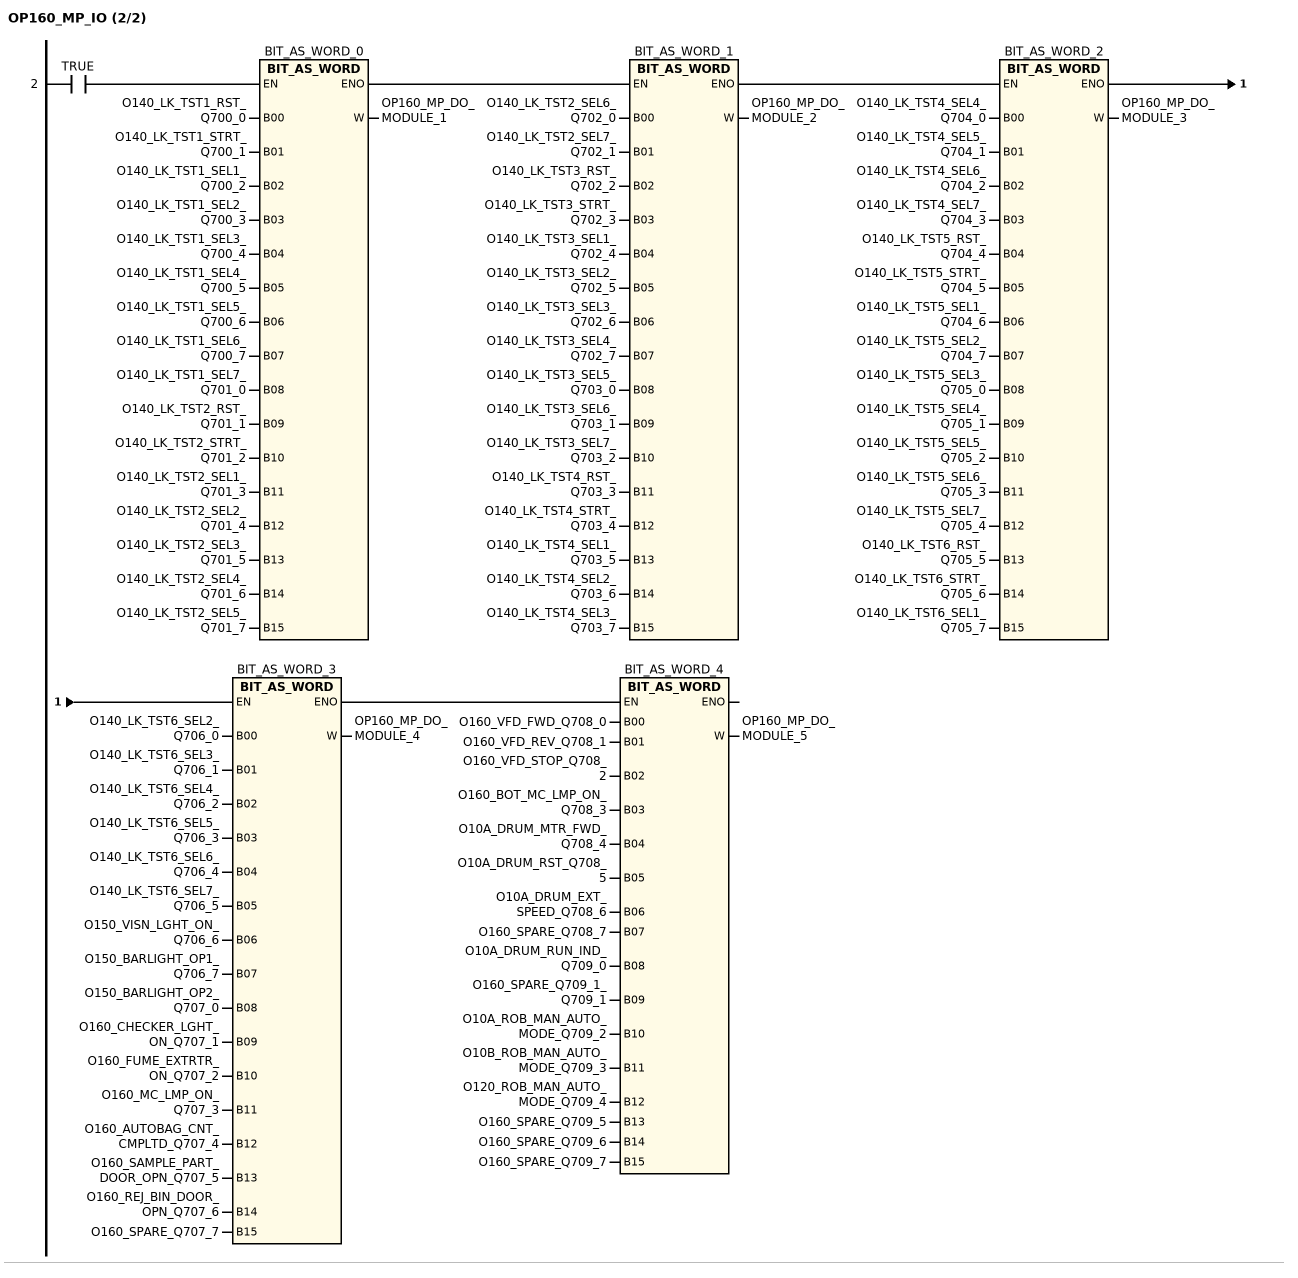
// NETWORK 2
BIT_AS_WORD_0(
    B00 := O140_LK_TST1_RST_Q700_0,
    B01 := O140_LK_TST1_STRT_Q700_1,
    B02 := O140_LK_TST1_SEL1_Q700_2,
    B03 := O140_LK_TST1_SEL2_Q700_3,
    B04 := O140_LK_TST1_SEL3_Q700_4,
    B05 := O140_LK_TST1_SEL4_Q700_5,
    B06 := O140_LK_TST1_SEL5_Q700_6,
    B07 := O140_LK_TST1_SEL6_Q700_7,
    B08 := O140_LK_TST1_SEL7_Q701_0,
    B09 := O140_LK_TST2_RST_Q701_1,
    B10 := O140_LK_TST2_STRT_Q701_2,
    B11 := O140_LK_TST2_SEL1_Q701_3,
    B12 := O140_LK_TST2_SEL2_Q701_4,
    B13 := O140_LK_TST2_SEL3_Q701_5,
    B14 := O140_LK_TST2_SEL4_Q701_6,
    B15 := O140_LK_TST2_SEL5_Q701_7,
    W => OP160_MP_DO_MODULE_1); // BIT_AS_WORD
BIT_AS_WORD_1(
    B00 := O140_LK_TST2_SEL6_Q702_0,
    B01 := O140_LK_TST2_SEL7_Q702_1,
    B02 := O140_LK_TST3_RST_Q702_2,
    B03 := O140_LK_TST3_STRT_Q702_3,
    B04 := O140_LK_TST3_SEL1_Q702_4,
    B05 := O140_LK_TST3_SEL2_Q702_5,
    B06 := O140_LK_TST3_SEL3_Q702_6,
    B07 := O140_LK_TST3_SEL4_Q702_7,
    B08 := O140_LK_TST3_SEL5_Q703_0,
    B09 := O140_LK_TST3_SEL6_Q703_1,
    B10 := O140_LK_TST3_SEL7_Q703_2,
    B11 := O140_LK_TST4_RST_Q703_3,
    B12 := O140_LK_TST4_STRT_Q703_4,
    B13 := O140_LK_TST4_SEL1_Q703_5,
    B14 := O140_LK_TST4_SEL2_Q703_6,
    B15 := O140_LK_TST4_SEL3_Q703_7,
    W => OP160_MP_DO_MODULE_2); // BIT_AS_WORD
BIT_AS_WORD_2(
    B00 := O140_LK_TST4_SEL4_Q704_0,
    B01 := O140_LK_TST4_SEL5_Q704_1,
    B02 := O140_LK_TST4_SEL6_Q704_2,
    B03 := O140_LK_TST4_SEL7_Q704_3,
    B04 := O140_LK_TST5_RST_Q704_4,
    B05 := O140_LK_TST5_STRT_Q704_5,
    B06 := O140_LK_TST5_SEL1_Q704_6,
    B07 := O140_LK_TST5_SEL2_Q704_7,
    B08 := O140_LK_TST5_SEL3_Q705_0,
    B09 := O140_LK_TST5_SEL4_Q705_1,
    B10 := O140_LK_TST5_SEL5_Q705_2,
    B11 := O140_LK_TST5_SEL6_Q705_3,
    B12 := O140_LK_TST5_SEL7_Q705_4,
    B13 := O140_LK_TST6_RST_Q705_5,
    B14 := O140_LK_TST6_STRT_Q705_6,
    B15 := O140_LK_TST6_SEL1_Q705_7,
    W => OP160_MP_DO_MODULE_3); // BIT_AS_WORD
BIT_AS_WORD_3(
    B00 := O140_LK_TST6_SEL2_Q706_0,
    B01 := O140_LK_TST6_SEL3_Q706_1,
    B02 := O140_LK_TST6_SEL4_Q706_2,
    B03 := O140_LK_TST6_SEL5_Q706_3,
    B04 := O140_LK_TST6_SEL6_Q706_4,
    B05 := O140_LK_TST6_SEL7_Q706_5,
    B06 := O150_VISN_LGHT_ON_Q706_6,
    B07 := O150_BARLIGHT_OP1_Q706_7,
    B08 := O150_BARLIGHT_OP2_Q707_0,
    B09 := O160_CHECKER_LGHT_ON_Q707_1,
    B10 := O160_FUME_EXTRTR_ON_Q707_2,
    B11 := O160_MC_LMP_ON_Q707_3,
    B12 := O160_AUTOBAG_CNT_CMPLTD_Q707_4,
    B13 := O160_SAMPLE_PART_DOOR_OPN_Q707_5,
    B14 := O160_REJ_BIN_DOOR_OPN_Q707_6,
    B15 := O160_SPARE_Q707_7,
    W => OP160_MP_DO_MODULE_4); // BIT_AS_WORD
BIT_AS_WORD_4(
    B00 := O160_VFD_FWD_Q708_0,
    B01 := O160_VFD_REV_Q708_1,
    B02 := O160_VFD_STOP_Q708_2,
    B03 := O160_BOT_MC_LMP_ON_Q708_3,
    B04 := O10A_DRUM_MTR_FWD_Q708_4,
    B05 := O10A_DRUM_RST_Q708_5,
    B06 := O10A_DRUM_EXT_SPEED_Q708_6,
    B07 := O160_SPARE_Q708_7,
    B08 := O10A_DRUM_RUN_IND_Q709_0,
    B09 := O160_SPARE_Q709_1_Q709_1,
    B10 := O10A_ROB_MAN_AUTO_MODE_Q709_2,
    B11 := O10B_ROB_MAN_AUTO_MODE_Q709_3,
    B12 := O120_ROB_MAN_AUTO_MODE_Q709_4,
    B13 := O160_SPARE_Q709_5,
    B14 := O160_SPARE_Q709_6,
    B15 := O160_SPARE_Q709_7,
    W => OP160_MP_DO_MODULE_5); // BIT_AS_WORD

END_PROGRAM

// ---- POUs/IO/OP160_MASTER4_IO.TcPOU
PROGRAM OP160_MASTER4_IO
VAR
	OP160_MAS4_PORT1_BYTE1_DI_MODULE_1 AT %I* : BYTE;
	OP160_MAS4_PORT1_BYTE2_DI_MODULE_1 AT %I* : BYTE;
	OP160_MAS4_PORT2_BYTE1_DI_MODULE_2 AT %I* : BYTE;
	OP160_MAS4_PORT2_BYTE2_DI_MODULE_2 AT %I* : BYTE;
	OP160_MAS4_PORT3_BYTE1_DI_MODULE_3 AT %I* : BYTE;
	OP160_MAS4_PORT3_BYTE2_DI_MODULE_3 AT %I* : BYTE;
	OP160_MAS4_PORT4_BYTE1_DI_MODULE_4 AT %I* : BYTE;
	OP160_MAS4_PORT4_BYTE2_DI_MODULE_4 AT %I* : BYTE;
	
	OP160_MAS4_PORT5_BYTE1_DO_MODULE_1 AT %Q* : BYTE;
	OP160_MAS4_PORT5_BYTE2_DO_MODULE_1 AT %Q* : BYTE;
	OP160_MAS4_PORT5_BYTE3_DO_MODULE_1 AT %Q* : BYTE;
	OP160_MAS4_PORT5_BYTE4_DO_MODULE_1 AT %Q* : BYTE;
	OP160_MAS4_PORT6_BYTE1_DO_MODULE_2 AT %Q* : BYTE;
	OP160_MAS4_PORT6_BYTE2_DO_MODULE_2 AT %Q* : BYTE;
	OP160_MAS4_PORT6_BYTE3_DO_MODULE_2 AT %Q* : BYTE;
	OP160_MAS4_PORT6_BYTE4_DO_MODULE_2 AT %Q* : BYTE;
	
	
	

	BYTE_AS_BIT_0: BYTE_AS_BIT;
	BYTE_AS_BIT_1: BYTE_AS_BIT;
	BYTE_AS_BIT_2: BYTE_AS_BIT;
	BYTE_AS_BIT_3: BYTE_AS_BIT;
	BYTE_AS_BIT_4: BYTE_AS_BIT;
	BYTE_AS_BIT_5: BYTE_AS_BIT;
	BYTE_AS_BIT_6: BYTE_AS_BIT;
	BYTE_AS_BIT_7: BYTE_AS_BIT;
	
		
	BIT_AS_BYTE_0: BIT_AS_BYTE;
	BIT_AS_BYTE_1: BIT_AS_BYTE;
	BIT_AS_BYTE_2: BIT_AS_BYTE;
	BIT_AS_BYTE_3: BIT_AS_BYTE;
	BIT_AS_BYTE_4: BIT_AS_BYTE;
	BIT_AS_BYTE_5: BIT_AS_BYTE;
	BIT_AS_BYTE_6: BIT_AS_BYTE;
	BIT_AS_BYTE_7: BIT_AS_BYTE;
END_VAR

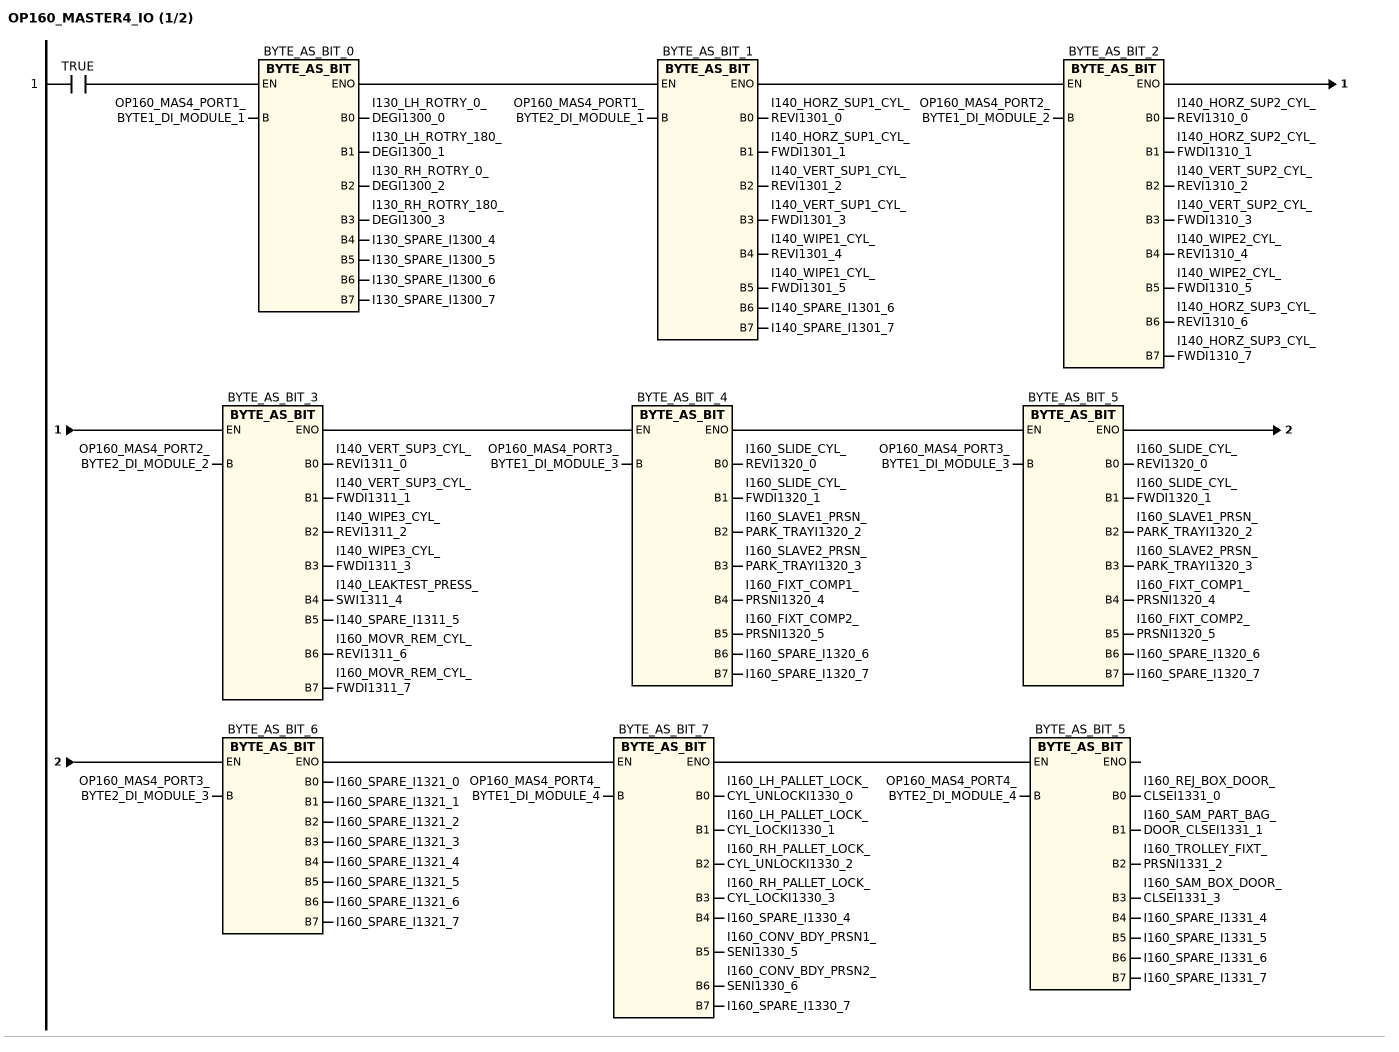
// NETWORK 1
BYTE_AS_BIT_0(
    B := OP160_MAS4_PORT1_BYTE1_DI_MODULE_1,
    B0 => I130_LH_ROTRY_0_DEGI1300_0,
    B1 => I130_LH_ROTRY_180_DEGI1300_1,
    B2 => I130_RH_ROTRY_0_DEGI1300_2,
    B3 => I130_RH_ROTRY_180_DEGI1300_3,
    B4 => I130_SPARE_I1300_4,
    B5 => I130_SPARE_I1300_5,
    B6 => I130_SPARE_I1300_6,
    B7 => I130_SPARE_I1300_7); // BYTE_AS_BIT
BYTE_AS_BIT_1(
    B := OP160_MAS4_PORT1_BYTE2_DI_MODULE_1,
    B0 => I140_HORZ_SUP1_CYL_REVI1301_0,
    B1 => I140_HORZ_SUP1_CYL_FWDI1301_1,
    B2 => I140_VERT_SUP1_CYL_REVI1301_2,
    B3 => I140_VERT_SUP1_CYL_FWDI1301_3,
    B4 => I140_WIPE1_CYL_REVI1301_4,
    B5 => I140_WIPE1_CYL_FWDI1301_5,
    B6 => I140_SPARE_I1301_6,
    B7 => I140_SPARE_I1301_7); // BYTE_AS_BIT
BYTE_AS_BIT_2(
    B := OP160_MAS4_PORT2_BYTE1_DI_MODULE_2,
    B0 => I140_HORZ_SUP2_CYL_REVI1310_0,
    B1 => I140_HORZ_SUP2_CYL_FWDI1310_1,
    B2 => I140_VERT_SUP2_CYL_REVI1310_2,
    B3 => I140_VERT_SUP2_CYL_FWDI1310_3,
    B4 => I140_WIPE2_CYL_REVI1310_4,
    B5 => I140_WIPE2_CYL_FWDI1310_5,
    B6 => I140_HORZ_SUP3_CYL_REVI1310_6,
    B7 => I140_HORZ_SUP3_CYL_FWDI1310_7); // BYTE_AS_BIT
BYTE_AS_BIT_3(
    B := OP160_MAS4_PORT2_BYTE2_DI_MODULE_2,
    B0 => I140_VERT_SUP3_CYL_REVI1311_0,
    B1 => I140_VERT_SUP3_CYL_FWDI1311_1,
    B2 => I140_WIPE3_CYL_REVI1311_2,
    B3 => I140_WIPE3_CYL_FWDI1311_3,
    B4 => I140_LEAKTEST_PRESS_SWI1311_4,
    B5 => I140_SPARE_I1311_5,
    B6 => I160_MOVR_REM_CYL_REVI1311_6,
    B7 => I160_MOVR_REM_CYL_FWDI1311_7); // BYTE_AS_BIT
BYTE_AS_BIT_4(
    B := OP160_MAS4_PORT3_BYTE1_DI_MODULE_3,
    B0 => I160_SLIDE_CYL_REVI1320_0,
    B1 => I160_SLIDE_CYL_FWDI1320_1,
    B2 => I160_SLAVE1_PRSN_PARK_TRAYI1320_2,
    B3 => I160_SLAVE2_PRSN_PARK_TRAYI1320_3,
    B4 => I160_FIXT_COMP1_PRSNI1320_4,
    B5 => I160_FIXT_COMP2_PRSNI1320_5,
    B6 => I160_SPARE_I1320_6,
    B7 => I160_SPARE_I1320_7); // BYTE_AS_BIT
BYTE_AS_BIT_5(
    B := OP160_MAS4_PORT3_BYTE1_DI_MODULE_3,
    B0 => I160_SLIDE_CYL_REVI1320_0,
    B1 => I160_SLIDE_CYL_FWDI1320_1,
    B2 => I160_SLAVE1_PRSN_PARK_TRAYI1320_2,
    B3 => I160_SLAVE2_PRSN_PARK_TRAYI1320_3,
    B4 => I160_FIXT_COMP1_PRSNI1320_4,
    B5 => I160_FIXT_COMP2_PRSNI1320_5,
    B6 => I160_SPARE_I1320_6,
    B7 => I160_SPARE_I1320_7); // BYTE_AS_BIT
BYTE_AS_BIT_6(
    B := OP160_MAS4_PORT3_BYTE2_DI_MODULE_3,
    B0 => I160_SPARE_I1321_0,
    B1 => I160_SPARE_I1321_1,
    B2 => I160_SPARE_I1321_2,
    B3 => I160_SPARE_I1321_3,
    B4 => I160_SPARE_I1321_4,
    B5 => I160_SPARE_I1321_5,
    B6 => I160_SPARE_I1321_6,
    B7 => I160_SPARE_I1321_7); // BYTE_AS_BIT
BYTE_AS_BIT_7(
    B := OP160_MAS4_PORT4_BYTE1_DI_MODULE_4,
    B0 => I160_LH_PALLET_LOCK_CYL_UNLOCKI1330_0,
    B1 => I160_LH_PALLET_LOCK_CYL_LOCKI1330_1,
    B2 => I160_RH_PALLET_LOCK_CYL_UNLOCKI1330_2,
    B3 => I160_RH_PALLET_LOCK_CYL_LOCKI1330_3,
    B4 => I160_SPARE_I1330_4,
    B5 => I160_CONV_BDY_PRSN1_SENI1330_5,
    B6 => I160_CONV_BDY_PRSN2_SENI1330_6,
    B7 => I160_SPARE_I1330_7); // BYTE_AS_BIT
BYTE_AS_BIT_5(
    B := OP160_MAS4_PORT4_BYTE2_DI_MODULE_4,
    B0 => I160_REJ_BOX_DOOR_CLSEI1331_0,
    B1 => I160_SAM_PART_BAG_DOOR_CLSEI1331_1,
    B2 => I160_TROLLEY_FIXT_PRSNI1331_2,
    B3 => I160_SAM_BOX_DOOR_CLSEI1331_3,
    B4 => I160_SPARE_I1331_4,
    B5 => I160_SPARE_I1331_5,
    B6 => I160_SPARE_I1331_6,
    B7 => I160_SPARE_I1331_7); // BYTE_AS_BIT

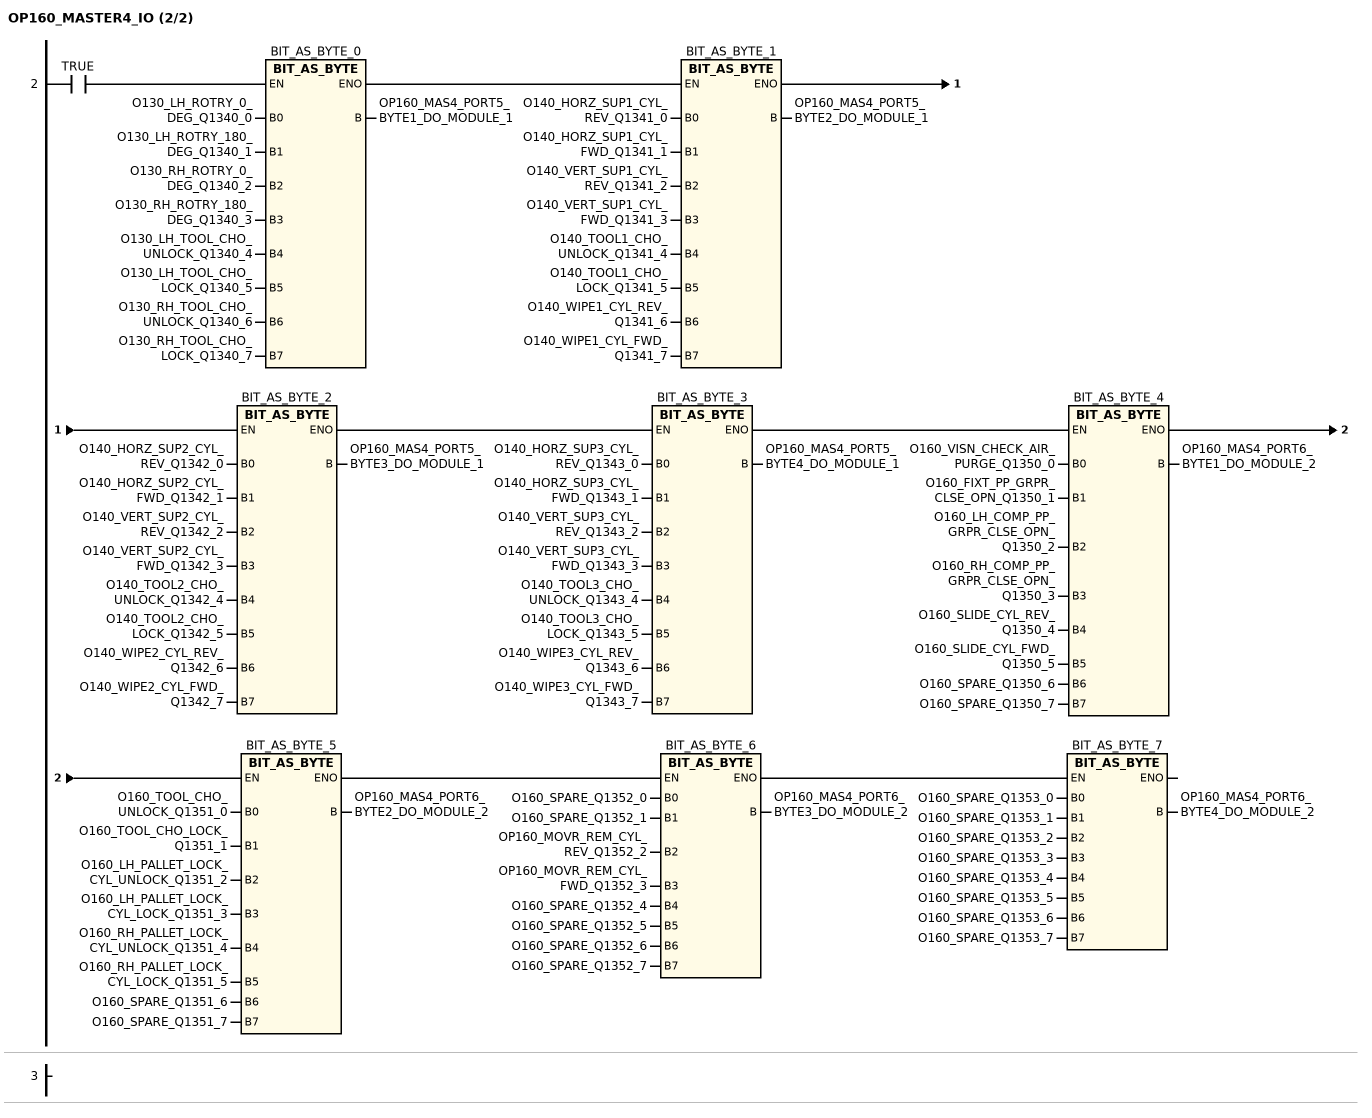
// NETWORK 2
BIT_AS_BYTE_0(
    B0 := O130_LH_ROTRY_0_DEG_Q1340_0,
    B1 := O130_LH_ROTRY_180_DEG_Q1340_1,
    B2 := O130_RH_ROTRY_0_DEG_Q1340_2,
    B3 := O130_RH_ROTRY_180_DEG_Q1340_3,
    B4 := O130_LH_TOOL_CHO_UNLOCK_Q1340_4,
    B5 := O130_LH_TOOL_CHO_LOCK_Q1340_5,
    B6 := O130_RH_TOOL_CHO_UNLOCK_Q1340_6,
    B7 := O130_RH_TOOL_CHO_LOCK_Q1340_7,
    B => OP160_MAS4_PORT5_BYTE1_DO_MODULE_1); // BIT_AS_BYTE
BIT_AS_BYTE_1(
    B0 := O140_HORZ_SUP1_CYL_REV_Q1341_0,
    B1 := O140_HORZ_SUP1_CYL_FWD_Q1341_1,
    B2 := O140_VERT_SUP1_CYL_REV_Q1341_2,
    B3 := O140_VERT_SUP1_CYL_FWD_Q1341_3,
    B4 := O140_TOOL1_CHO_UNLOCK_Q1341_4,
    B5 := O140_TOOL1_CHO_LOCK_Q1341_5,
    B6 := O140_WIPE1_CYL_REV_Q1341_6,
    B7 := O140_WIPE1_CYL_FWD_Q1341_7,
    B => OP160_MAS4_PORT5_BYTE2_DO_MODULE_1); // BIT_AS_BYTE
BIT_AS_BYTE_2(
    B0 := O140_HORZ_SUP2_CYL_REV_Q1342_0,
    B1 := O140_HORZ_SUP2_CYL_FWD_Q1342_1,
    B2 := O140_VERT_SUP2_CYL_REV_Q1342_2,
    B3 := O140_VERT_SUP2_CYL_FWD_Q1342_3,
    B4 := O140_TOOL2_CHO_UNLOCK_Q1342_4,
    B5 := O140_TOOL2_CHO_LOCK_Q1342_5,
    B6 := O140_WIPE2_CYL_REV_Q1342_6,
    B7 := O140_WIPE2_CYL_FWD_Q1342_7,
    B => OP160_MAS4_PORT5_BYTE3_DO_MODULE_1); // BIT_AS_BYTE
BIT_AS_BYTE_3(
    B0 := O140_HORZ_SUP3_CYL_REV_Q1343_0,
    B1 := O140_HORZ_SUP3_CYL_FWD_Q1343_1,
    B2 := O140_VERT_SUP3_CYL_REV_Q1343_2,
    B3 := O140_VERT_SUP3_CYL_FWD_Q1343_3,
    B4 := O140_TOOL3_CHO_UNLOCK_Q1343_4,
    B5 := O140_TOOL3_CHO_LOCK_Q1343_5,
    B6 := O140_WIPE3_CYL_REV_Q1343_6,
    B7 := O140_WIPE3_CYL_FWD_Q1343_7,
    B => OP160_MAS4_PORT5_BYTE4_DO_MODULE_1); // BIT_AS_BYTE
BIT_AS_BYTE_4(
    B0 := O160_VISN_CHECK_AIR_PURGE_Q1350_0,
    B1 := O160_FIXT_PP_GRPR_CLSE_OPN_Q1350_1,
    B2 := O160_LH_COMP_PP_GRPR_CLSE_OPN_Q1350_2,
    B3 := O160_RH_COMP_PP_GRPR_CLSE_OPN_Q1350_3,
    B4 := O160_SLIDE_CYL_REV_Q1350_4,
    B5 := O160_SLIDE_CYL_FWD_Q1350_5,
    B6 := O160_SPARE_Q1350_6,
    B7 := O160_SPARE_Q1350_7,
    B => OP160_MAS4_PORT6_BYTE1_DO_MODULE_2); // BIT_AS_BYTE
BIT_AS_BYTE_5(
    B0 := O160_TOOL_CHO_UNLOCK_Q1351_0,
    B1 := O160_TOOL_CHO_LOCK_Q1351_1,
    B2 := O160_LH_PALLET_LOCK_CYL_UNLOCK_Q1351_2,
    B3 := O160_LH_PALLET_LOCK_CYL_LOCK_Q1351_3,
    B4 := O160_RH_PALLET_LOCK_CYL_UNLOCK_Q1351_4,
    B5 := O160_RH_PALLET_LOCK_CYL_LOCK_Q1351_5,
    B6 := O160_SPARE_Q1351_6,
    B7 := O160_SPARE_Q1351_7,
    B => OP160_MAS4_PORT6_BYTE2_DO_MODULE_2); // BIT_AS_BYTE
BIT_AS_BYTE_6(
    B0 := O160_SPARE_Q1352_0,
    B1 := O160_SPARE_Q1352_1,
    B2 := OP160_MOVR_REM_CYL_REV_Q1352_2,
    B3 := OP160_MOVR_REM_CYL_FWD_Q1352_3,
    B4 := O160_SPARE_Q1352_4,
    B5 := O160_SPARE_Q1352_5,
    B6 := O160_SPARE_Q1352_6,
    B7 := O160_SPARE_Q1352_7,
    B => OP160_MAS4_PORT6_BYTE3_DO_MODULE_2); // BIT_AS_BYTE
BIT_AS_BYTE_7(
    B0 := O160_SPARE_Q1353_0,
    B1 := O160_SPARE_Q1353_1,
    B2 := O160_SPARE_Q1353_2,
    B3 := O160_SPARE_Q1353_3,
    B4 := O160_SPARE_Q1353_4,
    B5 := O160_SPARE_Q1353_5,
    B6 := O160_SPARE_Q1353_6,
    B7 := O160_SPARE_Q1353_7,
    B => OP160_MAS4_PORT6_BYTE4_DO_MODULE_2); // BIT_AS_BYTE

// NETWORK 3

END_PROGRAM

// ---- POUs/IO/OP120_JB_IO.TcPOU
PROGRAM OP120_JB_IO
VAR
OP120_JB_DI_MODULE_1 AT %I* : WORD;
OP120_JB_DI_MODULE_2 AT %I* : WORD;

OP120_JB_DO_MODULE_1 AT %Q* : WORD;
OP120_JB_DO_MODULE_2 AT %Q* : WORD;

	WORD_AS_BIT_0: WORD_AS_BIT;
	WORD_AS_BIT_1: WORD_AS_BIT;
	
	BIT_AS_WORD_0: BIT_AS_WORD;
	BIT_AS_WORD_1: BIT_AS_WORD;
END_VAR

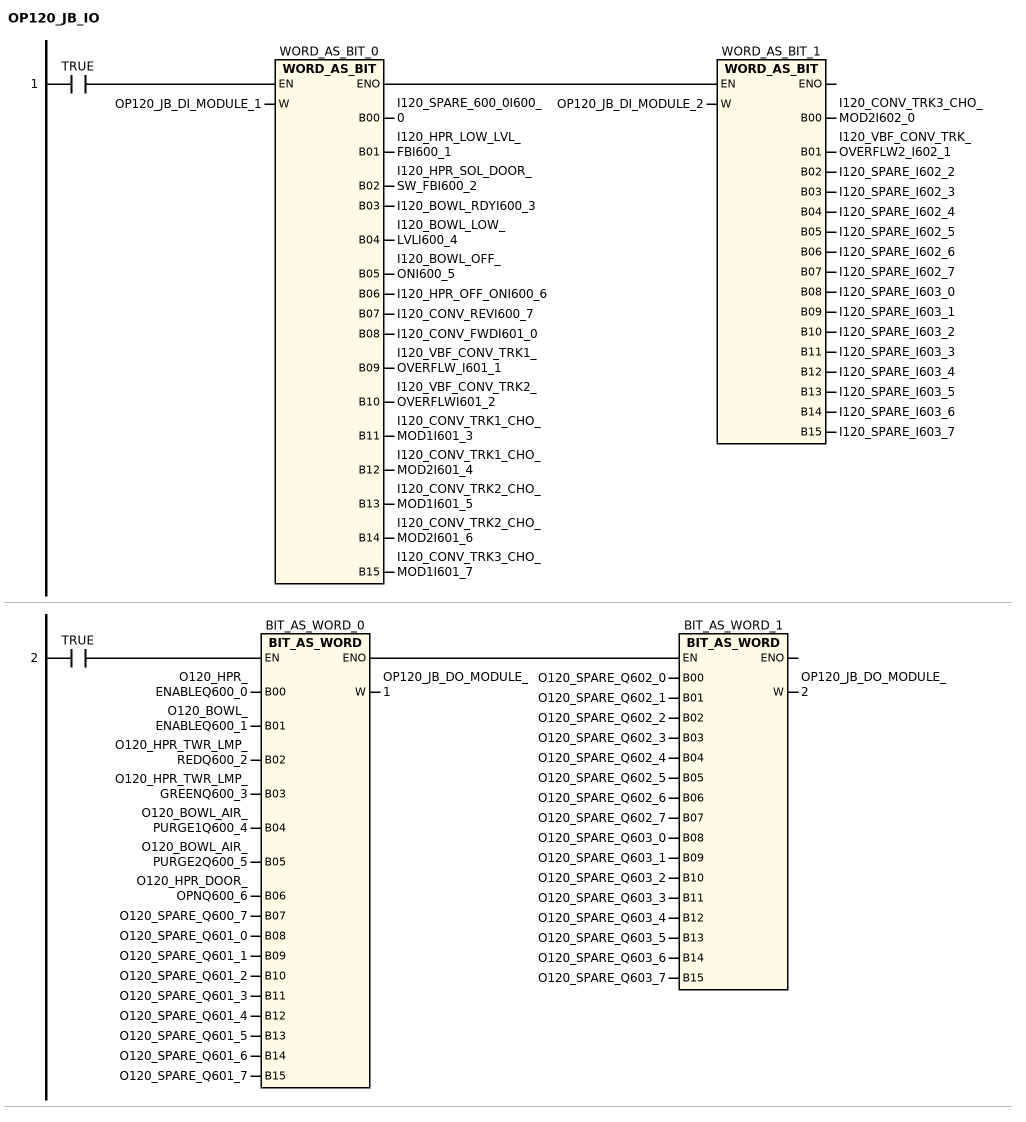
// NETWORK 1
WORD_AS_BIT_0(
    W := OP120_JB_DI_MODULE_1,
    B00 => I120_SPARE_600_0I600_0,
    B01 => I120_HPR_LOW_LVL_FBI600_1,
    B02 => I120_HPR_SOL_DOOR_SW_FBI600_2,
    B03 => I120_BOWL_RDYI600_3,
    B04 => I120_BOWL_LOW_LVLI600_4,
    B05 => I120_BOWL_OFF_ONI600_5,
    B06 => I120_HPR_OFF_ONI600_6,
    B07 => I120_CONV_REVI600_7,
    B08 => I120_CONV_FWDI601_0,
    B09 => I120_VBF_CONV_TRK1_OVERFLW_I601_1,
    B10 => I120_VBF_CONV_TRK2_OVERFLWI601_2,
    B11 => I120_CONV_TRK1_CHO_MOD1I601_3,
    B12 => I120_CONV_TRK1_CHO_MOD2I601_4,
    B13 => I120_CONV_TRK2_CHO_MOD1I601_5,
    B14 => I120_CONV_TRK2_CHO_MOD2I601_6,
    B15 => I120_CONV_TRK3_CHO_MOD1I601_7); // WORD_AS_BIT
WORD_AS_BIT_1(
    W := OP120_JB_DI_MODULE_2,
    B00 => I120_CONV_TRK3_CHO_MOD2I602_0,
    B01 => I120_VBF_CONV_TRK_OVERFLW2_I602_1,
    B02 => I120_SPARE_I602_2,
    B03 => I120_SPARE_I602_3,
    B04 => I120_SPARE_I602_4,
    B05 => I120_SPARE_I602_5,
    B06 => I120_SPARE_I602_6,
    B07 => I120_SPARE_I602_7,
    B08 => I120_SPARE_I603_0,
    B09 => I120_SPARE_I603_1,
    B10 => I120_SPARE_I603_2,
    B11 => I120_SPARE_I603_3,
    B12 => I120_SPARE_I603_4,
    B13 => I120_SPARE_I603_5,
    B14 => I120_SPARE_I603_6,
    B15 => I120_SPARE_I603_7); // WORD_AS_BIT

// NETWORK 2
BIT_AS_WORD_0(
    B00 := O120_HPR_ENABLEQ600_0,
    B01 := O120_BOWL_ENABLEQ600_1,
    B02 := O120_HPR_TWR_LMP_REDQ600_2,
    B03 := O120_HPR_TWR_LMP_GREENQ600_3,
    B04 := O120_BOWL_AIR_PURGE1Q600_4,
    B05 := O120_BOWL_AIR_PURGE2Q600_5,
    B06 := O120_HPR_DOOR_OPNQ600_6,
    B07 := O120_SPARE_Q600_7,
    B08 := O120_SPARE_Q601_0,
    B09 := O120_SPARE_Q601_1,
    B10 := O120_SPARE_Q601_2,
    B11 := O120_SPARE_Q601_3,
    B12 := O120_SPARE_Q601_4,
    B13 := O120_SPARE_Q601_5,
    B14 := O120_SPARE_Q601_6,
    B15 := O120_SPARE_Q601_7,
    W => OP120_JB_DO_MODULE_1); // BIT_AS_WORD
BIT_AS_WORD_1(
    B00 := O120_SPARE_Q602_0,
    B01 := O120_SPARE_Q602_1,
    B02 := O120_SPARE_Q602_2,
    B03 := O120_SPARE_Q602_3,
    B04 := O120_SPARE_Q602_4,
    B05 := O120_SPARE_Q602_5,
    B06 := O120_SPARE_Q602_6,
    B07 := O120_SPARE_Q602_7,
    B08 := O120_SPARE_Q603_0,
    B09 := O120_SPARE_Q603_1,
    B10 := O120_SPARE_Q603_2,
    B11 := O120_SPARE_Q603_3,
    B12 := O120_SPARE_Q603_4,
    B13 := O120_SPARE_Q603_5,
    B14 := O120_SPARE_Q603_6,
    B15 := O120_SPARE_Q603_7,
    W => OP120_JB_DO_MODULE_2); // BIT_AS_WORD

END_PROGRAM

// ---- POUs/Programs/OP150/OP150_Main.TcPOU
PROGRAM OP150_Main
VAR
	OP150_Modeselection_FB: Mode_Selection_Block1;
END_VAR

OP150_A();
OP150_B();
OP150_Laser_FB();
OP150_C();

IF (OP150_HMI_AutoMode AND NOT OP150_HMI_ManualMOde AND NOT OP150_HMI_StepMode) THEN
	OP150_Modeselection_FB.ModeWord:=1;
	ELSIF (NOT OP150_HMI_AutoMode AND OP150_HMI_ManualMOde AND NOT OP150_HMI_StepMode) THEN
		OP150_Modeselection_FB.ModeWord:=2;
	ELSIF  (NOT OP150_HMI_AutoMode AND NOT OP150_HMI_ManualMOde AND  OP150_HMI_StepMode) THEN
		OP150_Modeselection_FB.ModeWord:=3;
    ELSE   
		OP150_Modeselection_FB.ModeWord:=0;
END_IF
	

OP150_Modeselection_FB(
	ModeWord:= , 
	HomeConditionOK:=OP150_HomeCondition_OK , 
	OperationEnable:=OperationEnable , 
	StartPB:= , 
	SafetyAndNOError:=OperationEnable , 
	ModeAck:=TRUE , 
	HomingINProgress:= , 
	TempHomeOK:=OP150_Temp_Home_OK , 
	ResetPB:= , 
	AutoSelected=>OP150_AutoSelected , 
	ManualSelected=>OP150_ManualSelected , 
	StepSelected=>OP150_StepSelected , 
	ModeSelAck_Indication=> , 
	StatusDisplay=> , 
	AutoRunning:=OP150_AutoRunning , 
	StepRunning:=OP150_StepRunning , 
	StartEnable:=OP150_StartEnable , 
	MachineStop:=OP150_Machine_Stop );

END_PROGRAM

// ---- POUs/Programs/OP150/OP150_A.TcPOU
PROGRAM OP150_A
VAR
	OP150_Final_Camera 			  : FB_Cognex_ProfiNET_1;
	OP150_Camera_Trigger		  : BOOL;
	OP150_Camera_Job_Change_start : BOOL;
	OP150_Camera_Error			  : BOOL;
	OP150_Camera_Ready			  : BOOL;
	OP150_Camera_Online			  : BOOL;	
	
	OP150_Acquisition_Status AT %I*  :Acquisition_Status;
	OP150_Inspection_Status  AT %I*  :Inspection_Status;	
	OP150_Acquisition_ID     AT %I*  :UINT;
	OP150_Inspection_ID   	 AT %I*  :UINT;
	OP150_Error_code      	 AT %I*  :UINT;
	OP150_Current_Job_ID  	 AT %I*  :UINT;
	OP150_Result_code     	 AT %I*  :UINT;
	OP150_Cam_Result      	 AT %I*  :ARRAY[0..63] OF BYTE;
	
	OP150_User_Data      	 AT %Q*  :ARRAY[0..63] OF BYTE;
	OP150_Acquisition_Control AT %Q*  : Acquisition_Control;
	OP150_Inspection_Control  AT %Q*  : Inspection_Control;
	OP150_Command_word		  AT %Q*  : UINT;
	Error_status				      : STRING;
	OP150_Target_Job_ID				  : UINT;
	OP150_Loaded_Job_ID		    	  : UINT;
	OP150_Union                       : UNION_64Byte;
	OP150_Job_Change_Complete		  : BOOL;
	OP150_Job_Change_Error   		  : BOOL;
	OP150_Picture_Taken      		  : BOOL;
	OP150_Result_OK					  : BOOL;
	OP150_Result_NOK				  : BOOL;

	OP150A_STN_MOVER	: INT;

	OP150A_LH_STN_MOVER: INT;
	OP150A_RH_STN_MOVER: INT;
    OP150A_LH_STN_ENABLE: BOOL;
    OP150A_RH_STN_ENABLE: BOOL;		
	Dry_run             : BOOL;
	Complete_Delay      : TON;
	Error_Delay	: TON;
	tmp: BOOL;
	
	OP150_LH_CMP_OK: BOOL;
	OP150_LH_CMP_NOK: BOOL;
	tmr: Ton;
	tmr1: Ton;
	
	OP150a_Auto_Seq		: INT;
	Fixture_LH 			: INT;
	Fixture_RH 	 		: INT;
	Inspection_ID_Temp	: UINT;
	
	OP150A_Cam_Job_Change_FB : Camera_Job_Change;
	OP150a_Job_Change_Start	 : BOOL;
	OP150a_Targ_Job_ID		 : UINT;
	OP150A_Job_OK 			 : BOOL;
	
	Toggle_Pos : R_TRIG;
	Toggle_Neg : F_TRIG;
	LH_Cam_Completed : BOOL;
END_VAR

Toggle_Pos(CLK:=OP150_A.OP150_Inspection_Status.Inspection_Completed);
Toggle_Neg(CLK:=OP150_A.OP150_Inspection_Status.Inspection_Completed);

IF Toggle_Pos.Q OR Toggle_Neg.Q THEN
	LH_Cam_Completed:=1;	
END_IF


OP150_Final_Camera(
	tTimeout:= , 
	sJob_Name:= , 
	camera_ready=> OP150_Camera_Ready,
	Camera_online=> OP150_Camera_Online,
	stCognex_record_status:=OP150_Acquisition_Status, 
	Acquisition_ID:=OP150_Acquisition_ID , 
	stCognex_Inspection_status:=OP150_Inspection_Status, 
	Error_Code:=OP150_Error_code , 
	wcommand_control_in:= OP150_Current_Job_ID, 
	aResults_64_Bytes:= OP150_Cam_Result, 
	number_of_inspections:=OP150_Inspection_ID , 
	iresult_code:= OP150_Result_code, 
	bTarget_job_ID:=OP150_Target_Job_ID , 
	Error_Status_message=> Error_status, 
	bError=> OP150_Camera_Error, 
	stCognex_record_control=>OP150_Acquisition_Control , 
	stCognex_inspection_control=>OP150_Inspection_Control , 
	wCommandControl_out=>OP150_Command_word , 
	aUser_data_64_Byte=> OP150_Union.aArrayOfByte, 
	bJob_loading_completed=>OP150_Job_Change_Complete , 
	bJob_load_failed=>OP150_Job_Change_Error , 
	bInspection_Result_IO=>  OP150_Result_OK, 
	bInspection_Result_NIO=> OP150_Result_NOK, 
	bTXTSM_Error_Job_Change=> , 
	bPictureTakenComplete=> OP150_Picture_Taken, 
	Loaded_Job_ID=>OP150_Loaded_Job_ID	 , 
	bClear_Error:= HMI_Reset, 
	bJob_change_start:= OP150_Camera_Job_Change_start, 
	TXTSM_camera_not_online=>	 , 
	bTrigger_start:= OP150_Camera_Trigger );

IF HMI_Reset OR OP150_HMI_Reset THEN
	OP150_A_ErrorActive:=0;
END_IF	

Error_Delay(IN:= NOT OP150_Camera_Online,PT:=T#10S);
	
IF Error_Delay.Q THEN
	OP150_A_ErrorActive:=1;
END_IF


IF OP150_A_ErrorActive OR NOT OperationEnable THEN
	OP150a_Auto_Seq:=10;
END_IF

CASE OP150a_Auto_Seq OF
	10: IF NOT OP150_A_ErrorActive THEN
		 	OP150a_Auto_Seq :=20;
		END_IF
		
	20: IF OP150_Camera_Online THEN
			OP150a_Auto_Seq :=30;
		END_IF
		
	30: IF OP150_Camera_Online THEN
			OP150A_RH_CMP_OK	:= FALSE;
			OP150A_LH_CMP_OK	:= FALSE;
			OP150a_Auto_Seq :=40;
		END_IF
	
	40: IF OP150A_LH_STN_ENABLE THEN
			IF Fixture_LH=140 THEN
				OP150a_Auto_Seq :=50;
			ELSE
				OP150a_Auto_Seq :=90;	
			END_IF
		ELSIF OP150A_RH_STN_ENABLE THEN
			IF  Fixture_RH=140 THEN
				OP150a_Auto_Seq :=100;
			ELSE
				OP150a_Auto_Seq :=90;	
			END_IF
		END_IF
		
	50: OP150_Camera_Trigger:=1;
		IF LH_Cam_Completed THEN
			OP150_Camera_Trigger:=0;
			OP150a_Auto_Seq :=60;
		END_IF	
	
	60: IF OP150_Cam_Result[0]=1  THEN
			OP150a_Auto_Seq :=70;	
		ELSIF OP150_Cam_Result[1]=1 THEN
			OP150a_Auto_Seq :=76;
		END_IF
			
	70:	OP150A_LH_CMP_OK	:= TRUE;
		OP150a_Auto_Seq :=75;
	
	75: MOVER_CMP_STATUS[OP150A_LH_STN_MOVER][1]:=150;
		IF MOVER_CMP_STATUS[OP150A_LH_STN_MOVER][1]=150 THEN
			OP150a_Auto_Seq :=80;
		END_IF

	76: MOVER_CMP_STATUS[OP150A_LH_STN_MOVER][1]	:=151;
		IF MOVER_CMP_STATUS[OP150A_LH_STN_MOVER][1] =151 THEN
			OP150a_Auto_Seq :=80;
		END_IF	
		
	80: OP150A_LH_STN_ENABLE:=0;
		LH_Cam_Completed:=0;
		STATION_DONE[OP150A_RH_STN_MOVER][OP150A_LH_XTS_POS_NO]	:= TRUE;
		OP150a_Auto_Seq :=30;
		
	90: OP150A_LH_STN_ENABLE:=0;
		OP150A_RH_STN_ENABLE:=0;
		STATION_DONE[OP150A_RH_STN_MOVER][OP150A_LH_XTS_POS_NO]	:= TRUE;
		OP150a_Auto_Seq :=30;	
		
	100:  OP150_Camera_Trigger:=1;
		IF LH_Cam_Completed THEN
			OP150_Camera_Trigger:=0;
			OP150a_Auto_Seq :=110;
		END_IF	
	
	110: IF OP150_Cam_Result[0]=1  THEN
			OP150a_Auto_Seq :=115;	
		ELSIF OP150_Cam_Result[1]=1 THEN
			OP150a_Auto_Seq :=126;
		END_IF
			
	115:OP150A_RH_CMP_OK:= TRUE;
		OP150a_Auto_Seq :=125;
		
	125: MOVER_CMP_STATUS[OP150A_RH_STN_MOVER][2]:=150;
		 IF MOVER_CMP_STATUS[OP150A_RH_STN_MOVER][2]=150 THEN
			OP150a_Auto_Seq :=130;
		 END_IF

	126:  MOVER_CMP_STATUS[OP150A_RH_STN_MOVER][2]:=151;
		 IF MOVER_CMP_STATUS[OP150A_RH_STN_MOVER][2]=151 THEN
			OP150a_Auto_Seq :=130;
		 END_IF	

	130: OP150A_RH_STN_ENABLE:=0;
		 LH_Cam_Completed:=0;
	 	 STATION_DONE[OP150A_RH_STN_MOVER][OP150A_RH_XTS_POS_NO]:= TRUE;
		 OP150a_Auto_Seq :=30;	
END_CASE

IF Dry_run THEN
	Fixture_LH	:=140;
	Fixture_RH  :=140;
ELSE	
    Fixture_LH:=MOVER_CMP_STATUS[OP150A_LH_STN_MOVER][1];
    Fixture_RH:=MOVER_CMP_STATUS[OP150A_RH_STN_MOVER][2];
END_IF

OP150A_Cam_Job_Change_FB(
	Target_Job_ID:= OP150a_Targ_Job_ID, 
	Block_Reset:= , 
	Job_Change_Start:= OP150a_Job_Change_Start, 
	Job_Change_Start_FB:= OP150_Camera_Job_Change_start, 
	Job_Change_Error_FB:= OP150_Job_Change_Error, 
	Job_Change_Completed_FB:= OP150_Job_Change_Complete,  
	Camera_Error_FB:= OP150_Camera_Error, 
	Camera_Online_FB:= OP150_Camera_Online, 
	Loaded_Job_ID_FB:= OP150_Current_Job_ID, 
	Target_Job_ID_FB:= OP150_Target_Job_ID);

IF OP150_Model='6.3' THEN
	OP150_Target_Job_ID:=2;
ELSIF OP150_Model='7.89' THEN
	OP150_Target_Job_ID:=1;
END_IF

IF OP150_Model='6.3' AND OP150_Current_Job_ID=2 THEN
	OP150a_Job_Change_Start:=0;
	OP150A_Job_OK:=1;
ELSIF OP150_Model='7.89' AND OP150_Current_Job_ID=1 THEN
	OP150a_Job_Change_Start:=0;
	OP150A_Job_OK:=1;
ELSE
    OP150a_Job_Change_Start:=1;
	OP150A_Job_OK:=0;
END_IF


	
(*IF 	(OP150A_LH_Start OR OP150A_LH_STN_ENABLE) AND NOT OP150_A_ErrorActive AND OP150_Camera_Ready AND OP150_Camera_Online THEN
 	IF  MOVER_CMP_STATUS[OP150A_LH_STN_MOVER][1]=145 THEN	
		OP150_Camera_Trigger:=1;
		tmp:=1;
		IF OP150_Cam_Result[0]=1 AND Complete_Delay.Q THEN
			OP150_Camera_Trigger:=0;
			OP150_LH_CMP_OK				:= TRUE;
			MOVER_CMP_STATUS[OP150A_LH_STN_MOVER][1]:=150;
			tmp:=1;
		ELSIF OP150_Cam_Result[0]=2 AND Complete_Delay.Q THEN
			OP150_Camera_Trigger:=0;
			OP150_LH_CMP_NOK				:= TRUE;
			MOVER_CMP_STATUS[OP150A_LH_STN_MOVER][1]:=151;
			tmp:=1;	
		END_IF
 	ELSIF MOVER_CMP_STATUS[OP150A_LH_STN_MOVER][1]<>145 THEN
		 	MOVER_CMP_STATUS[OP150A_LH_STN_MOVER][1]:=151;
			ALL_STATION_DONE.POSITION_DONE[OP150A_LH_XTS_POS_NO]:= TRUE;
			OP150A_LH_Start:=0;
 	END_IF	
END_IF

IF (OP150_LH_CMP_OK OR OP150_LH_CMP_NOK) AND MOVER_CMP_STATUS[OP150A_LH_STN_MOVER][1]=150 THEN
	ALL_STATION_DONE.POSITION_DONE[OP150A_LH_XTS_POS_NO]:= TRUE;
	OP150A_LH_Start:=0;
END_IF
IF (OP150_LH_CMP_OK OR OP150_LH_CMP_NOK)AND MOVER_CMP_STATUS[OP150A_LH_STN_MOVER][1]=151 THEN
	ALL_STATION_DONE.POSITION_DONE[OP150A_LH_XTS_POS_NO]:= TRUE;
	OP150A_LH_Start:=0;
END_IF
	
IF 	(OP150A_RH_Start OR OP150A_RH_STN_ENABLE) AND NOT OP150_A_ErrorActive AND OP150_Camera_Ready AND OP150_Camera_Online THEN
 	IF  MOVER_CMP_STATUS[OP150A_RH_STN_MOVER][2]=145 THEN	
		OP150_Camera_Trigger:=1;
		tmp:=1;
		IF OP150_Cam_Result[0]=1 AND Complete_Delay.Q THEN
			OP150_Camera_Trigger:=0;
			MOVER_CMP_STATUS[OP150A_RH_STN_MOVER][2]:=150;
			tmp:=1;

		ELSIF OP150_Cam_Result[0]=2 AND Complete_Delay.Q  THEN
			OP150_Camera_Trigger:=0;
			MOVER_CMP_STATUS[OP150A_RH_STN_MOVER][2]:=151;
			tmp:=1;

		END_IF
 	ELSIF MOVER_CMP_STATUS[OP150A_RH_STN_MOVER][2]<>145 THEN
		 	MOVER_CMP_STATUS[OP150A_RH_STN_MOVER][2]:=151;
			ALL_STATION_DONE.POSITION_DONE[OP150A_RH_XTS_POS_NO]:= TRUE;
			OP150A_RH_Start:=0;
 	END_IF	
END_IF	
			IF Complete_Delay.Q AND MOVER_CMP_STATUS[OP150A_RH_STN_MOVER][2]=150 THEN
				ALL_STATION_DONE.POSITION_DONE[OP150A_RH_XTS_POS_NO]:= TRUE;
				OP150A_RH_Start:=0;
			END_IF
			IF Complete_Delay.Q AND MOVER_CMP_STATUS[OP150A_RH_STN_MOVER][2]=151 THEN
				ALL_STATION_DONE.POSITION_DONE[OP150A_RH_XTS_POS_NO]:= TRUE;
				OP150A_RH_Start:=0;
			END_IF	
	
	OP150A_LH_STN_MOVER					:= MOVER_POSITION[OP150A_LH_XTS_POS_NO];
	OP150A_RH_STN_MOVER					:= MOVER_POSITION[OP150A_RH_XTS_POS_NO];*)	


//**********************************************************************************************************\\
OP150A_LH_STN_MOVER					:= MOVER_POSITION[OP150A_LH_XTS_POS_NO];
OP150A_RH_STN_MOVER					:= MOVER_POSITION[OP150A_RH_XTS_POS_NO];

IF AUTO_WITH_XTS THEN
//#########################################		LH 	##########################################
	IF OP150A_LH_STN_MOVER>0 THEN
	IF NOT (END_OF_CYCLE AND MOVER_CMP_STATUS[OP150A_LH_STN_MOVER][1]=5) THEN		
		OP150A_LH_STN_ENABLE		:= MOVER_POS_RECHED[OP150A_LH_STN_MOVER] AND (MOVER_CMP_STATUS[OP150A_LH_STN_MOVER][1]>130);
	ELSE
	STATION_DONE[OP150A_LH_STN_MOVER][OP150A_LH_XTS_POS_NO]			:= TRUE;	
	END_IF
	ELSE
		OP150A_LH_STN_ENABLE		:= FALSE;
	END_IF	
	STATION_DONE[OP150A_LH_STN_MOVER][OP150A_LH_XTS_POS_NO]			:= TRUE;
//#########################################		RH 	##########################################
	IF OP150A_RH_STN_MOVER>0 THEN
	IF NOT(END_OF_CYCLE AND MOVER_CMP_STATUS[OP150A_RH_STN_MOVER][2]=5)THEN			
		OP150A_RH_STN_ENABLE		:= MOVER_POS_RECHED[OP150A_RH_STN_MOVER] AND (MOVER_CMP_STATUS[OP150A_RH_STN_MOVER][2]>130);
	ELSE
	STATION_DONE[OP150A_RH_STN_MOVER][OP150A_RH_XTS_POS_NO]			:= TRUE;		
	END_IF
	ELSE
		OP150A_RH_STN_ENABLE		:= FALSE;
	END_IF	 	
END_IF	



STATION_DONE[OP150A_LH_STN_MOVER][OP150A_LH_XTS_POS_NO]		:= tmr.Q;
IF tmr.Q THEN
	MOVER_CMP_STATUS[OP150A_LH_STN_MOVER][2]:=150;
	MOVER_CMP_STATUS[OP150A_LH_STN_MOVER][1]:=150;	
END_IF
tmr(IN:=OP150A_LH_STN_ENABLE , PT:= T#800MS, Q=> , ET=> );	

STATION_DONE[OP150A_RH_STN_MOVER][OP150A_RH_XTS_POS_NO]		:= tmr1.Q;
IF tmr1.Q THEN
	MOVER_CMP_STATUS[OP150A_RH_STN_MOVER][2]:=150;
	MOVER_CMP_STATUS[OP150A_RH_STN_MOVER][1]:=150;	
END_IF
tmr1(IN:=OP150A_RH_STN_ENABLE , PT:= T#800MS, Q=> , ET=> );

END_PROGRAM

// ---- POUs/Programs/OP30/Camera_Job_Change.TcPOU
FUNCTION_BLOCK Camera_Job_Change
VAR_INPUT
	Target_Job_ID	: UINT;
	Block_Reset		: BOOL;
END_VAR
VAR_OUTPUT
	Job_Change_Completed	: BOOL;
	Job_Change_Error		: BOOL;
END_VAR
VAR_IN_OUT
	Job_Change_Start_FB		: BOOL;
	Job_Change_Error_FB		: BOOL;
	Job_Change_Completed_FB	: BOOL;
	Camera_Error_FB			: BOOL;
	Camera_Online_FB		: BOOL;
	Loaded_Job_ID_FB		: UINT;	
	Target_Job_ID_FB		: UINT;
	Job_Change_Start		: BOOL;
END_VAR

VAR
	Job_Change_Step_no		: INT;
END_VAR

IF NOT Job_Change_Start OR NOT Camera_Online_FB OR Camera_Error_FB OR Block_Reset THEN
	Job_Change_Step_no:=1;
END_IF

CASE Job_Change_Step_no OF
	
	1: IF Job_Change_Start THEN
		Job_Change_Completed:=0;
		Job_Change_Error:=0;
		Job_Change_Step_no:=10;
	   END_IF
	   
	10: IF Target_Job_ID <> Loaded_Job_ID_FB THEN
			Target_Job_ID_FB:=Target_Job_ID;
			Job_Change_Step_no:=20;
		ELSE
			Job_Change_Completed:=1;
			Job_Change_Start:=0;
			Job_Change_Step_no:=1;
	    END_IF
		
	20: Job_Change_Start_FB:=Job_Change_Start;	
		IF Job_Change_Completed_FB AND NOT (Job_Change_Error_FB OR Camera_Error_FB) THEN
			Job_Change_Completed:=Job_Change_Completed_FB;
			Job_Change_Start	:=0;
			Job_Change_Start_FB :=0;
			Job_Change_Step_no	:=1;
		ELSIF Job_Change_Error_FB THEN	
			Job_Change_Error	:=1;
			Job_Change_Start	:=0;
			Job_Change_Start_FB :=0;
			Job_Change_Step_no  :=1;			
		END_IF	
		
END_CASE

END_FUNCTION_BLOCK

// ---- POUs/Programs/OP150/OP150_B.TcPOU
PROGRAM OP150_B
VAR
	OP150b_Auto_Seq			: INT;
	OP150b_Job_Change_Seq	: INT;
	Job_Change_Seq_Start  	: BOOL;
	OP150b_Text_Change_Seq  : INT;
	Text_Change_Seq_Start  	: BOOL;
	Batch_Change			: BOOL;
	
	OP150B_STN_MOVER	: INT;
	OP150B_LH_STN_MOVER: INT;
	OP150B_RH_STN_MOVER: INT;
    OP150B_LH_STN_ENABLE: BOOL;
    OP150B_RH_STN_ENABLE: BOOL;

	Line_1: STRING ;	
	Line_2: STRING ;
	Line_3: STRING ;
	
	Rejection_Code : STRING;
	Temp_String	   : STRING;
	
	Laser_Mark_Delay : TON;
	Fixture_LH  : INT;
	Fixture_RH  : INT;
	Dry_run 	: BOOL;
	OP150B_Job_OK	: BOOL :=0;
	OP150B_Text_OK  : BOOL ;
	temp : BOOL;
	Timer : TON;
	Txt_Change_Tmr : TON;
	Laser_Marked : BOOL;
	Txt_Changed  : BOOL;

	Laser_R			     : R_TRIG;
	Text_Change_R		 : R_TRIG;
	Job_Initialize      : BOOL;
END_VAR


IF OP150_B_ErrorActive OR NOT OperationEnable OR NOT OP150B_Job_OK THEN
	OP150b_Auto_Seq:=10;
END_IF

Line_2:=Laser_Line2;
Line_3:=Laser_Line3;

Laser_R(CLK:=OP150_Laser_Completed);
IF Laser_R. Q THEN
	Laser_Marked:=1;
END_IF

Text_Change_R(CLK:=OP150_Lsr_Text_Change_Complete);
IF Text_Change_R. Q THEN
	//Laser_Marked:=1;
END_IF


CASE OP150b_Auto_Seq OF 
	10: IF NOT OP150_B_ErrorActive THEN
		 	OP150b_Auto_Seq :=20;
		END_IF
		
	20: IF OP150_Lsr_Ready AND OP150B_Job_OK AND OP150B_Text_OK THEN
			OP150b_Auto_Seq :=30;
		END_IF
		
	30: Laser_Marked:=0;
		IF OP150B_LH_STN_ENABLE THEN
			IF Fixture_LH=150 THEN
				OP150b_Auto_Seq :=40;
			ELSE
				OP150b_Auto_Seq :=60;	
			END_IF
		ELSIF OP150B_RH_STN_ENABLE THEN
			IF  Fixture_RH=150 THEN
				OP150b_Auto_Seq :=100;
			ELSE
				OP150b_Auto_Seq :=140;	
			END_IF
		END_IF
		
	40:	IF OP150B_Text_OK THEN// NOT OP150_Lsr_Text_Change_Start THEN
			OP150_Laser_Start := TRUE;
			IF OP150_Laser_Start THEN
				OP150b_Auto_Seq :=46;
			END_IF	
		END_IF	
		
